SYSTEM OPCUATests
  (* Version 1.0, 2018-08-29, Alois Zoitl, Johannes Kepler University, initial API and implementation and/or initial documentation *)
  APPLICATION OpcUWrongParameters
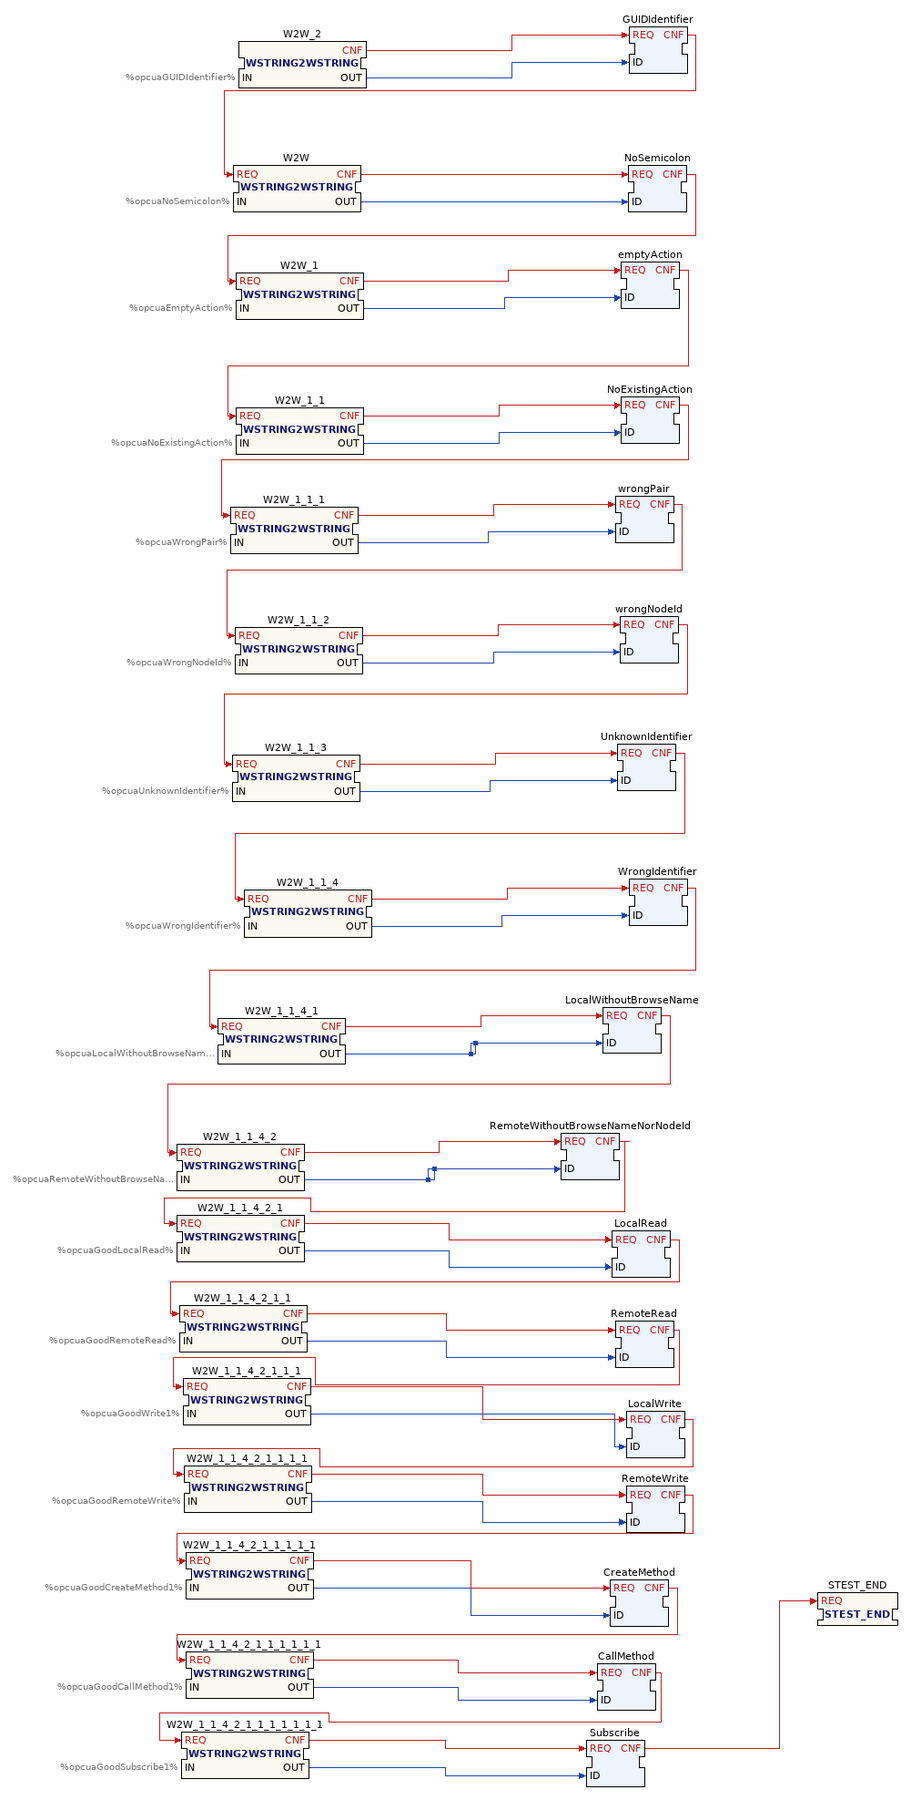
    FBS
      STEST_END : STEST_END;
      W2W : WSTRING2WSTRING(IN := %opcuaNoSemicolon%);
      W2W_1 : WSTRING2WSTRING(IN := %opcuaEmptyAction%);
      W2W_1_1 : WSTRING2WSTRING(IN := %opcuaNoExistingAction%);
      W2W_1_1_1 : WSTRING2WSTRING(IN := %opcuaWrongPair%);
      W2W_1_1_2 : WSTRING2WSTRING(IN := %opcuaWrongNodeId%);
      W2W_1_1_3 : WSTRING2WSTRING(IN := %opcuaUnknownIdentifier%);
      W2W_1_1_4 : WSTRING2WSTRING(IN := %opcuaWrongIdentifier%);
      W2W_1_1_4_1 : WSTRING2WSTRING(IN := %opcuaLocalWithoutBrowseName%);
      W2W_1_1_4_2 : WSTRING2WSTRING(IN := %opcuaRemoteWithoutBrowseNameNorNodeId%);
      W2W_1_1_4_2_1 : WSTRING2WSTRING(IN := %opcuaGoodLocalRead%);
      W2W_1_1_4_2_1_1 : WSTRING2WSTRING(IN := %opcuaGoodRemoteRead%);
      W2W_1_1_4_2_1_1_1 : WSTRING2WSTRING(IN := %opcuaGoodWrite1%);
      W2W_1_1_4_2_1_1_1_1 : WSTRING2WSTRING(IN := %opcuaGoodRemoteWrite%);
      W2W_1_1_4_2_1_1_1_1_1 : WSTRING2WSTRING(IN := %opcuaGoodCreateMethod1%);
      W2W_1_1_4_2_1_1_1_1_1_1 : WSTRING2WSTRING(IN := %opcuaGoodCallMethod1%);
      W2W_1_1_4_2_1_1_1_1_1_1_1 : WSTRING2WSTRING(IN := %opcuaGoodSubscribe1%);
      W2W_2 : WSTRING2WSTRING(IN := %opcuaGUIDIdentifier%);
    END_FBS
    SUBAPPLICATION NoSemicolon
      EVENT_INPUT
        REQ;
      END_EVENT
      EVENT_OUTPUT
        CNF;
      END_EVENT
      VAR_INPUT
        ID : WSTRING;
      END_VAR
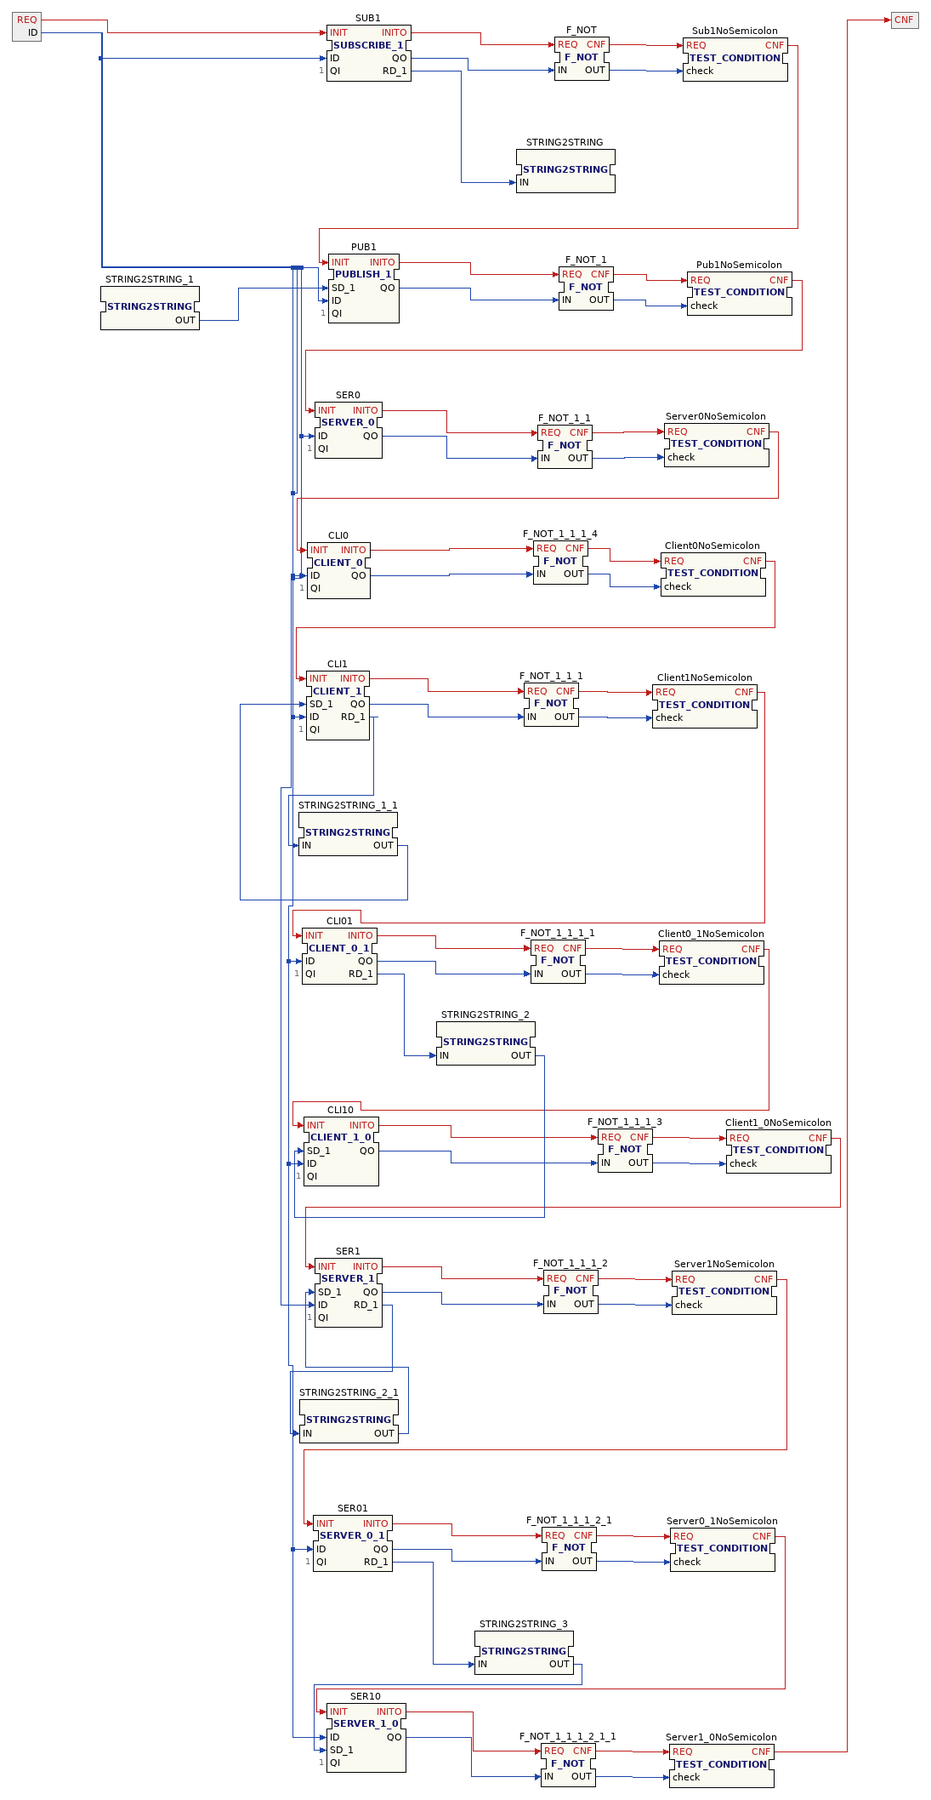
      FBS
        F_NOT_1_1_1 : F_NOT;
        Client1NoSemicolon : TEST_CONDITION;
        Pub1NoSemicolon : TEST_CONDITION;
        F_NOT_1_1 : F_NOT;
        PUB1 : PUBLISH_1(QI := 1);
        F_NOT : F_NOT;
        Server0NoSemicolon : TEST_CONDITION;
        Sub1NoSemicolon : TEST_CONDITION;
        F_NOT_1 : F_NOT;
        STRING2STRING : STRING2STRING;
        SUB1 : SUBSCRIBE_1(QI := 1);
        SER0 : SERVER_0(QI := 1);
        STRING2STRING_1 : STRING2STRING;
        Client0_1NoSemicolon : TEST_CONDITION;
        F_NOT_1_1_1_1 : F_NOT;
        Server1NoSemicolon : TEST_CONDITION;
        F_NOT_1_1_1_2 : F_NOT;
        CLI1 : CLIENT_1(QI := 1);
        CLI01 : CLIENT_0_1(QI := 1);
        Client1_0NoSemicolon : TEST_CONDITION;
        F_NOT_1_1_1_3 : F_NOT;
        CLI10 : CLIENT_1_0(QI := 1);
        STRING2STRING_1_1 : STRING2STRING;
        F_NOT_1_1_1_4 : F_NOT;
        Client0NoSemicolon : TEST_CONDITION;
        CLI0 : CLIENT_0(QI := 1);
        SER1 : SERVER_1(QI := 1);
        F_NOT_1_1_1_2_1 : F_NOT;
        Server0_1NoSemicolon : TEST_CONDITION;
        STRING2STRING_2 : STRING2STRING;
        STRING2STRING_2_1 : STRING2STRING;
        SER01 : SERVER_0_1(QI := 1);
        STRING2STRING_3 : STRING2STRING;
        Server1_0NoSemicolon : TEST_CONDITION;
        F_NOT_1_1_1_2_1_1 : F_NOT;
        SER10 : SERVER_1_0(QI := 1);
      END_FBS
      EVENT_CONNECTIONS
        F_NOT_1_1_1.CNF TO Client1NoSemicolon.REQ;
        F_NOT_1.CNF TO Pub1NoSemicolon.REQ;
        Pub1NoSemicolon.CNF TO SER0.INIT;
        SER0.INITO TO F_NOT_1_1.REQ;
        F_NOT_1_1.CNF TO Server0NoSemicolon.REQ;
        Sub1NoSemicolon.CNF TO PUB1.INIT;
        PUB1.INITO TO F_NOT_1.REQ;
        SUB1.INITO TO F_NOT.REQ;
        F_NOT.CNF TO Sub1NoSemicolon.REQ;
        REQ TO SUB1.INIT;
        F_NOT_1_1_1_1.CNF TO Client0_1NoSemicolon.REQ;
        F_NOT_1_1_1_2.CNF TO Server1NoSemicolon.REQ;
        CLI1.INITO TO F_NOT_1_1_1.REQ;
        CLI01.INITO TO F_NOT_1_1_1_1.REQ;
        CLI0.INITO TO F_NOT_1_1_1_4.REQ;
        F_NOT_1_1_1_4.CNF TO Client0NoSemicolon.REQ;
        F_NOT_1_1_1_3.CNF TO Client1_0NoSemicolon.REQ;
        CLI10.INITO TO F_NOT_1_1_1_3.REQ;
        SER1.INITO TO F_NOT_1_1_1_2.REQ;
        F_NOT_1_1_1_2_1.CNF TO Server0_1NoSemicolon.REQ;
        SER01.INITO TO F_NOT_1_1_1_2_1.REQ;
        Server0NoSemicolon.CNF TO CLI0.INIT;
        Client0NoSemicolon.CNF TO CLI1.INIT;
        Client1NoSemicolon.CNF TO CLI01.INIT;
        Client0_1NoSemicolon.CNF TO CLI10.INIT;
        Client1_0NoSemicolon.CNF TO SER1.INIT;
        Server1NoSemicolon.CNF TO SER01.INIT;
        F_NOT_1_1_1_2_1_1.CNF TO Server1_0NoSemicolon.REQ;
        Server1_0NoSemicolon.CNF TO CNF;
        Server0_1NoSemicolon.CNF TO SER10.INIT;
        SER10.INITO TO F_NOT_1_1_1_2_1_1.REQ;
      END_CONNECTIONS
      DATA_CONNECTIONS
        F_NOT_1_1_1.OUT TO Client1NoSemicolon.check;
        F_NOT_1.OUT TO Pub1NoSemicolon.check;
        SER0.QO TO F_NOT_1_1.IN;
        F_NOT_1_1.OUT TO Server0NoSemicolon.check;
        STRING2STRING_1.OUT TO PUB1.SD_1;
        PUB1.QO TO F_NOT_1.IN;
        SUB1.QO TO F_NOT.IN;
        F_NOT.OUT TO Sub1NoSemicolon.check;
        SUB1.RD_1 TO STRING2STRING.IN;
        F_NOT_1_1_1_1.OUT TO Client0_1NoSemicolon.check;
        F_NOT_1_1_1_2.OUT TO Server1NoSemicolon.check;
        CLI1.QO TO F_NOT_1_1_1.IN;
        CLI01.QO TO F_NOT_1_1_1_1.IN;
        STRING2STRING_1_1.OUT TO CLI1.SD_1;
        CLI1.RD_1 TO STRING2STRING_1_1.IN;
        F_NOT_1_1_1_4.OUT TO Client0NoSemicolon.check;
        CLI0.QO TO F_NOT_1_1_1_4.IN;
        F_NOT_1_1_1_3.OUT TO Client1_0NoSemicolon.check;
        CLI10.QO TO F_NOT_1_1_1_3.IN;
        SER1.QO TO F_NOT_1_1_1_2.IN;
        F_NOT_1_1_1_2_1.OUT TO Server0_1NoSemicolon.check;
        CLI01.RD_1 TO STRING2STRING_2.IN;
        STRING2STRING_2.OUT TO CLI10.SD_1;
        STRING2STRING_2_1.OUT TO SER1.SD_1;
        SER1.RD_1 TO STRING2STRING_2_1.IN;
        SER01.QO TO F_NOT_1_1_1_2_1.IN;
        SER01.RD_1 TO STRING2STRING_3.IN;
        ID TO SUB1.ID;
        ID TO PUB1.ID;
        ID TO SER0.ID;
        ID TO CLI0.ID;
        ID TO CLI1.ID;
        ID TO CLI01.ID;
        ID TO CLI10.ID;
        ID TO SER01.ID;
        ID TO SER1.ID;
        F_NOT_1_1_1_2_1_1.OUT TO Server1_0NoSemicolon.check;
        ID TO SER10.ID;
        SER10.QO TO F_NOT_1_1_1_2_1_1.IN;
        STRING2STRING_3.OUT TO SER10.SD_1;
      END_CONNECTIONS
    END_SUBAPPLICATION
    SUBAPPLICATION emptyAction
      EVENT_INPUT
        REQ;
      END_EVENT
      EVENT_OUTPUT
        CNF;
      END_EVENT
      VAR_INPUT
        ID : WSTRING;
      END_VAR
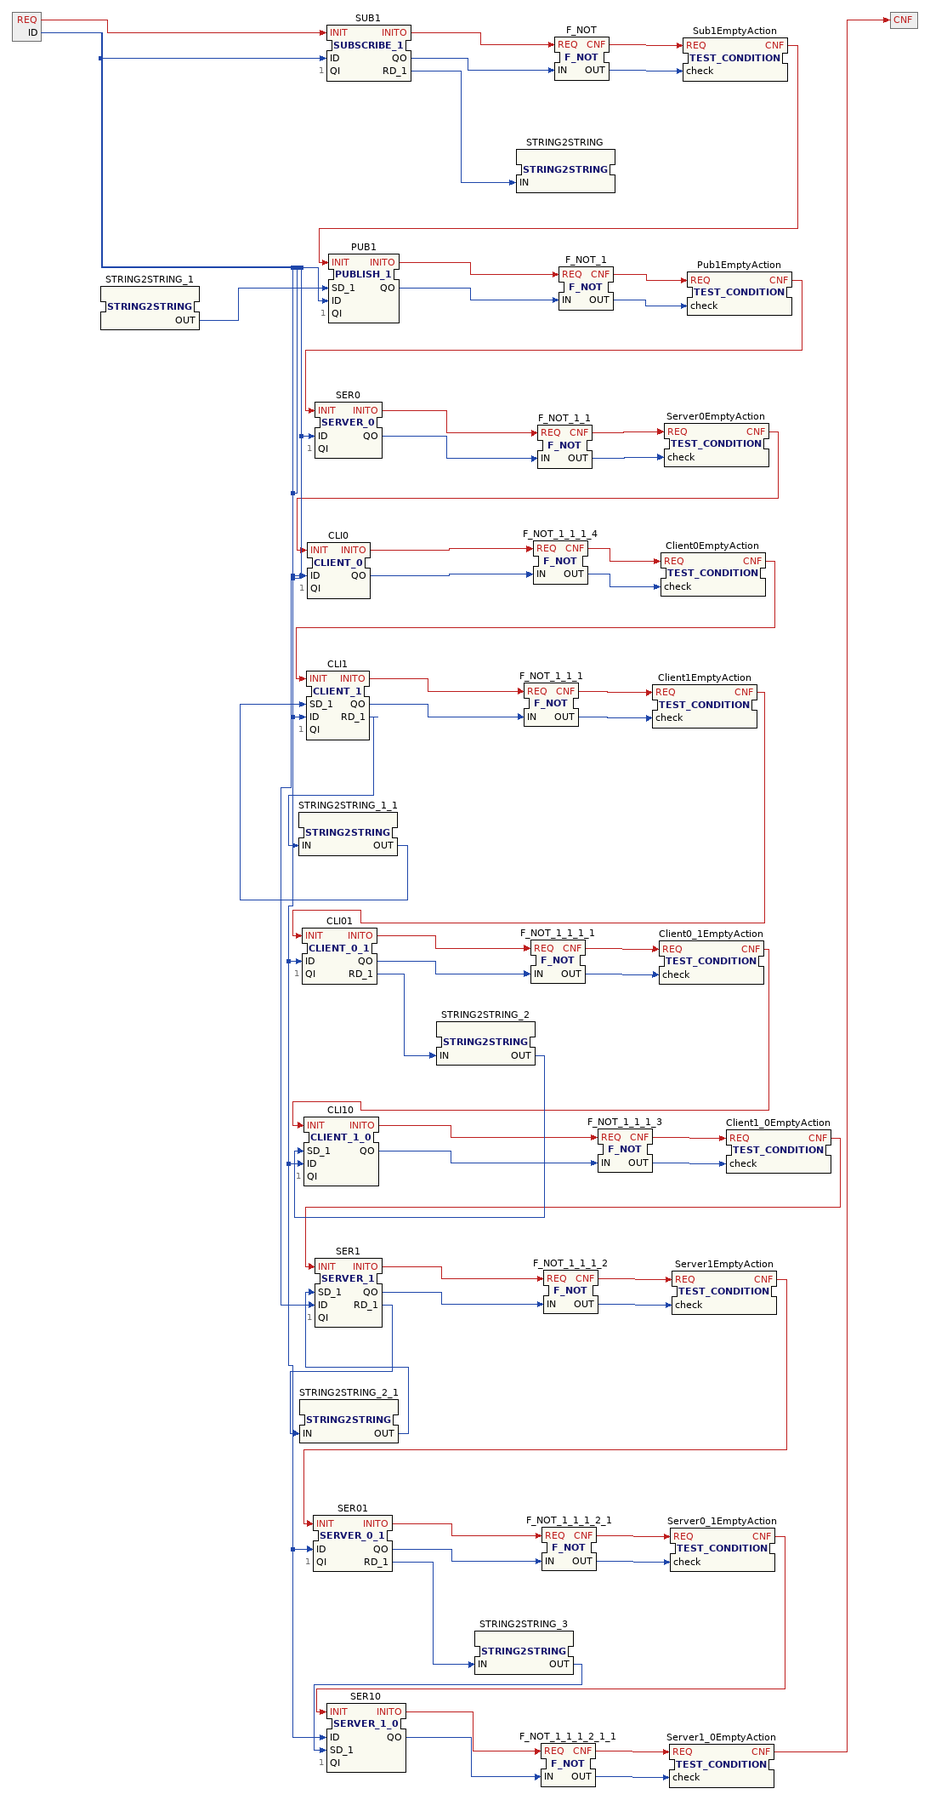
      FBS
        F_NOT_1_1_1 : F_NOT;
        Client1EmptyAction : TEST_CONDITION;
        Pub1EmptyAction : TEST_CONDITION;
        F_NOT_1_1 : F_NOT;
        PUB1 : PUBLISH_1(QI := 1);
        F_NOT : F_NOT;
        Server0EmptyAction : TEST_CONDITION;
        Sub1EmptyAction : TEST_CONDITION;
        F_NOT_1 : F_NOT;
        STRING2STRING : STRING2STRING;
        SUB1 : SUBSCRIBE_1(QI := 1);
        SER0 : SERVER_0(QI := 1);
        STRING2STRING_1 : STRING2STRING;
        Client0_1EmptyAction : TEST_CONDITION;
        F_NOT_1_1_1_1 : F_NOT;
        Server1EmptyAction : TEST_CONDITION;
        F_NOT_1_1_1_2 : F_NOT;
        CLI1 : CLIENT_1(QI := 1);
        CLI01 : CLIENT_0_1(QI := 1);
        Client1_0EmptyAction : TEST_CONDITION;
        F_NOT_1_1_1_3 : F_NOT;
        CLI10 : CLIENT_1_0(QI := 1);
        STRING2STRING_1_1 : STRING2STRING;
        F_NOT_1_1_1_4 : F_NOT;
        Client0EmptyAction : TEST_CONDITION;
        CLI0 : CLIENT_0(QI := 1);
        SER1 : SERVER_1(QI := 1);
        F_NOT_1_1_1_2_1 : F_NOT;
        Server0_1EmptyAction : TEST_CONDITION;
        STRING2STRING_2 : STRING2STRING;
        STRING2STRING_2_1 : STRING2STRING;
        SER01 : SERVER_0_1(QI := 1);
        STRING2STRING_3 : STRING2STRING;
        Server1_0EmptyAction : TEST_CONDITION;
        F_NOT_1_1_1_2_1_1 : F_NOT;
        SER10 : SERVER_1_0(QI := 1);
      END_FBS
      EVENT_CONNECTIONS
        F_NOT_1_1_1.CNF TO Client1EmptyAction.REQ;
        F_NOT_1.CNF TO Pub1EmptyAction.REQ;
        Pub1EmptyAction.CNF TO SER0.INIT;
        SER0.INITO TO F_NOT_1_1.REQ;
        F_NOT_1_1.CNF TO Server0EmptyAction.REQ;
        Sub1EmptyAction.CNF TO PUB1.INIT;
        PUB1.INITO TO F_NOT_1.REQ;
        SUB1.INITO TO F_NOT.REQ;
        F_NOT.CNF TO Sub1EmptyAction.REQ;
        REQ TO SUB1.INIT;
        F_NOT_1_1_1_1.CNF TO Client0_1EmptyAction.REQ;
        F_NOT_1_1_1_2.CNF TO Server1EmptyAction.REQ;
        CLI1.INITO TO F_NOT_1_1_1.REQ;
        CLI01.INITO TO F_NOT_1_1_1_1.REQ;
        CLI0.INITO TO F_NOT_1_1_1_4.REQ;
        F_NOT_1_1_1_4.CNF TO Client0EmptyAction.REQ;
        F_NOT_1_1_1_3.CNF TO Client1_0EmptyAction.REQ;
        CLI10.INITO TO F_NOT_1_1_1_3.REQ;
        SER1.INITO TO F_NOT_1_1_1_2.REQ;
        F_NOT_1_1_1_2_1.CNF TO Server0_1EmptyAction.REQ;
        SER01.INITO TO F_NOT_1_1_1_2_1.REQ;
        Server0EmptyAction.CNF TO CLI0.INIT;
        Client0EmptyAction.CNF TO CLI1.INIT;
        Client1EmptyAction.CNF TO CLI01.INIT;
        Client0_1EmptyAction.CNF TO CLI10.INIT;
        Client1_0EmptyAction.CNF TO SER1.INIT;
        Server1EmptyAction.CNF TO SER01.INIT;
        F_NOT_1_1_1_2_1_1.CNF TO Server1_0EmptyAction.REQ;
        Server1_0EmptyAction.CNF TO CNF;
        Server0_1EmptyAction.CNF TO SER10.INIT;
        SER10.INITO TO F_NOT_1_1_1_2_1_1.REQ;
      END_CONNECTIONS
      DATA_CONNECTIONS
        F_NOT_1_1_1.OUT TO Client1EmptyAction.check;
        F_NOT_1.OUT TO Pub1EmptyAction.check;
        SER0.QO TO F_NOT_1_1.IN;
        F_NOT_1_1.OUT TO Server0EmptyAction.check;
        STRING2STRING_1.OUT TO PUB1.SD_1;
        PUB1.QO TO F_NOT_1.IN;
        SUB1.QO TO F_NOT.IN;
        F_NOT.OUT TO Sub1EmptyAction.check;
        SUB1.RD_1 TO STRING2STRING.IN;
        F_NOT_1_1_1_1.OUT TO Client0_1EmptyAction.check;
        F_NOT_1_1_1_2.OUT TO Server1EmptyAction.check;
        CLI1.QO TO F_NOT_1_1_1.IN;
        CLI01.QO TO F_NOT_1_1_1_1.IN;
        STRING2STRING_1_1.OUT TO CLI1.SD_1;
        CLI1.RD_1 TO STRING2STRING_1_1.IN;
        F_NOT_1_1_1_4.OUT TO Client0EmptyAction.check;
        CLI0.QO TO F_NOT_1_1_1_4.IN;
        F_NOT_1_1_1_3.OUT TO Client1_0EmptyAction.check;
        CLI10.QO TO F_NOT_1_1_1_3.IN;
        SER1.QO TO F_NOT_1_1_1_2.IN;
        F_NOT_1_1_1_2_1.OUT TO Server0_1EmptyAction.check;
        CLI01.RD_1 TO STRING2STRING_2.IN;
        STRING2STRING_2.OUT TO CLI10.SD_1;
        STRING2STRING_2_1.OUT TO SER1.SD_1;
        SER1.RD_1 TO STRING2STRING_2_1.IN;
        SER01.QO TO F_NOT_1_1_1_2_1.IN;
        SER01.RD_1 TO STRING2STRING_3.IN;
        ID TO SUB1.ID;
        ID TO PUB1.ID;
        ID TO SER0.ID;
        ID TO CLI0.ID;
        ID TO CLI1.ID;
        ID TO CLI01.ID;
        ID TO CLI10.ID;
        ID TO SER01.ID;
        ID TO SER1.ID;
        F_NOT_1_1_1_2_1_1.OUT TO Server1_0EmptyAction.check;
        ID TO SER10.ID;
        SER10.QO TO F_NOT_1_1_1_2_1_1.IN;
        STRING2STRING_3.OUT TO SER10.SD_1;
      END_CONNECTIONS
    END_SUBAPPLICATION
    SUBAPPLICATION NoExistingAction
      EVENT_INPUT
        REQ;
      END_EVENT
      EVENT_OUTPUT
        CNF;
      END_EVENT
      VAR_INPUT
        ID : WSTRING;
      END_VAR
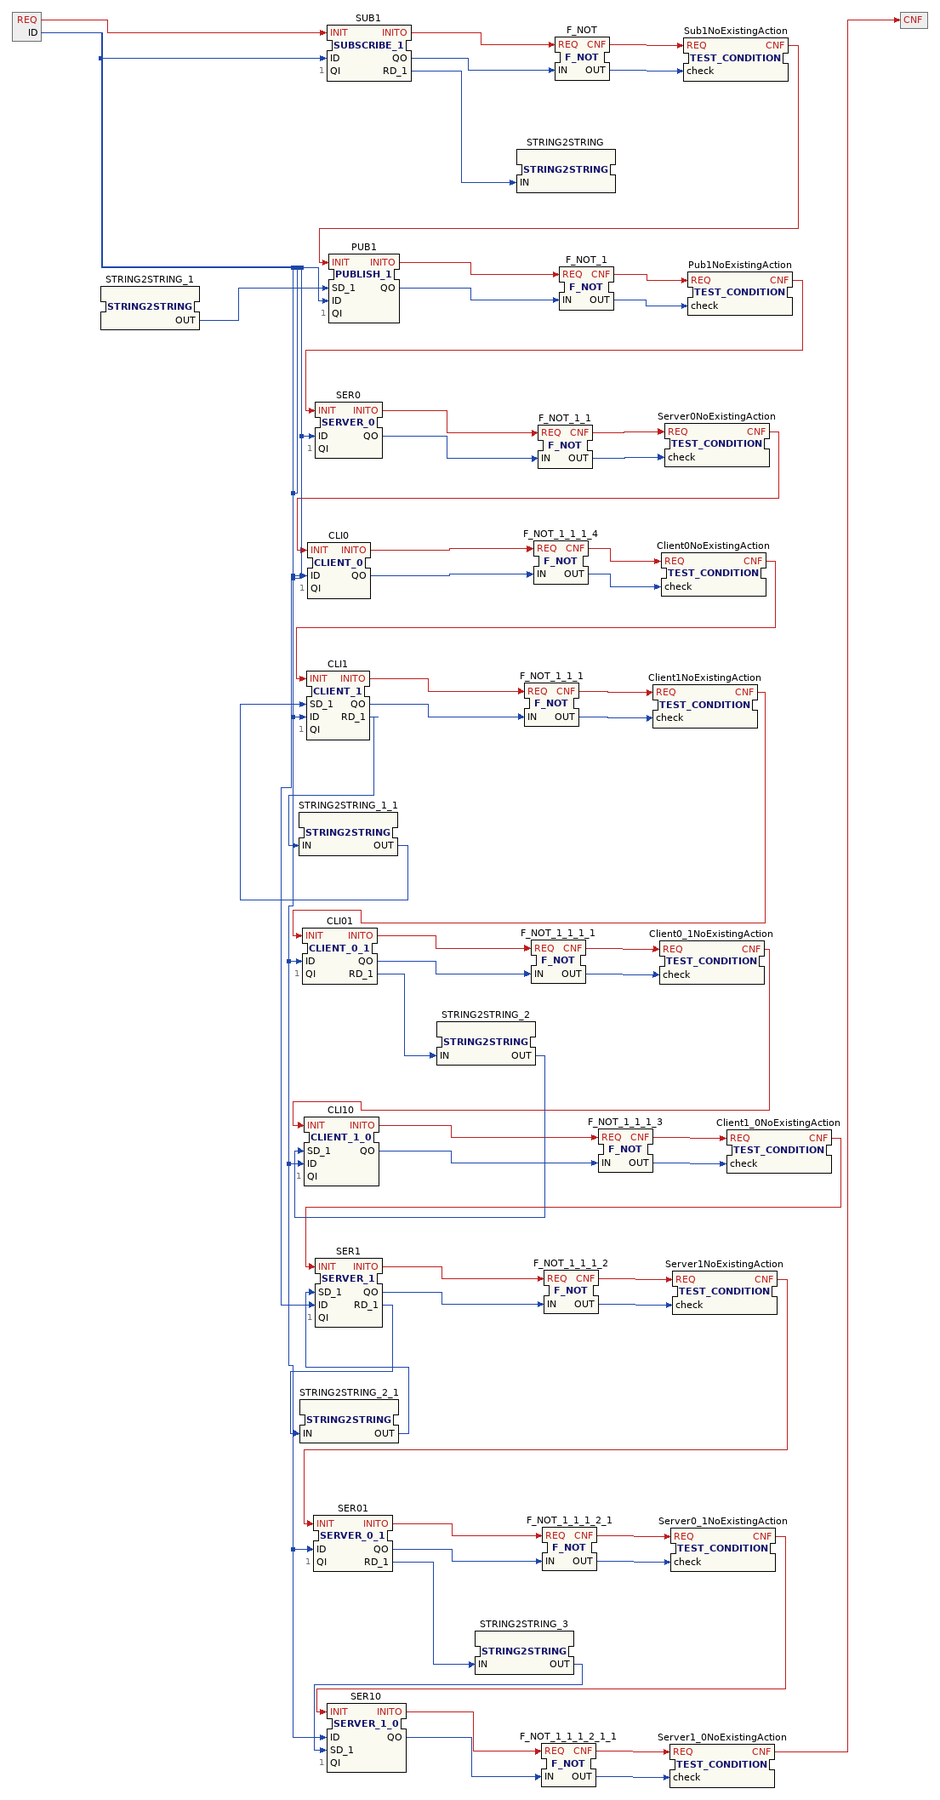
      FBS
        F_NOT_1_1_1 : F_NOT;
        Client1NoExistingAction : TEST_CONDITION;
        Pub1NoExistingAction : TEST_CONDITION;
        F_NOT_1_1 : F_NOT;
        PUB1 : PUBLISH_1(QI := 1);
        F_NOT : F_NOT;
        Server0NoExistingAction : TEST_CONDITION;
        Sub1NoExistingAction : TEST_CONDITION;
        F_NOT_1 : F_NOT;
        STRING2STRING : STRING2STRING;
        SUB1 : SUBSCRIBE_1(QI := 1);
        SER0 : SERVER_0(QI := 1);
        STRING2STRING_1 : STRING2STRING;
        Client0_1NoExistingAction : TEST_CONDITION;
        F_NOT_1_1_1_1 : F_NOT;
        Server1NoExistingAction : TEST_CONDITION;
        F_NOT_1_1_1_2 : F_NOT;
        CLI1 : CLIENT_1(QI := 1);
        CLI01 : CLIENT_0_1(QI := 1);
        Client1_0NoExistingAction : TEST_CONDITION;
        F_NOT_1_1_1_3 : F_NOT;
        CLI10 : CLIENT_1_0(QI := 1);
        STRING2STRING_1_1 : STRING2STRING;
        F_NOT_1_1_1_4 : F_NOT;
        Client0NoExistingAction : TEST_CONDITION;
        CLI0 : CLIENT_0(QI := 1);
        SER1 : SERVER_1(QI := 1);
        F_NOT_1_1_1_2_1 : F_NOT;
        Server0_1NoExistingAction : TEST_CONDITION;
        STRING2STRING_2 : STRING2STRING;
        STRING2STRING_2_1 : STRING2STRING;
        SER01 : SERVER_0_1(QI := 1);
        STRING2STRING_3 : STRING2STRING;
        Server1_0NoExistingAction : TEST_CONDITION;
        F_NOT_1_1_1_2_1_1 : F_NOT;
        SER10 : SERVER_1_0(QI := 1);
      END_FBS
      EVENT_CONNECTIONS
        F_NOT_1_1_1.CNF TO Client1NoExistingAction.REQ;
        F_NOT_1.CNF TO Pub1NoExistingAction.REQ;
        Pub1NoExistingAction.CNF TO SER0.INIT;
        SER0.INITO TO F_NOT_1_1.REQ;
        F_NOT_1_1.CNF TO Server0NoExistingAction.REQ;
        Sub1NoExistingAction.CNF TO PUB1.INIT;
        PUB1.INITO TO F_NOT_1.REQ;
        SUB1.INITO TO F_NOT.REQ;
        F_NOT.CNF TO Sub1NoExistingAction.REQ;
        REQ TO SUB1.INIT;
        F_NOT_1_1_1_1.CNF TO Client0_1NoExistingAction.REQ;
        F_NOT_1_1_1_2.CNF TO Server1NoExistingAction.REQ;
        CLI1.INITO TO F_NOT_1_1_1.REQ;
        CLI01.INITO TO F_NOT_1_1_1_1.REQ;
        CLI0.INITO TO F_NOT_1_1_1_4.REQ;
        F_NOT_1_1_1_4.CNF TO Client0NoExistingAction.REQ;
        F_NOT_1_1_1_3.CNF TO Client1_0NoExistingAction.REQ;
        CLI10.INITO TO F_NOT_1_1_1_3.REQ;
        SER1.INITO TO F_NOT_1_1_1_2.REQ;
        F_NOT_1_1_1_2_1.CNF TO Server0_1NoExistingAction.REQ;
        SER01.INITO TO F_NOT_1_1_1_2_1.REQ;
        Server0NoExistingAction.CNF TO CLI0.INIT;
        Client0NoExistingAction.CNF TO CLI1.INIT;
        Client1NoExistingAction.CNF TO CLI01.INIT;
        Client0_1NoExistingAction.CNF TO CLI10.INIT;
        Client1_0NoExistingAction.CNF TO SER1.INIT;
        Server1NoExistingAction.CNF TO SER01.INIT;
        F_NOT_1_1_1_2_1_1.CNF TO Server1_0NoExistingAction.REQ;
        Server1_0NoExistingAction.CNF TO CNF;
        Server0_1NoExistingAction.CNF TO SER10.INIT;
        SER10.INITO TO F_NOT_1_1_1_2_1_1.REQ;
      END_CONNECTIONS
      DATA_CONNECTIONS
        F_NOT_1_1_1.OUT TO Client1NoExistingAction.check;
        F_NOT_1.OUT TO Pub1NoExistingAction.check;
        SER0.QO TO F_NOT_1_1.IN;
        F_NOT_1_1.OUT TO Server0NoExistingAction.check;
        STRING2STRING_1.OUT TO PUB1.SD_1;
        PUB1.QO TO F_NOT_1.IN;
        SUB1.QO TO F_NOT.IN;
        F_NOT.OUT TO Sub1NoExistingAction.check;
        SUB1.RD_1 TO STRING2STRING.IN;
        F_NOT_1_1_1_1.OUT TO Client0_1NoExistingAction.check;
        F_NOT_1_1_1_2.OUT TO Server1NoExistingAction.check;
        CLI1.QO TO F_NOT_1_1_1.IN;
        CLI01.QO TO F_NOT_1_1_1_1.IN;
        STRING2STRING_1_1.OUT TO CLI1.SD_1;
        CLI1.RD_1 TO STRING2STRING_1_1.IN;
        F_NOT_1_1_1_4.OUT TO Client0NoExistingAction.check;
        CLI0.QO TO F_NOT_1_1_1_4.IN;
        F_NOT_1_1_1_3.OUT TO Client1_0NoExistingAction.check;
        CLI10.QO TO F_NOT_1_1_1_3.IN;
        SER1.QO TO F_NOT_1_1_1_2.IN;
        F_NOT_1_1_1_2_1.OUT TO Server0_1NoExistingAction.check;
        CLI01.RD_1 TO STRING2STRING_2.IN;
        STRING2STRING_2.OUT TO CLI10.SD_1;
        STRING2STRING_2_1.OUT TO SER1.SD_1;
        SER1.RD_1 TO STRING2STRING_2_1.IN;
        SER01.QO TO F_NOT_1_1_1_2_1.IN;
        SER01.RD_1 TO STRING2STRING_3.IN;
        ID TO SUB1.ID;
        ID TO PUB1.ID;
        ID TO SER0.ID;
        ID TO CLI0.ID;
        ID TO CLI1.ID;
        ID TO CLI01.ID;
        ID TO CLI10.ID;
        ID TO SER01.ID;
        ID TO SER1.ID;
        F_NOT_1_1_1_2_1_1.OUT TO Server1_0NoExistingAction.check;
        ID TO SER10.ID;
        SER10.QO TO F_NOT_1_1_1_2_1_1.IN;
        STRING2STRING_3.OUT TO SER10.SD_1;
      END_CONNECTIONS
    END_SUBAPPLICATION
    SUBAPPLICATION wrongPair
      EVENT_INPUT
        REQ;
      END_EVENT
      EVENT_OUTPUT
        CNF;
      END_EVENT
      VAR_INPUT
        ID : WSTRING;
      END_VAR
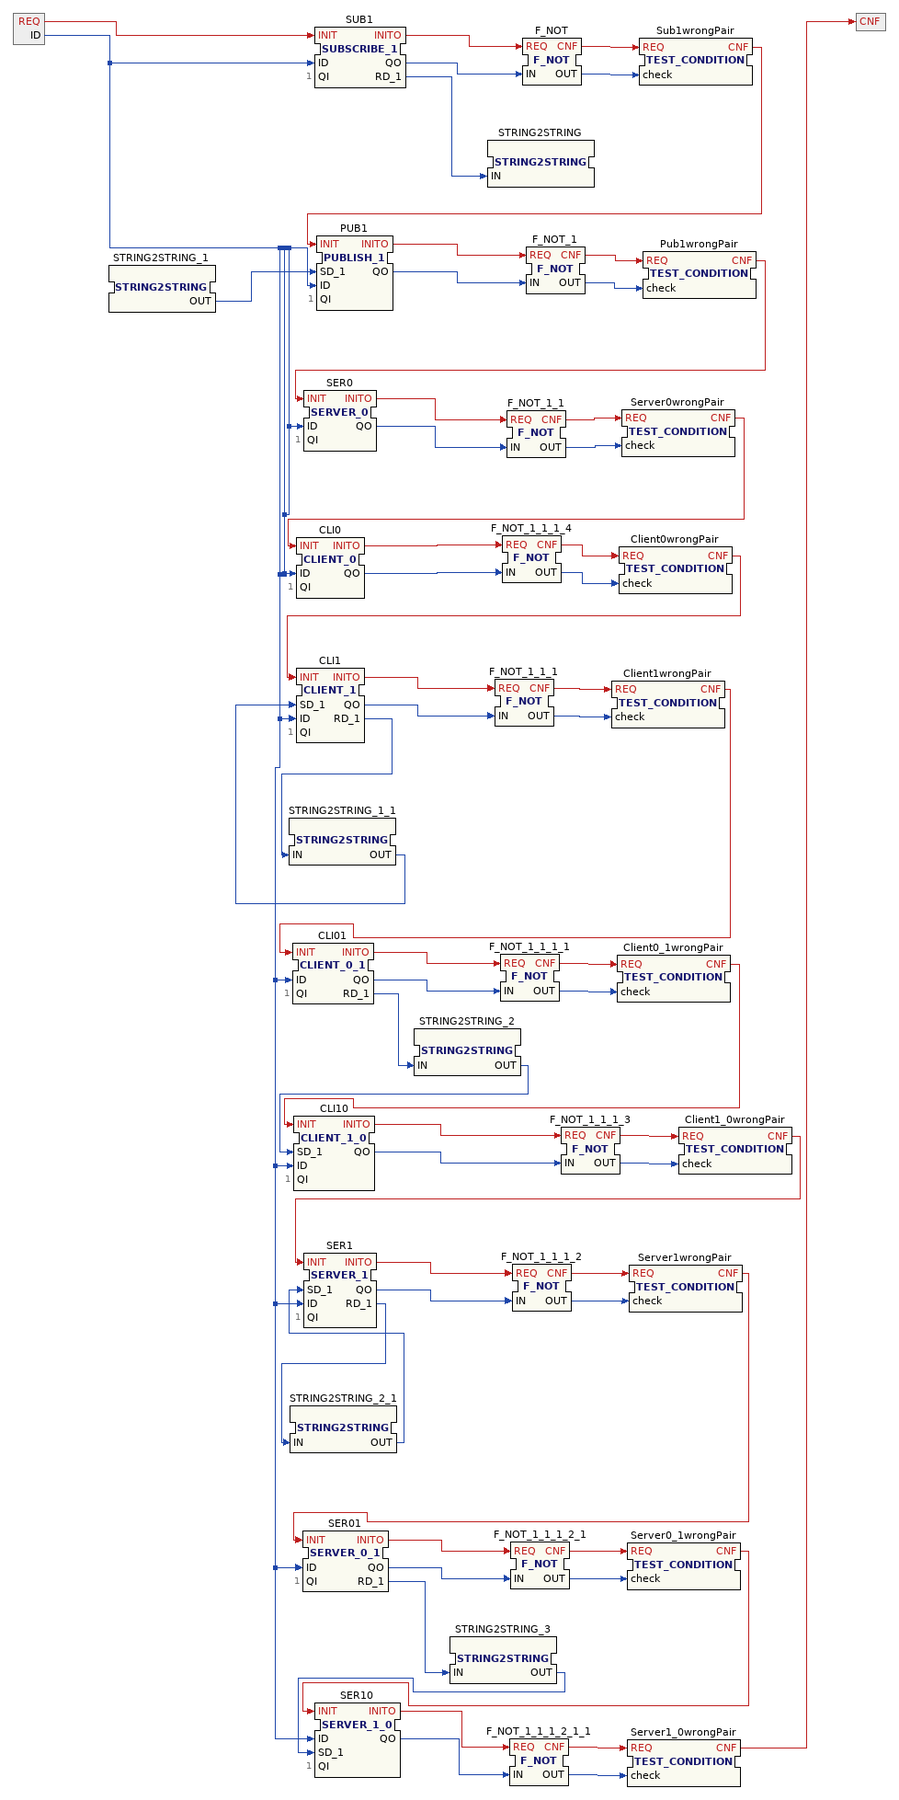
      FBS
        F_NOT_1_1_1 : F_NOT;
        Client1wrongPair : TEST_CONDITION;
        Pub1wrongPair : TEST_CONDITION;
        F_NOT_1_1 : F_NOT;
        PUB1 : PUBLISH_1(QI := 1);
        F_NOT : F_NOT;
        Server0wrongPair : TEST_CONDITION;
        Sub1wrongPair : TEST_CONDITION;
        F_NOT_1 : F_NOT;
        STRING2STRING : STRING2STRING;
        SUB1 : SUBSCRIBE_1(QI := 1);
        SER0 : SERVER_0(QI := 1);
        STRING2STRING_1 : STRING2STRING;
        Client0_1wrongPair : TEST_CONDITION;
        F_NOT_1_1_1_1 : F_NOT;
        Server1wrongPair : TEST_CONDITION;
        F_NOT_1_1_1_2 : F_NOT;
        CLI1 : CLIENT_1(QI := 1);
        CLI01 : CLIENT_0_1(QI := 1);
        Client1_0wrongPair : TEST_CONDITION;
        F_NOT_1_1_1_3 : F_NOT;
        CLI10 : CLIENT_1_0(QI := 1);
        STRING2STRING_1_1 : STRING2STRING;
        F_NOT_1_1_1_4 : F_NOT;
        Client0wrongPair : TEST_CONDITION;
        CLI0 : CLIENT_0(QI := 1);
        SER1 : SERVER_1(QI := 1);
        F_NOT_1_1_1_2_1 : F_NOT;
        Server0_1wrongPair : TEST_CONDITION;
        STRING2STRING_2 : STRING2STRING;
        STRING2STRING_2_1 : STRING2STRING;
        SER01 : SERVER_0_1(QI := 1);
        STRING2STRING_3 : STRING2STRING;
        Server1_0wrongPair : TEST_CONDITION;
        F_NOT_1_1_1_2_1_1 : F_NOT;
        SER10 : SERVER_1_0(QI := 1);
      END_FBS
      EVENT_CONNECTIONS
        F_NOT_1_1_1.CNF TO Client1wrongPair.REQ;
        F_NOT_1.CNF TO Pub1wrongPair.REQ;
        Pub1wrongPair.CNF TO SER0.INIT;
        SER0.INITO TO F_NOT_1_1.REQ;
        F_NOT_1_1.CNF TO Server0wrongPair.REQ;
        Sub1wrongPair.CNF TO PUB1.INIT;
        PUB1.INITO TO F_NOT_1.REQ;
        SUB1.INITO TO F_NOT.REQ;
        F_NOT.CNF TO Sub1wrongPair.REQ;
        REQ TO SUB1.INIT;
        F_NOT_1_1_1_1.CNF TO Client0_1wrongPair.REQ;
        F_NOT_1_1_1_2.CNF TO Server1wrongPair.REQ;
        CLI1.INITO TO F_NOT_1_1_1.REQ;
        CLI01.INITO TO F_NOT_1_1_1_1.REQ;
        CLI0.INITO TO F_NOT_1_1_1_4.REQ;
        F_NOT_1_1_1_4.CNF TO Client0wrongPair.REQ;
        F_NOT_1_1_1_3.CNF TO Client1_0wrongPair.REQ;
        CLI10.INITO TO F_NOT_1_1_1_3.REQ;
        SER1.INITO TO F_NOT_1_1_1_2.REQ;
        F_NOT_1_1_1_2_1.CNF TO Server0_1wrongPair.REQ;
        SER01.INITO TO F_NOT_1_1_1_2_1.REQ;
        Server0wrongPair.CNF TO CLI0.INIT;
        Client0wrongPair.CNF TO CLI1.INIT;
        Client1wrongPair.CNF TO CLI01.INIT;
        Client0_1wrongPair.CNF TO CLI10.INIT;
        Client1_0wrongPair.CNF TO SER1.INIT;
        Server1wrongPair.CNF TO SER01.INIT;
        F_NOT_1_1_1_2_1_1.CNF TO Server1_0wrongPair.REQ;
        Server1_0wrongPair.CNF TO CNF;
        Server0_1wrongPair.CNF TO SER10.INIT;
        SER10.INITO TO F_NOT_1_1_1_2_1_1.REQ;
      END_CONNECTIONS
      DATA_CONNECTIONS
        F_NOT_1_1_1.OUT TO Client1wrongPair.check;
        F_NOT_1.OUT TO Pub1wrongPair.check;
        SER0.QO TO F_NOT_1_1.IN;
        F_NOT_1_1.OUT TO Server0wrongPair.check;
        STRING2STRING_1.OUT TO PUB1.SD_1;
        PUB1.QO TO F_NOT_1.IN;
        SUB1.QO TO F_NOT.IN;
        F_NOT.OUT TO Sub1wrongPair.check;
        SUB1.RD_1 TO STRING2STRING.IN;
        F_NOT_1_1_1_1.OUT TO Client0_1wrongPair.check;
        F_NOT_1_1_1_2.OUT TO Server1wrongPair.check;
        CLI1.QO TO F_NOT_1_1_1.IN;
        CLI01.QO TO F_NOT_1_1_1_1.IN;
        STRING2STRING_1_1.OUT TO CLI1.SD_1;
        CLI1.RD_1 TO STRING2STRING_1_1.IN;
        F_NOT_1_1_1_4.OUT TO Client0wrongPair.check;
        CLI0.QO TO F_NOT_1_1_1_4.IN;
        F_NOT_1_1_1_3.OUT TO Client1_0wrongPair.check;
        CLI10.QO TO F_NOT_1_1_1_3.IN;
        SER1.QO TO F_NOT_1_1_1_2.IN;
        F_NOT_1_1_1_2_1.OUT TO Server0_1wrongPair.check;
        CLI01.RD_1 TO STRING2STRING_2.IN;
        STRING2STRING_2.OUT TO CLI10.SD_1;
        STRING2STRING_2_1.OUT TO SER1.SD_1;
        SER1.RD_1 TO STRING2STRING_2_1.IN;
        SER01.QO TO F_NOT_1_1_1_2_1.IN;
        SER01.RD_1 TO STRING2STRING_3.IN;
        ID TO SUB1.ID;
        ID TO PUB1.ID;
        ID TO SER0.ID;
        ID TO CLI0.ID;
        ID TO CLI1.ID;
        ID TO CLI01.ID;
        ID TO CLI10.ID;
        ID TO SER01.ID;
        ID TO SER1.ID;
        F_NOT_1_1_1_2_1_1.OUT TO Server1_0wrongPair.check;
        ID TO SER10.ID;
        SER10.QO TO F_NOT_1_1_1_2_1_1.IN;
        STRING2STRING_3.OUT TO SER10.SD_1;
      END_CONNECTIONS
    END_SUBAPPLICATION
    SUBAPPLICATION wrongNodeId
      EVENT_INPUT
        REQ;
      END_EVENT
      EVENT_OUTPUT
        CNF;
      END_EVENT
      VAR_INPUT
        ID : WSTRING;
      END_VAR
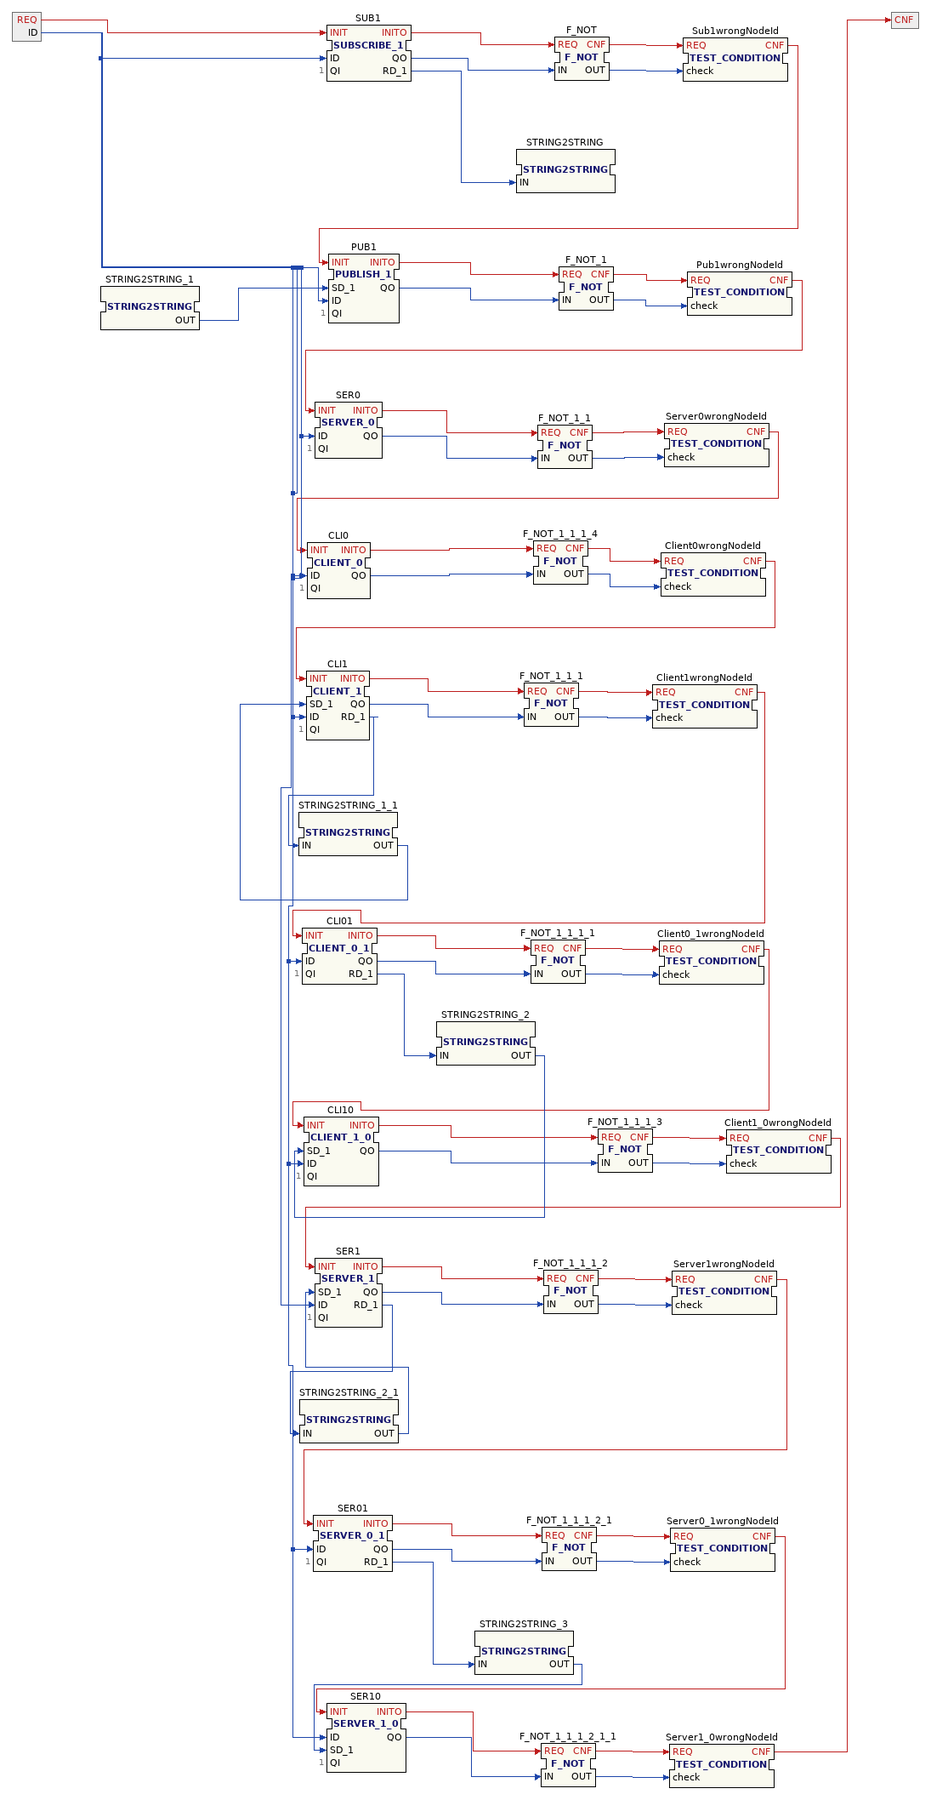
      FBS
        F_NOT_1_1_1 : F_NOT;
        Client1wrongNodeId : TEST_CONDITION;
        Pub1wrongNodeId : TEST_CONDITION;
        F_NOT_1_1 : F_NOT;
        PUB1 : PUBLISH_1(QI := 1);
        F_NOT : F_NOT;
        Server0wrongNodeId : TEST_CONDITION;
        Sub1wrongNodeId : TEST_CONDITION;
        F_NOT_1 : F_NOT;
        STRING2STRING : STRING2STRING;
        SUB1 : SUBSCRIBE_1(QI := 1);
        SER0 : SERVER_0(QI := 1);
        STRING2STRING_1 : STRING2STRING;
        Client0_1wrongNodeId : TEST_CONDITION;
        F_NOT_1_1_1_1 : F_NOT;
        Server1wrongNodeId : TEST_CONDITION;
        F_NOT_1_1_1_2 : F_NOT;
        CLI1 : CLIENT_1(QI := 1);
        CLI01 : CLIENT_0_1(QI := 1);
        Client1_0wrongNodeId : TEST_CONDITION;
        F_NOT_1_1_1_3 : F_NOT;
        CLI10 : CLIENT_1_0(QI := 1);
        STRING2STRING_1_1 : STRING2STRING;
        F_NOT_1_1_1_4 : F_NOT;
        Client0wrongNodeId : TEST_CONDITION;
        CLI0 : CLIENT_0(QI := 1);
        SER1 : SERVER_1(QI := 1);
        F_NOT_1_1_1_2_1 : F_NOT;
        Server0_1wrongNodeId : TEST_CONDITION;
        STRING2STRING_2 : STRING2STRING;
        STRING2STRING_2_1 : STRING2STRING;
        SER01 : SERVER_0_1(QI := 1);
        STRING2STRING_3 : STRING2STRING;
        Server1_0wrongNodeId : TEST_CONDITION;
        F_NOT_1_1_1_2_1_1 : F_NOT;
        SER10 : SERVER_1_0(QI := 1);
      END_FBS
      EVENT_CONNECTIONS
        F_NOT_1_1_1.CNF TO Client1wrongNodeId.REQ;
        F_NOT_1.CNF TO Pub1wrongNodeId.REQ;
        Pub1wrongNodeId.CNF TO SER0.INIT;
        SER0.INITO TO F_NOT_1_1.REQ;
        F_NOT_1_1.CNF TO Server0wrongNodeId.REQ;
        Sub1wrongNodeId.CNF TO PUB1.INIT;
        PUB1.INITO TO F_NOT_1.REQ;
        SUB1.INITO TO F_NOT.REQ;
        F_NOT.CNF TO Sub1wrongNodeId.REQ;
        REQ TO SUB1.INIT;
        F_NOT_1_1_1_1.CNF TO Client0_1wrongNodeId.REQ;
        F_NOT_1_1_1_2.CNF TO Server1wrongNodeId.REQ;
        CLI1.INITO TO F_NOT_1_1_1.REQ;
        CLI01.INITO TO F_NOT_1_1_1_1.REQ;
        CLI0.INITO TO F_NOT_1_1_1_4.REQ;
        F_NOT_1_1_1_4.CNF TO Client0wrongNodeId.REQ;
        F_NOT_1_1_1_3.CNF TO Client1_0wrongNodeId.REQ;
        CLI10.INITO TO F_NOT_1_1_1_3.REQ;
        SER1.INITO TO F_NOT_1_1_1_2.REQ;
        F_NOT_1_1_1_2_1.CNF TO Server0_1wrongNodeId.REQ;
        SER01.INITO TO F_NOT_1_1_1_2_1.REQ;
        Server0wrongNodeId.CNF TO CLI0.INIT;
        Client0wrongNodeId.CNF TO CLI1.INIT;
        Client1wrongNodeId.CNF TO CLI01.INIT;
        Client0_1wrongNodeId.CNF TO CLI10.INIT;
        Client1_0wrongNodeId.CNF TO SER1.INIT;
        Server1wrongNodeId.CNF TO SER01.INIT;
        F_NOT_1_1_1_2_1_1.CNF TO Server1_0wrongNodeId.REQ;
        Server1_0wrongNodeId.CNF TO CNF;
        Server0_1wrongNodeId.CNF TO SER10.INIT;
        SER10.INITO TO F_NOT_1_1_1_2_1_1.REQ;
      END_CONNECTIONS
      DATA_CONNECTIONS
        F_NOT_1_1_1.OUT TO Client1wrongNodeId.check;
        F_NOT_1.OUT TO Pub1wrongNodeId.check;
        SER0.QO TO F_NOT_1_1.IN;
        F_NOT_1_1.OUT TO Server0wrongNodeId.check;
        STRING2STRING_1.OUT TO PUB1.SD_1;
        PUB1.QO TO F_NOT_1.IN;
        SUB1.QO TO F_NOT.IN;
        F_NOT.OUT TO Sub1wrongNodeId.check;
        SUB1.RD_1 TO STRING2STRING.IN;
        F_NOT_1_1_1_1.OUT TO Client0_1wrongNodeId.check;
        F_NOT_1_1_1_2.OUT TO Server1wrongNodeId.check;
        CLI1.QO TO F_NOT_1_1_1.IN;
        CLI01.QO TO F_NOT_1_1_1_1.IN;
        STRING2STRING_1_1.OUT TO CLI1.SD_1;
        CLI1.RD_1 TO STRING2STRING_1_1.IN;
        F_NOT_1_1_1_4.OUT TO Client0wrongNodeId.check;
        CLI0.QO TO F_NOT_1_1_1_4.IN;
        F_NOT_1_1_1_3.OUT TO Client1_0wrongNodeId.check;
        CLI10.QO TO F_NOT_1_1_1_3.IN;
        SER1.QO TO F_NOT_1_1_1_2.IN;
        F_NOT_1_1_1_2_1.OUT TO Server0_1wrongNodeId.check;
        CLI01.RD_1 TO STRING2STRING_2.IN;
        STRING2STRING_2.OUT TO CLI10.SD_1;
        STRING2STRING_2_1.OUT TO SER1.SD_1;
        SER1.RD_1 TO STRING2STRING_2_1.IN;
        SER01.QO TO F_NOT_1_1_1_2_1.IN;
        SER01.RD_1 TO STRING2STRING_3.IN;
        ID TO SUB1.ID;
        ID TO PUB1.ID;
        ID TO SER0.ID;
        ID TO CLI0.ID;
        ID TO CLI1.ID;
        ID TO CLI01.ID;
        ID TO CLI10.ID;
        ID TO SER01.ID;
        ID TO SER1.ID;
        F_NOT_1_1_1_2_1_1.OUT TO Server1_0wrongNodeId.check;
        ID TO SER10.ID;
        SER10.QO TO F_NOT_1_1_1_2_1_1.IN;
        STRING2STRING_3.OUT TO SER10.SD_1;
      END_CONNECTIONS
    END_SUBAPPLICATION
    SUBAPPLICATION UnknownIdentifier
      EVENT_INPUT
        REQ;
      END_EVENT
      EVENT_OUTPUT
        CNF;
      END_EVENT
      VAR_INPUT
        ID : WSTRING;
      END_VAR
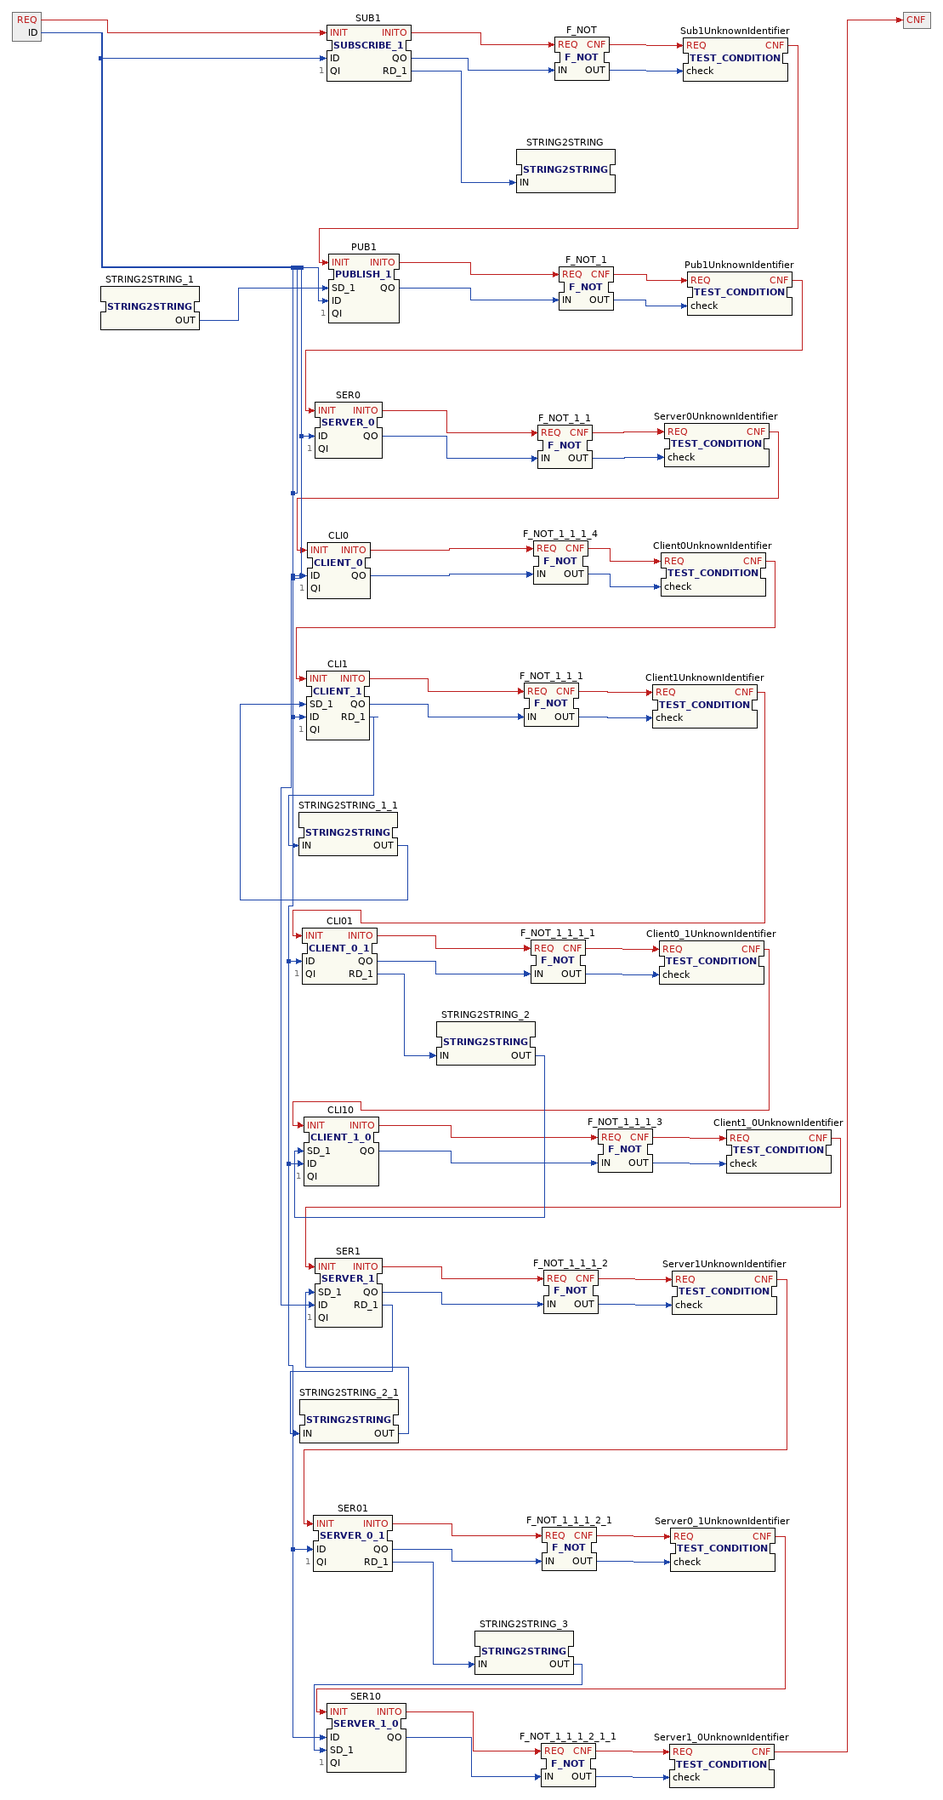
      FBS
        F_NOT_1_1_1 : F_NOT;
        Client1UnknownIdentifier : TEST_CONDITION;
        Pub1UnknownIdentifier : TEST_CONDITION;
        F_NOT_1_1 : F_NOT;
        PUB1 : PUBLISH_1(QI := 1);
        F_NOT : F_NOT;
        Server0UnknownIdentifier : TEST_CONDITION;
        Sub1UnknownIdentifier : TEST_CONDITION;
        F_NOT_1 : F_NOT;
        STRING2STRING : STRING2STRING;
        SUB1 : SUBSCRIBE_1(QI := 1);
        SER0 : SERVER_0(QI := 1);
        STRING2STRING_1 : STRING2STRING;
        Client0_1UnknownIdentifier : TEST_CONDITION;
        F_NOT_1_1_1_1 : F_NOT;
        Server1UnknownIdentifier : TEST_CONDITION;
        F_NOT_1_1_1_2 : F_NOT;
        CLI1 : CLIENT_1(QI := 1);
        CLI01 : CLIENT_0_1(QI := 1);
        Client1_0UnknownIdentifier : TEST_CONDITION;
        F_NOT_1_1_1_3 : F_NOT;
        CLI10 : CLIENT_1_0(QI := 1);
        STRING2STRING_1_1 : STRING2STRING;
        F_NOT_1_1_1_4 : F_NOT;
        Client0UnknownIdentifier : TEST_CONDITION;
        CLI0 : CLIENT_0(QI := 1);
        SER1 : SERVER_1(QI := 1);
        F_NOT_1_1_1_2_1 : F_NOT;
        Server0_1UnknownIdentifier : TEST_CONDITION;
        STRING2STRING_2 : STRING2STRING;
        STRING2STRING_2_1 : STRING2STRING;
        SER01 : SERVER_0_1(QI := 1);
        STRING2STRING_3 : STRING2STRING;
        Server1_0UnknownIdentifier : TEST_CONDITION;
        F_NOT_1_1_1_2_1_1 : F_NOT;
        SER10 : SERVER_1_0(QI := 1);
      END_FBS
      EVENT_CONNECTIONS
        F_NOT_1_1_1.CNF TO Client1UnknownIdentifier.REQ;
        F_NOT_1.CNF TO Pub1UnknownIdentifier.REQ;
        Pub1UnknownIdentifier.CNF TO SER0.INIT;
        SER0.INITO TO F_NOT_1_1.REQ;
        F_NOT_1_1.CNF TO Server0UnknownIdentifier.REQ;
        Sub1UnknownIdentifier.CNF TO PUB1.INIT;
        PUB1.INITO TO F_NOT_1.REQ;
        SUB1.INITO TO F_NOT.REQ;
        F_NOT.CNF TO Sub1UnknownIdentifier.REQ;
        REQ TO SUB1.INIT;
        F_NOT_1_1_1_1.CNF TO Client0_1UnknownIdentifier.REQ;
        F_NOT_1_1_1_2.CNF TO Server1UnknownIdentifier.REQ;
        CLI1.INITO TO F_NOT_1_1_1.REQ;
        CLI01.INITO TO F_NOT_1_1_1_1.REQ;
        CLI0.INITO TO F_NOT_1_1_1_4.REQ;
        F_NOT_1_1_1_4.CNF TO Client0UnknownIdentifier.REQ;
        F_NOT_1_1_1_3.CNF TO Client1_0UnknownIdentifier.REQ;
        CLI10.INITO TO F_NOT_1_1_1_3.REQ;
        SER1.INITO TO F_NOT_1_1_1_2.REQ;
        F_NOT_1_1_1_2_1.CNF TO Server0_1UnknownIdentifier.REQ;
        SER01.INITO TO F_NOT_1_1_1_2_1.REQ;
        Server0UnknownIdentifier.CNF TO CLI0.INIT;
        Client0UnknownIdentifier.CNF TO CLI1.INIT;
        Client1UnknownIdentifier.CNF TO CLI01.INIT;
        Client0_1UnknownIdentifier.CNF TO CLI10.INIT;
        Client1_0UnknownIdentifier.CNF TO SER1.INIT;
        Server1UnknownIdentifier.CNF TO SER01.INIT;
        F_NOT_1_1_1_2_1_1.CNF TO Server1_0UnknownIdentifier.REQ;
        Server1_0UnknownIdentifier.CNF TO CNF;
        Server0_1UnknownIdentifier.CNF TO SER10.INIT;
        SER10.INITO TO F_NOT_1_1_1_2_1_1.REQ;
      END_CONNECTIONS
      DATA_CONNECTIONS
        F_NOT_1_1_1.OUT TO Client1UnknownIdentifier.check;
        F_NOT_1.OUT TO Pub1UnknownIdentifier.check;
        SER0.QO TO F_NOT_1_1.IN;
        F_NOT_1_1.OUT TO Server0UnknownIdentifier.check;
        STRING2STRING_1.OUT TO PUB1.SD_1;
        PUB1.QO TO F_NOT_1.IN;
        SUB1.QO TO F_NOT.IN;
        F_NOT.OUT TO Sub1UnknownIdentifier.check;
        SUB1.RD_1 TO STRING2STRING.IN;
        F_NOT_1_1_1_1.OUT TO Client0_1UnknownIdentifier.check;
        F_NOT_1_1_1_2.OUT TO Server1UnknownIdentifier.check;
        CLI1.QO TO F_NOT_1_1_1.IN;
        CLI01.QO TO F_NOT_1_1_1_1.IN;
        STRING2STRING_1_1.OUT TO CLI1.SD_1;
        CLI1.RD_1 TO STRING2STRING_1_1.IN;
        F_NOT_1_1_1_4.OUT TO Client0UnknownIdentifier.check;
        CLI0.QO TO F_NOT_1_1_1_4.IN;
        F_NOT_1_1_1_3.OUT TO Client1_0UnknownIdentifier.check;
        CLI10.QO TO F_NOT_1_1_1_3.IN;
        SER1.QO TO F_NOT_1_1_1_2.IN;
        F_NOT_1_1_1_2_1.OUT TO Server0_1UnknownIdentifier.check;
        CLI01.RD_1 TO STRING2STRING_2.IN;
        STRING2STRING_2.OUT TO CLI10.SD_1;
        STRING2STRING_2_1.OUT TO SER1.SD_1;
        SER1.RD_1 TO STRING2STRING_2_1.IN;
        SER01.QO TO F_NOT_1_1_1_2_1.IN;
        SER01.RD_1 TO STRING2STRING_3.IN;
        ID TO SUB1.ID;
        ID TO PUB1.ID;
        ID TO SER0.ID;
        ID TO CLI0.ID;
        ID TO CLI1.ID;
        ID TO CLI01.ID;
        ID TO CLI10.ID;
        ID TO SER01.ID;
        ID TO SER1.ID;
        F_NOT_1_1_1_2_1_1.OUT TO Server1_0UnknownIdentifier.check;
        ID TO SER10.ID;
        SER10.QO TO F_NOT_1_1_1_2_1_1.IN;
        STRING2STRING_3.OUT TO SER10.SD_1;
      END_CONNECTIONS
    END_SUBAPPLICATION
    SUBAPPLICATION WrongIdentifier
      EVENT_INPUT
        REQ;
      END_EVENT
      EVENT_OUTPUT
        CNF;
      END_EVENT
      VAR_INPUT
        ID : WSTRING;
      END_VAR
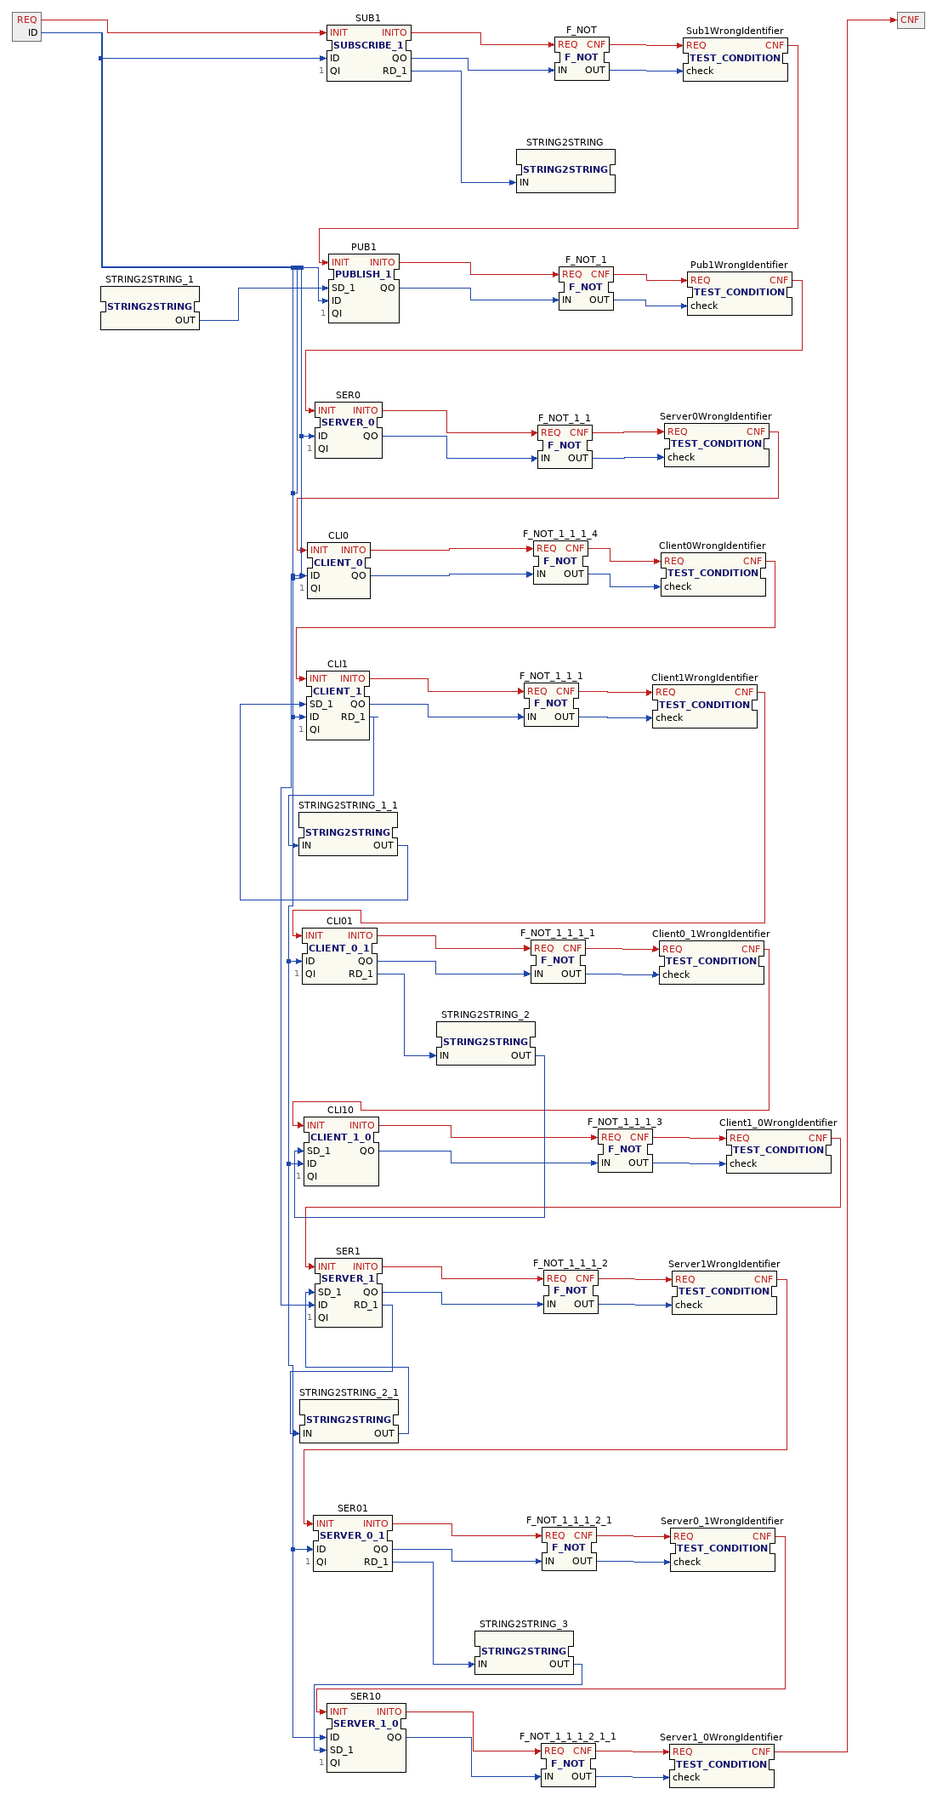
      FBS
        F_NOT_1_1_1 : F_NOT;
        Client1WrongIdentifier : TEST_CONDITION;
        Pub1WrongIdentifier : TEST_CONDITION;
        F_NOT_1_1 : F_NOT;
        PUB1 : PUBLISH_1(QI := 1);
        F_NOT : F_NOT;
        Server0WrongIdentifier : TEST_CONDITION;
        Sub1WrongIdentifier : TEST_CONDITION;
        F_NOT_1 : F_NOT;
        STRING2STRING : STRING2STRING;
        SUB1 : SUBSCRIBE_1(QI := 1);
        SER0 : SERVER_0(QI := 1);
        STRING2STRING_1 : STRING2STRING;
        Client0_1WrongIdentifier : TEST_CONDITION;
        F_NOT_1_1_1_1 : F_NOT;
        Server1WrongIdentifier : TEST_CONDITION;
        F_NOT_1_1_1_2 : F_NOT;
        CLI1 : CLIENT_1(QI := 1);
        CLI01 : CLIENT_0_1(QI := 1);
        Client1_0WrongIdentifier : TEST_CONDITION;
        F_NOT_1_1_1_3 : F_NOT;
        CLI10 : CLIENT_1_0(QI := 1);
        STRING2STRING_1_1 : STRING2STRING;
        F_NOT_1_1_1_4 : F_NOT;
        Client0WrongIdentifier : TEST_CONDITION;
        CLI0 : CLIENT_0(QI := 1);
        SER1 : SERVER_1(QI := 1);
        F_NOT_1_1_1_2_1 : F_NOT;
        Server0_1WrongIdentifier : TEST_CONDITION;
        STRING2STRING_2 : STRING2STRING;
        STRING2STRING_2_1 : STRING2STRING;
        SER01 : SERVER_0_1(QI := 1);
        STRING2STRING_3 : STRING2STRING;
        Server1_0WrongIdentifier : TEST_CONDITION;
        F_NOT_1_1_1_2_1_1 : F_NOT;
        SER10 : SERVER_1_0(QI := 1);
      END_FBS
      EVENT_CONNECTIONS
        F_NOT_1_1_1.CNF TO Client1WrongIdentifier.REQ;
        F_NOT_1.CNF TO Pub1WrongIdentifier.REQ;
        Pub1WrongIdentifier.CNF TO SER0.INIT;
        SER0.INITO TO F_NOT_1_1.REQ;
        F_NOT_1_1.CNF TO Server0WrongIdentifier.REQ;
        Sub1WrongIdentifier.CNF TO PUB1.INIT;
        PUB1.INITO TO F_NOT_1.REQ;
        SUB1.INITO TO F_NOT.REQ;
        F_NOT.CNF TO Sub1WrongIdentifier.REQ;
        REQ TO SUB1.INIT;
        F_NOT_1_1_1_1.CNF TO Client0_1WrongIdentifier.REQ;
        F_NOT_1_1_1_2.CNF TO Server1WrongIdentifier.REQ;
        CLI1.INITO TO F_NOT_1_1_1.REQ;
        CLI01.INITO TO F_NOT_1_1_1_1.REQ;
        CLI0.INITO TO F_NOT_1_1_1_4.REQ;
        F_NOT_1_1_1_4.CNF TO Client0WrongIdentifier.REQ;
        F_NOT_1_1_1_3.CNF TO Client1_0WrongIdentifier.REQ;
        CLI10.INITO TO F_NOT_1_1_1_3.REQ;
        SER1.INITO TO F_NOT_1_1_1_2.REQ;
        F_NOT_1_1_1_2_1.CNF TO Server0_1WrongIdentifier.REQ;
        SER01.INITO TO F_NOT_1_1_1_2_1.REQ;
        Server0WrongIdentifier.CNF TO CLI0.INIT;
        Client0WrongIdentifier.CNF TO CLI1.INIT;
        Client1WrongIdentifier.CNF TO CLI01.INIT;
        Client0_1WrongIdentifier.CNF TO CLI10.INIT;
        Client1_0WrongIdentifier.CNF TO SER1.INIT;
        Server1WrongIdentifier.CNF TO SER01.INIT;
        F_NOT_1_1_1_2_1_1.CNF TO Server1_0WrongIdentifier.REQ;
        Server1_0WrongIdentifier.CNF TO CNF;
        Server0_1WrongIdentifier.CNF TO SER10.INIT;
        SER10.INITO TO F_NOT_1_1_1_2_1_1.REQ;
      END_CONNECTIONS
      DATA_CONNECTIONS
        F_NOT_1_1_1.OUT TO Client1WrongIdentifier.check;
        F_NOT_1.OUT TO Pub1WrongIdentifier.check;
        SER0.QO TO F_NOT_1_1.IN;
        F_NOT_1_1.OUT TO Server0WrongIdentifier.check;
        STRING2STRING_1.OUT TO PUB1.SD_1;
        PUB1.QO TO F_NOT_1.IN;
        SUB1.QO TO F_NOT.IN;
        F_NOT.OUT TO Sub1WrongIdentifier.check;
        SUB1.RD_1 TO STRING2STRING.IN;
        F_NOT_1_1_1_1.OUT TO Client0_1WrongIdentifier.check;
        F_NOT_1_1_1_2.OUT TO Server1WrongIdentifier.check;
        CLI1.QO TO F_NOT_1_1_1.IN;
        CLI01.QO TO F_NOT_1_1_1_1.IN;
        STRING2STRING_1_1.OUT TO CLI1.SD_1;
        CLI1.RD_1 TO STRING2STRING_1_1.IN;
        F_NOT_1_1_1_4.OUT TO Client0WrongIdentifier.check;
        CLI0.QO TO F_NOT_1_1_1_4.IN;
        F_NOT_1_1_1_3.OUT TO Client1_0WrongIdentifier.check;
        CLI10.QO TO F_NOT_1_1_1_3.IN;
        SER1.QO TO F_NOT_1_1_1_2.IN;
        F_NOT_1_1_1_2_1.OUT TO Server0_1WrongIdentifier.check;
        CLI01.RD_1 TO STRING2STRING_2.IN;
        STRING2STRING_2.OUT TO CLI10.SD_1;
        STRING2STRING_2_1.OUT TO SER1.SD_1;
        SER1.RD_1 TO STRING2STRING_2_1.IN;
        SER01.QO TO F_NOT_1_1_1_2_1.IN;
        SER01.RD_1 TO STRING2STRING_3.IN;
        ID TO SUB1.ID;
        ID TO PUB1.ID;
        ID TO SER0.ID;
        ID TO CLI0.ID;
        ID TO CLI1.ID;
        ID TO CLI01.ID;
        ID TO CLI10.ID;
        ID TO SER01.ID;
        ID TO SER1.ID;
        F_NOT_1_1_1_2_1_1.OUT TO Server1_0WrongIdentifier.check;
        ID TO SER10.ID;
        SER10.QO TO F_NOT_1_1_1_2_1_1.IN;
        STRING2STRING_3.OUT TO SER10.SD_1;
      END_CONNECTIONS
    END_SUBAPPLICATION
    SUBAPPLICATION LocalWithoutBrowseName
      EVENT_INPUT
        REQ;
      END_EVENT
      EVENT_OUTPUT
        CNF;
      END_EVENT
      VAR_INPUT
        ID : WSTRING;
      END_VAR
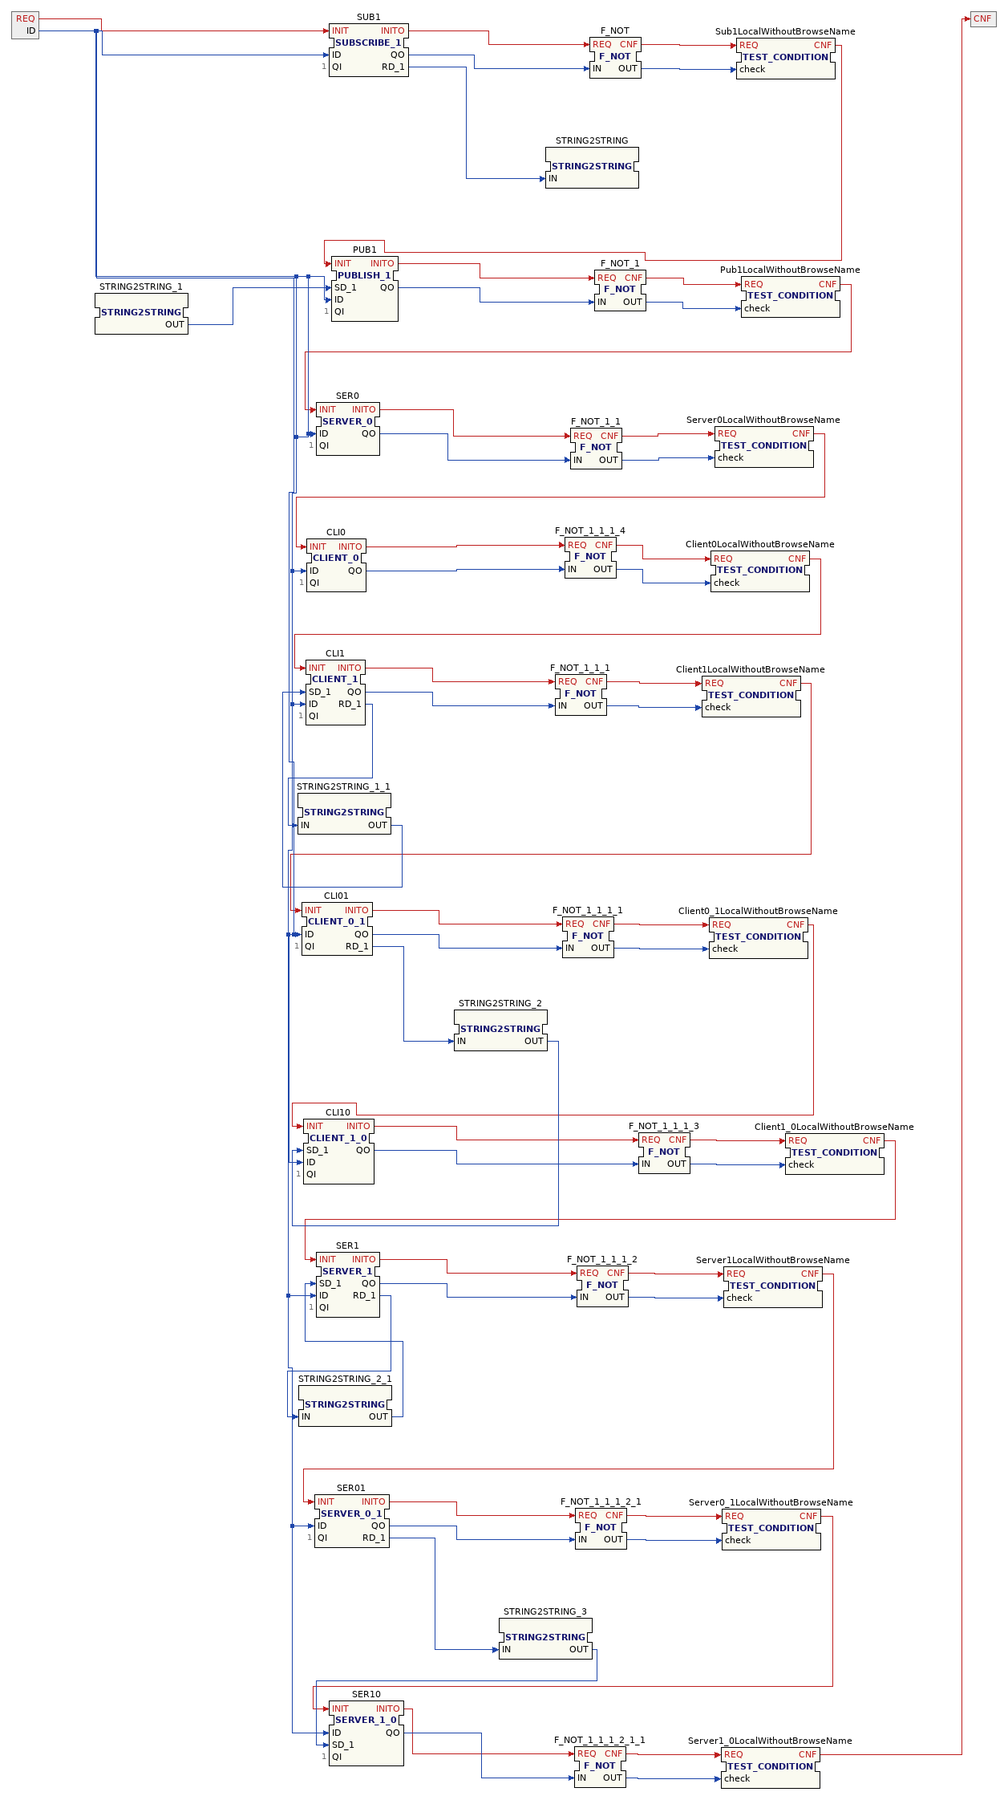
      FBS
        F_NOT_1_1_1 : F_NOT;
        Client1LocalWithoutBrowseName : TEST_CONDITION;
        Pub1LocalWithoutBrowseName : TEST_CONDITION;
        F_NOT_1_1 : F_NOT;
        PUB1 : PUBLISH_1(QI := 1);
        F_NOT : F_NOT;
        Server0LocalWithoutBrowseName : TEST_CONDITION;
        Sub1LocalWithoutBrowseName : TEST_CONDITION;
        F_NOT_1 : F_NOT;
        STRING2STRING : STRING2STRING;
        SUB1 : SUBSCRIBE_1(QI := 1);
        SER0 : SERVER_0(QI := 1);
        STRING2STRING_1 : STRING2STRING;
        Client0_1LocalWithoutBrowseName : TEST_CONDITION;
        F_NOT_1_1_1_1 : F_NOT;
        Server1LocalWithoutBrowseName : TEST_CONDITION;
        F_NOT_1_1_1_2 : F_NOT;
        CLI1 : CLIENT_1(QI := 1);
        CLI01 : CLIENT_0_1(QI := 1);
        Client1_0LocalWithoutBrowseName : TEST_CONDITION;
        F_NOT_1_1_1_3 : F_NOT;
        CLI10 : CLIENT_1_0(QI := 1);
        STRING2STRING_1_1 : STRING2STRING;
        F_NOT_1_1_1_4 : F_NOT;
        Client0LocalWithoutBrowseName : TEST_CONDITION;
        CLI0 : CLIENT_0(QI := 1);
        SER1 : SERVER_1(QI := 1);
        F_NOT_1_1_1_2_1 : F_NOT;
        Server0_1LocalWithoutBrowseName : TEST_CONDITION;
        STRING2STRING_2 : STRING2STRING;
        STRING2STRING_2_1 : STRING2STRING;
        SER01 : SERVER_0_1(QI := 1);
        STRING2STRING_3 : STRING2STRING;
        Server1_0LocalWithoutBrowseName : TEST_CONDITION;
        F_NOT_1_1_1_2_1_1 : F_NOT;
        SER10 : SERVER_1_0(QI := 1);
      END_FBS
      EVENT_CONNECTIONS
        F_NOT_1_1_1.CNF TO Client1LocalWithoutBrowseName.REQ;
        F_NOT_1.CNF TO Pub1LocalWithoutBrowseName.REQ;
        Pub1LocalWithoutBrowseName.CNF TO SER0.INIT;
        SER0.INITO TO F_NOT_1_1.REQ;
        F_NOT_1_1.CNF TO Server0LocalWithoutBrowseName.REQ;
        Sub1LocalWithoutBrowseName.CNF TO PUB1.INIT;
        PUB1.INITO TO F_NOT_1.REQ;
        SUB1.INITO TO F_NOT.REQ;
        F_NOT.CNF TO Sub1LocalWithoutBrowseName.REQ;
        REQ TO SUB1.INIT;
        F_NOT_1_1_1_1.CNF TO Client0_1LocalWithoutBrowseName.REQ;
        F_NOT_1_1_1_2.CNF TO Server1LocalWithoutBrowseName.REQ;
        CLI1.INITO TO F_NOT_1_1_1.REQ;
        CLI01.INITO TO F_NOT_1_1_1_1.REQ;
        CLI0.INITO TO F_NOT_1_1_1_4.REQ;
        F_NOT_1_1_1_4.CNF TO Client0LocalWithoutBrowseName.REQ;
        F_NOT_1_1_1_3.CNF TO Client1_0LocalWithoutBrowseName.REQ;
        CLI10.INITO TO F_NOT_1_1_1_3.REQ;
        SER1.INITO TO F_NOT_1_1_1_2.REQ;
        F_NOT_1_1_1_2_1.CNF TO Server0_1LocalWithoutBrowseName.REQ;
        SER01.INITO TO F_NOT_1_1_1_2_1.REQ;
        Server0LocalWithoutBrowseName.CNF TO CLI0.INIT;
        Client0LocalWithoutBrowseName.CNF TO CLI1.INIT;
        Client1LocalWithoutBrowseName.CNF TO CLI01.INIT;
        Client0_1LocalWithoutBrowseName.CNF TO CLI10.INIT;
        Client1_0LocalWithoutBrowseName.CNF TO SER1.INIT;
        Server1LocalWithoutBrowseName.CNF TO SER01.INIT;
        F_NOT_1_1_1_2_1_1.CNF TO Server1_0LocalWithoutBrowseName.REQ;
        Server1_0LocalWithoutBrowseName.CNF TO CNF;
        Server0_1LocalWithoutBrowseName.CNF TO SER10.INIT;
        SER10.INITO TO F_NOT_1_1_1_2_1_1.REQ;
      END_CONNECTIONS
      DATA_CONNECTIONS
        F_NOT_1_1_1.OUT TO Client1LocalWithoutBrowseName.check;
        F_NOT_1.OUT TO Pub1LocalWithoutBrowseName.check;
        SER0.QO TO F_NOT_1_1.IN;
        F_NOT_1_1.OUT TO Server0LocalWithoutBrowseName.check;
        STRING2STRING_1.OUT TO PUB1.SD_1;
        PUB1.QO TO F_NOT_1.IN;
        SUB1.QO TO F_NOT.IN;
        F_NOT.OUT TO Sub1LocalWithoutBrowseName.check;
        SUB1.RD_1 TO STRING2STRING.IN;
        F_NOT_1_1_1_1.OUT TO Client0_1LocalWithoutBrowseName.check;
        F_NOT_1_1_1_2.OUT TO Server1LocalWithoutBrowseName.check;
        CLI1.QO TO F_NOT_1_1_1.IN;
        CLI01.QO TO F_NOT_1_1_1_1.IN;
        STRING2STRING_1_1.OUT TO CLI1.SD_1;
        CLI1.RD_1 TO STRING2STRING_1_1.IN;
        F_NOT_1_1_1_4.OUT TO Client0LocalWithoutBrowseName.check;
        CLI0.QO TO F_NOT_1_1_1_4.IN;
        F_NOT_1_1_1_3.OUT TO Client1_0LocalWithoutBrowseName.check;
        CLI10.QO TO F_NOT_1_1_1_3.IN;
        SER1.QO TO F_NOT_1_1_1_2.IN;
        F_NOT_1_1_1_2_1.OUT TO Server0_1LocalWithoutBrowseName.check;
        CLI01.RD_1 TO STRING2STRING_2.IN;
        STRING2STRING_2.OUT TO CLI10.SD_1;
        STRING2STRING_2_1.OUT TO SER1.SD_1;
        SER1.RD_1 TO STRING2STRING_2_1.IN;
        SER01.QO TO F_NOT_1_1_1_2_1.IN;
        SER01.RD_1 TO STRING2STRING_3.IN;
        ID TO SUB1.ID;
        ID TO PUB1.ID;
        ID TO SER0.ID;
        ID TO CLI0.ID;
        ID TO CLI1.ID;
        ID TO CLI01.ID;
        ID TO CLI10.ID;
        ID TO SER01.ID;
        ID TO SER1.ID;
        F_NOT_1_1_1_2_1_1.OUT TO Server1_0LocalWithoutBrowseName.check;
        ID TO SER10.ID;
        SER10.QO TO F_NOT_1_1_1_2_1_1.IN;
        STRING2STRING_3.OUT TO SER10.SD_1;
      END_CONNECTIONS
    END_SUBAPPLICATION
    SUBAPPLICATION RemoteWithoutBrowseNameNorNodeId
      EVENT_INPUT
        REQ;
      END_EVENT
      EVENT_OUTPUT
        CNF;
      END_EVENT
      VAR_INPUT
        ID : WSTRING;
      END_VAR
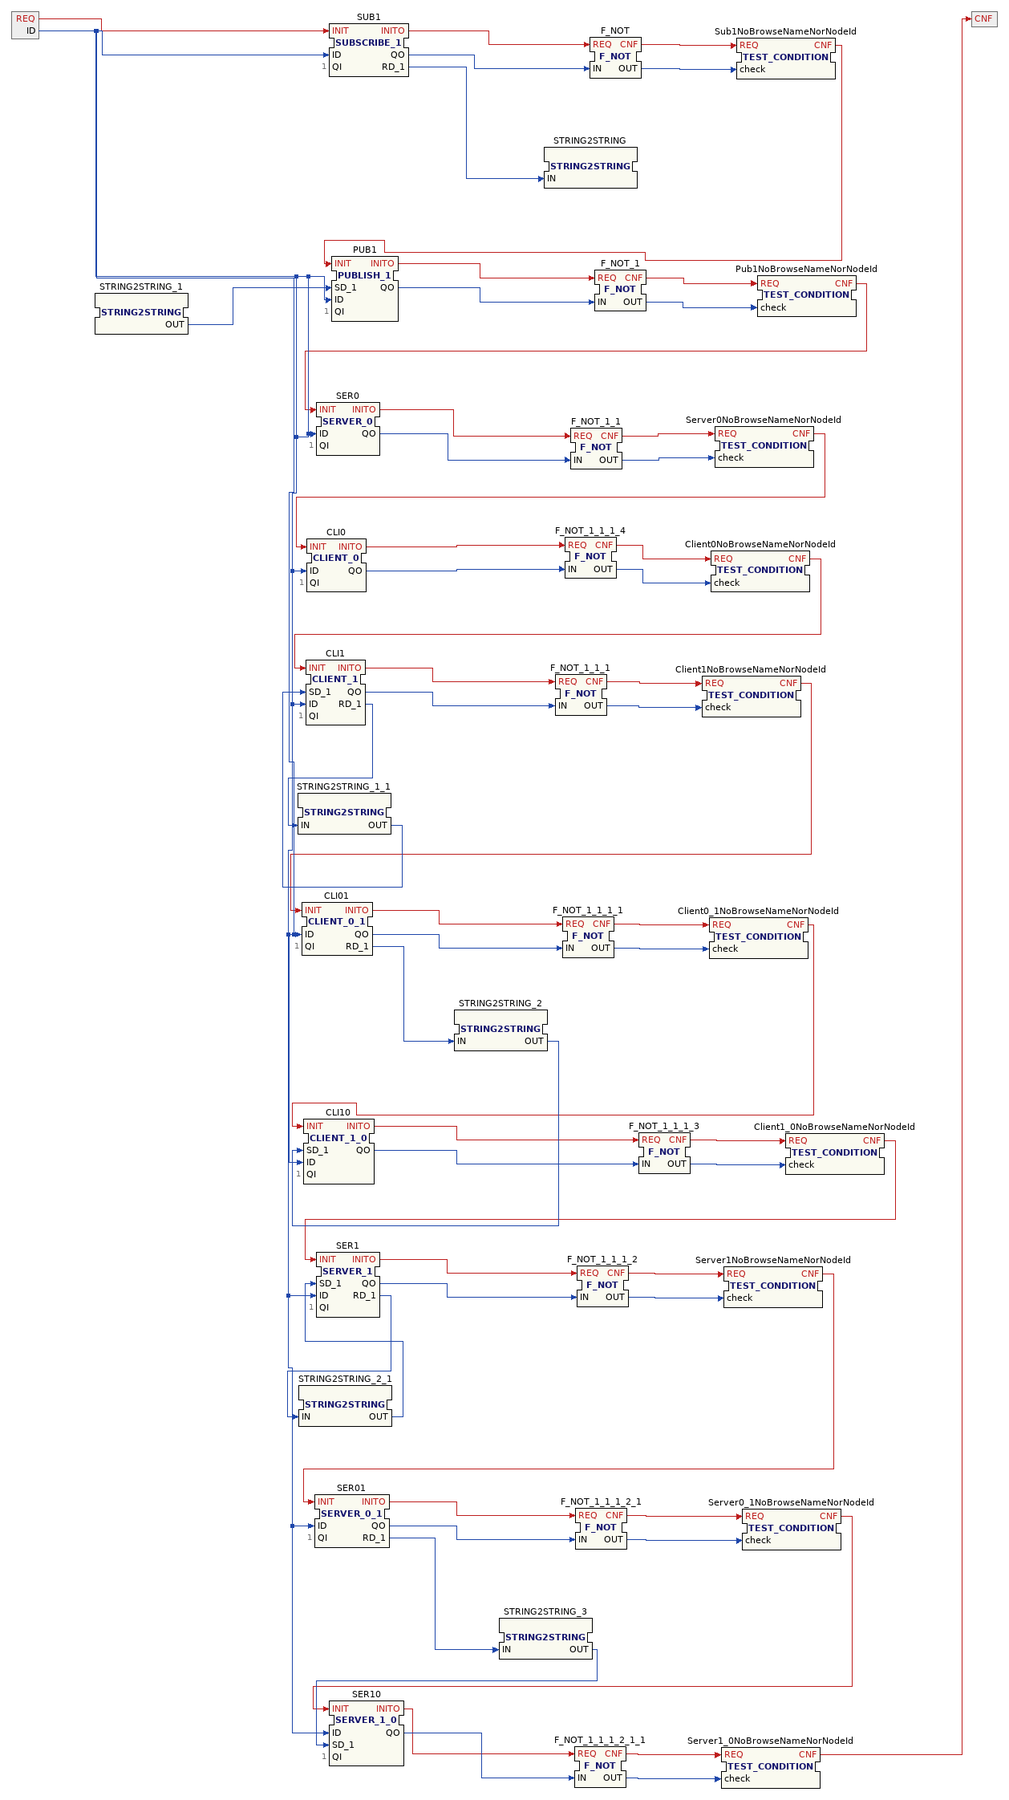
      FBS
        F_NOT_1_1_1 : F_NOT;
        Client1NoBrowseNameNorNodeId : TEST_CONDITION;
        Pub1NoBrowseNameNorNodeId : TEST_CONDITION;
        F_NOT_1_1 : F_NOT;
        PUB1 : PUBLISH_1(QI := 1);
        F_NOT : F_NOT;
        Server0NoBrowseNameNorNodeId : TEST_CONDITION;
        Sub1NoBrowseNameNorNodeId : TEST_CONDITION;
        F_NOT_1 : F_NOT;
        STRING2STRING : STRING2STRING;
        SUB1 : SUBSCRIBE_1(QI := 1);
        SER0 : SERVER_0(QI := 1);
        STRING2STRING_1 : STRING2STRING;
        Client0_1NoBrowseNameNorNodeId : TEST_CONDITION;
        F_NOT_1_1_1_1 : F_NOT;
        Server1NoBrowseNameNorNodeId : TEST_CONDITION;
        F_NOT_1_1_1_2 : F_NOT;
        CLI1 : CLIENT_1(QI := 1);
        CLI01 : CLIENT_0_1(QI := 1);
        Client1_0NoBrowseNameNorNodeId : TEST_CONDITION;
        F_NOT_1_1_1_3 : F_NOT;
        CLI10 : CLIENT_1_0(QI := 1);
        STRING2STRING_1_1 : STRING2STRING;
        F_NOT_1_1_1_4 : F_NOT;
        Client0NoBrowseNameNorNodeId : TEST_CONDITION;
        CLI0 : CLIENT_0(QI := 1);
        SER1 : SERVER_1(QI := 1);
        F_NOT_1_1_1_2_1 : F_NOT;
        Server0_1NoBrowseNameNorNodeId : TEST_CONDITION;
        STRING2STRING_2 : STRING2STRING;
        STRING2STRING_2_1 : STRING2STRING;
        SER01 : SERVER_0_1(QI := 1);
        STRING2STRING_3 : STRING2STRING;
        Server1_0NoBrowseNameNorNodeId : TEST_CONDITION;
        F_NOT_1_1_1_2_1_1 : F_NOT;
        SER10 : SERVER_1_0(QI := 1);
      END_FBS
      EVENT_CONNECTIONS
        F_NOT_1_1_1.CNF TO Client1NoBrowseNameNorNodeId.REQ;
        F_NOT_1.CNF TO Pub1NoBrowseNameNorNodeId.REQ;
        Pub1NoBrowseNameNorNodeId.CNF TO SER0.INIT;
        SER0.INITO TO F_NOT_1_1.REQ;
        F_NOT_1_1.CNF TO Server0NoBrowseNameNorNodeId.REQ;
        Sub1NoBrowseNameNorNodeId.CNF TO PUB1.INIT;
        PUB1.INITO TO F_NOT_1.REQ;
        SUB1.INITO TO F_NOT.REQ;
        F_NOT.CNF TO Sub1NoBrowseNameNorNodeId.REQ;
        REQ TO SUB1.INIT;
        F_NOT_1_1_1_1.CNF TO Client0_1NoBrowseNameNorNodeId.REQ;
        F_NOT_1_1_1_2.CNF TO Server1NoBrowseNameNorNodeId.REQ;
        CLI1.INITO TO F_NOT_1_1_1.REQ;
        CLI01.INITO TO F_NOT_1_1_1_1.REQ;
        CLI0.INITO TO F_NOT_1_1_1_4.REQ;
        F_NOT_1_1_1_4.CNF TO Client0NoBrowseNameNorNodeId.REQ;
        F_NOT_1_1_1_3.CNF TO Client1_0NoBrowseNameNorNodeId.REQ;
        CLI10.INITO TO F_NOT_1_1_1_3.REQ;
        SER1.INITO TO F_NOT_1_1_1_2.REQ;
        F_NOT_1_1_1_2_1.CNF TO Server0_1NoBrowseNameNorNodeId.REQ;
        SER01.INITO TO F_NOT_1_1_1_2_1.REQ;
        Server0NoBrowseNameNorNodeId.CNF TO CLI0.INIT;
        Client0NoBrowseNameNorNodeId.CNF TO CLI1.INIT;
        Client1NoBrowseNameNorNodeId.CNF TO CLI01.INIT;
        Client0_1NoBrowseNameNorNodeId.CNF TO CLI10.INIT;
        Client1_0NoBrowseNameNorNodeId.CNF TO SER1.INIT;
        Server1NoBrowseNameNorNodeId.CNF TO SER01.INIT;
        F_NOT_1_1_1_2_1_1.CNF TO Server1_0NoBrowseNameNorNodeId.REQ;
        Server1_0NoBrowseNameNorNodeId.CNF TO CNF;
        Server0_1NoBrowseNameNorNodeId.CNF TO SER10.INIT;
        SER10.INITO TO F_NOT_1_1_1_2_1_1.REQ;
      END_CONNECTIONS
      DATA_CONNECTIONS
        F_NOT_1_1_1.OUT TO Client1NoBrowseNameNorNodeId.check;
        F_NOT_1.OUT TO Pub1NoBrowseNameNorNodeId.check;
        SER0.QO TO F_NOT_1_1.IN;
        F_NOT_1_1.OUT TO Server0NoBrowseNameNorNodeId.check;
        STRING2STRING_1.OUT TO PUB1.SD_1;
        PUB1.QO TO F_NOT_1.IN;
        SUB1.QO TO F_NOT.IN;
        F_NOT.OUT TO Sub1NoBrowseNameNorNodeId.check;
        SUB1.RD_1 TO STRING2STRING.IN;
        F_NOT_1_1_1_1.OUT TO Client0_1NoBrowseNameNorNodeId.check;
        F_NOT_1_1_1_2.OUT TO Server1NoBrowseNameNorNodeId.check;
        CLI1.QO TO F_NOT_1_1_1.IN;
        CLI01.QO TO F_NOT_1_1_1_1.IN;
        STRING2STRING_1_1.OUT TO CLI1.SD_1;
        CLI1.RD_1 TO STRING2STRING_1_1.IN;
        F_NOT_1_1_1_4.OUT TO Client0NoBrowseNameNorNodeId.check;
        CLI0.QO TO F_NOT_1_1_1_4.IN;
        F_NOT_1_1_1_3.OUT TO Client1_0NoBrowseNameNorNodeId.check;
        CLI10.QO TO F_NOT_1_1_1_3.IN;
        SER1.QO TO F_NOT_1_1_1_2.IN;
        F_NOT_1_1_1_2_1.OUT TO Server0_1NoBrowseNameNorNodeId.check;
        CLI01.RD_1 TO STRING2STRING_2.IN;
        STRING2STRING_2.OUT TO CLI10.SD_1;
        STRING2STRING_2_1.OUT TO SER1.SD_1;
        SER1.RD_1 TO STRING2STRING_2_1.IN;
        SER01.QO TO F_NOT_1_1_1_2_1.IN;
        SER01.RD_1 TO STRING2STRING_3.IN;
        ID TO SUB1.ID;
        ID TO PUB1.ID;
        ID TO SER0.ID;
        ID TO CLI0.ID;
        ID TO CLI1.ID;
        ID TO CLI01.ID;
        ID TO CLI10.ID;
        ID TO SER01.ID;
        ID TO SER1.ID;
        F_NOT_1_1_1_2_1_1.OUT TO Server1_0NoBrowseNameNorNodeId.check;
        ID TO SER10.ID;
        SER10.QO TO F_NOT_1_1_1_2_1_1.IN;
        STRING2STRING_3.OUT TO SER10.SD_1;
      END_CONNECTIONS
    END_SUBAPPLICATION
    SUBAPPLICATION LocalRead
      EVENT_INPUT
        REQ;
      END_EVENT
      EVENT_OUTPUT
        CNF;
      END_EVENT
      VAR_INPUT
        ID : WSTRING;
      END_VAR
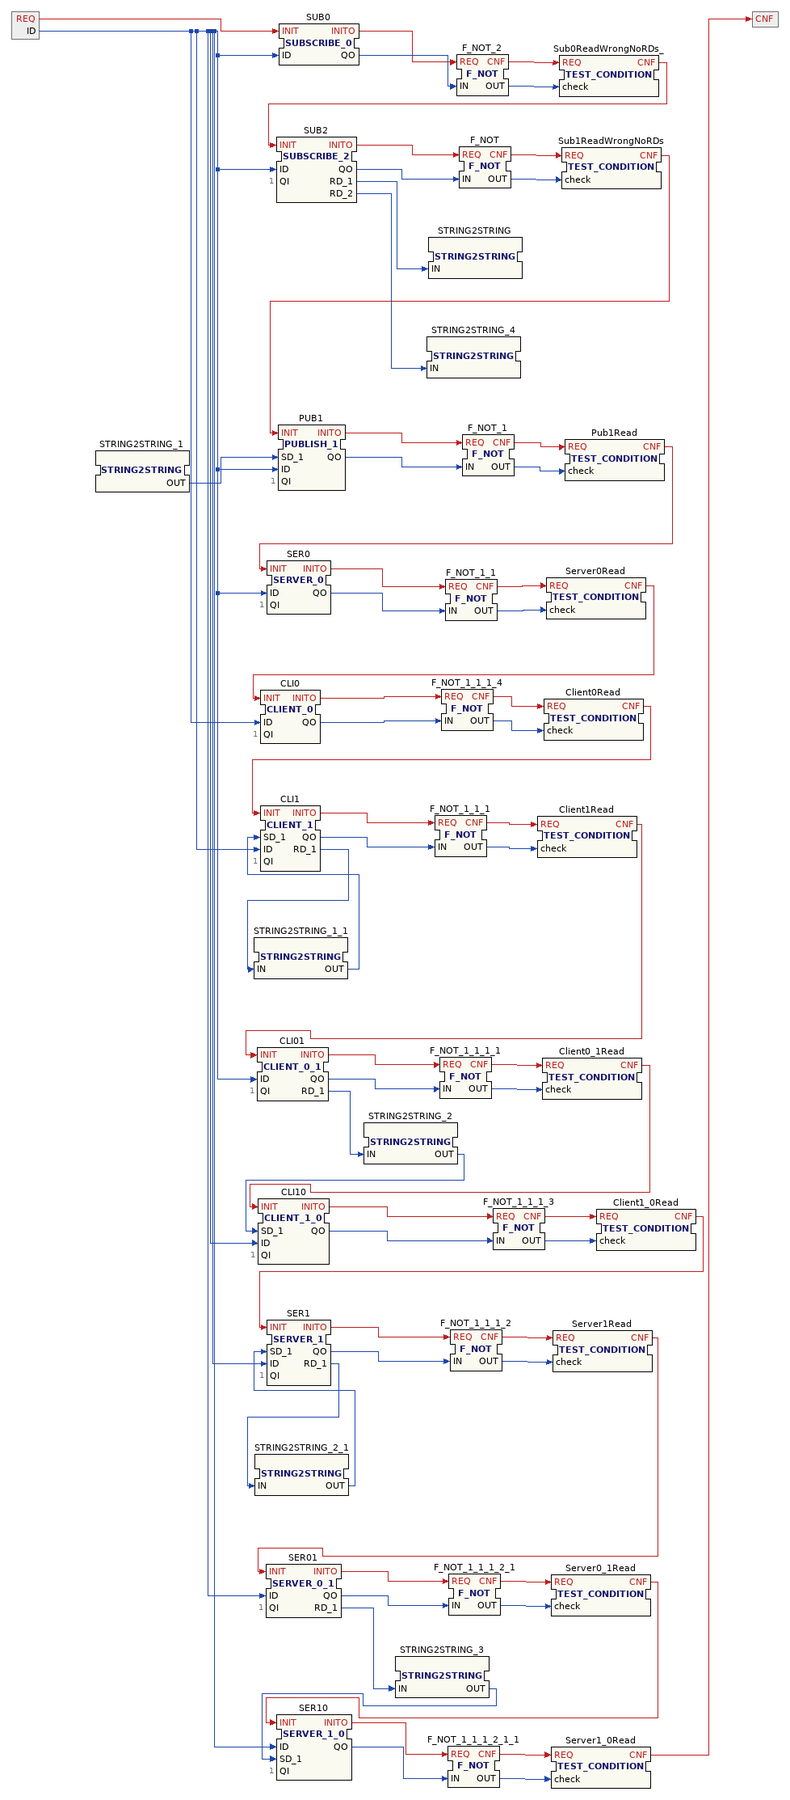
      FBS
        F_NOT_1_1_1 : F_NOT;
        Client1Read : TEST_CONDITION;
        Pub1Read : TEST_CONDITION;
        F_NOT_1_1 : F_NOT;
        PUB1 : PUBLISH_1(QI := 1);
        F_NOT : F_NOT;
        Server0Read : TEST_CONDITION;
        Sub1ReadWrongNoRDs : TEST_CONDITION;
        F_NOT_1 : F_NOT;
        STRING2STRING : STRING2STRING;
        SER0 : SERVER_0(QI := 1);
        STRING2STRING_1 : STRING2STRING;
        Client0_1Read : TEST_CONDITION;
        F_NOT_1_1_1_1 : F_NOT;
        Server1Read : TEST_CONDITION;
        F_NOT_1_1_1_2 : F_NOT;
        CLI1 : CLIENT_1(QI := 1);
        CLI01 : CLIENT_0_1(QI := 1);
        Client1_0Read : TEST_CONDITION;
        F_NOT_1_1_1_3 : F_NOT;
        CLI10 : CLIENT_1_0(QI := 1);
        STRING2STRING_1_1 : STRING2STRING;
        F_NOT_1_1_1_4 : F_NOT;
        Client0Read : TEST_CONDITION;
        CLI0 : CLIENT_0(QI := 1);
        SER1 : SERVER_1(QI := 1);
        F_NOT_1_1_1_2_1 : F_NOT;
        Server0_1Read : TEST_CONDITION;
        STRING2STRING_2 : STRING2STRING;
        STRING2STRING_2_1 : STRING2STRING;
        SER01 : SERVER_0_1(QI := 1);
        STRING2STRING_3 : STRING2STRING;
        Server1_0Read : TEST_CONDITION;
        F_NOT_1_1_1_2_1_1 : F_NOT;
        SER10 : SERVER_1_0(QI := 1);
        SUB2 : SUBSCRIBE_2(QI := 1);
        STRING2STRING_4 : STRING2STRING;
        Sub0ReadWrongNoRDs_ : TEST_CONDITION;
        F_NOT_2 : F_NOT;
        SUB0 : SUBSCRIBE_0;
      END_FBS
      EVENT_CONNECTIONS
        F_NOT_1_1_1.CNF TO Client1Read.REQ;
        F_NOT_1.CNF TO Pub1Read.REQ;
        Pub1Read.CNF TO SER0.INIT;
        SER0.INITO TO F_NOT_1_1.REQ;
        F_NOT_1_1.CNF TO Server0Read.REQ;
        Sub1ReadWrongNoRDs.CNF TO PUB1.INIT;
        PUB1.INITO TO F_NOT_1.REQ;
        F_NOT.CNF TO Sub1ReadWrongNoRDs.REQ;
        F_NOT_1_1_1_1.CNF TO Client0_1Read.REQ;
        F_NOT_1_1_1_2.CNF TO Server1Read.REQ;
        CLI1.INITO TO F_NOT_1_1_1.REQ;
        CLI01.INITO TO F_NOT_1_1_1_1.REQ;
        CLI0.INITO TO F_NOT_1_1_1_4.REQ;
        F_NOT_1_1_1_4.CNF TO Client0Read.REQ;
        F_NOT_1_1_1_3.CNF TO Client1_0Read.REQ;
        CLI10.INITO TO F_NOT_1_1_1_3.REQ;
        SER1.INITO TO F_NOT_1_1_1_2.REQ;
        F_NOT_1_1_1_2_1.CNF TO Server0_1Read.REQ;
        SER01.INITO TO F_NOT_1_1_1_2_1.REQ;
        Server0Read.CNF TO CLI0.INIT;
        Client0Read.CNF TO CLI1.INIT;
        Client1Read.CNF TO CLI01.INIT;
        Client0_1Read.CNF TO CLI10.INIT;
        Client1_0Read.CNF TO SER1.INIT;
        Server1Read.CNF TO SER01.INIT;
        F_NOT_1_1_1_2_1_1.CNF TO Server1_0Read.REQ;
        Server1_0Read.CNF TO CNF;
        Server0_1Read.CNF TO SER10.INIT;
        SER10.INITO TO F_NOT_1_1_1_2_1_1.REQ;
        SUB2.INITO TO F_NOT.REQ;
        REQ TO SUB0.INIT;
        SUB0.INITO TO F_NOT_2.REQ;
        F_NOT_2.CNF TO Sub0ReadWrongNoRDs_.REQ;
        Sub0ReadWrongNoRDs_.CNF TO SUB2.INIT;
      END_CONNECTIONS
      DATA_CONNECTIONS
        F_NOT_1_1_1.OUT TO Client1Read.check;
        F_NOT_1.OUT TO Pub1Read.check;
        SER0.QO TO F_NOT_1_1.IN;
        F_NOT_1_1.OUT TO Server0Read.check;
        STRING2STRING_1.OUT TO PUB1.SD_1;
        PUB1.QO TO F_NOT_1.IN;
        F_NOT.OUT TO Sub1ReadWrongNoRDs.check;
        F_NOT_1_1_1_1.OUT TO Client0_1Read.check;
        F_NOT_1_1_1_2.OUT TO Server1Read.check;
        CLI1.QO TO F_NOT_1_1_1.IN;
        CLI01.QO TO F_NOT_1_1_1_1.IN;
        STRING2STRING_1_1.OUT TO CLI1.SD_1;
        CLI1.RD_1 TO STRING2STRING_1_1.IN;
        F_NOT_1_1_1_4.OUT TO Client0Read.check;
        CLI0.QO TO F_NOT_1_1_1_4.IN;
        F_NOT_1_1_1_3.OUT TO Client1_0Read.check;
        CLI10.QO TO F_NOT_1_1_1_3.IN;
        SER1.QO TO F_NOT_1_1_1_2.IN;
        F_NOT_1_1_1_2_1.OUT TO Server0_1Read.check;
        CLI01.RD_1 TO STRING2STRING_2.IN;
        STRING2STRING_2.OUT TO CLI10.SD_1;
        STRING2STRING_2_1.OUT TO SER1.SD_1;
        SER1.RD_1 TO STRING2STRING_2_1.IN;
        SER01.QO TO F_NOT_1_1_1_2_1.IN;
        SER01.RD_1 TO STRING2STRING_3.IN;
        ID TO PUB1.ID;
        ID TO SER0.ID;
        ID TO CLI0.ID;
        ID TO CLI1.ID;
        ID TO CLI01.ID;
        ID TO CLI10.ID;
        ID TO SER01.ID;
        ID TO SER1.ID;
        F_NOT_1_1_1_2_1_1.OUT TO Server1_0Read.check;
        ID TO SER10.ID;
        SER10.QO TO F_NOT_1_1_1_2_1_1.IN;
        STRING2STRING_3.OUT TO SER10.SD_1;
        SUB2.QO TO F_NOT.IN;
        SUB2.RD_1 TO STRING2STRING.IN;
        SUB2.RD_2 TO STRING2STRING_4.IN;
        ID TO SUB2.ID;
        ID TO SUB0.ID;
        SUB0.QO TO F_NOT_2.IN;
        F_NOT_2.OUT TO Sub0ReadWrongNoRDs_.check;
      END_CONNECTIONS
    END_SUBAPPLICATION
    SUBAPPLICATION RemoteRead
      EVENT_INPUT
        REQ;
      END_EVENT
      EVENT_OUTPUT
        CNF;
      END_EVENT
      VAR_INPUT
        ID : WSTRING;
      END_VAR
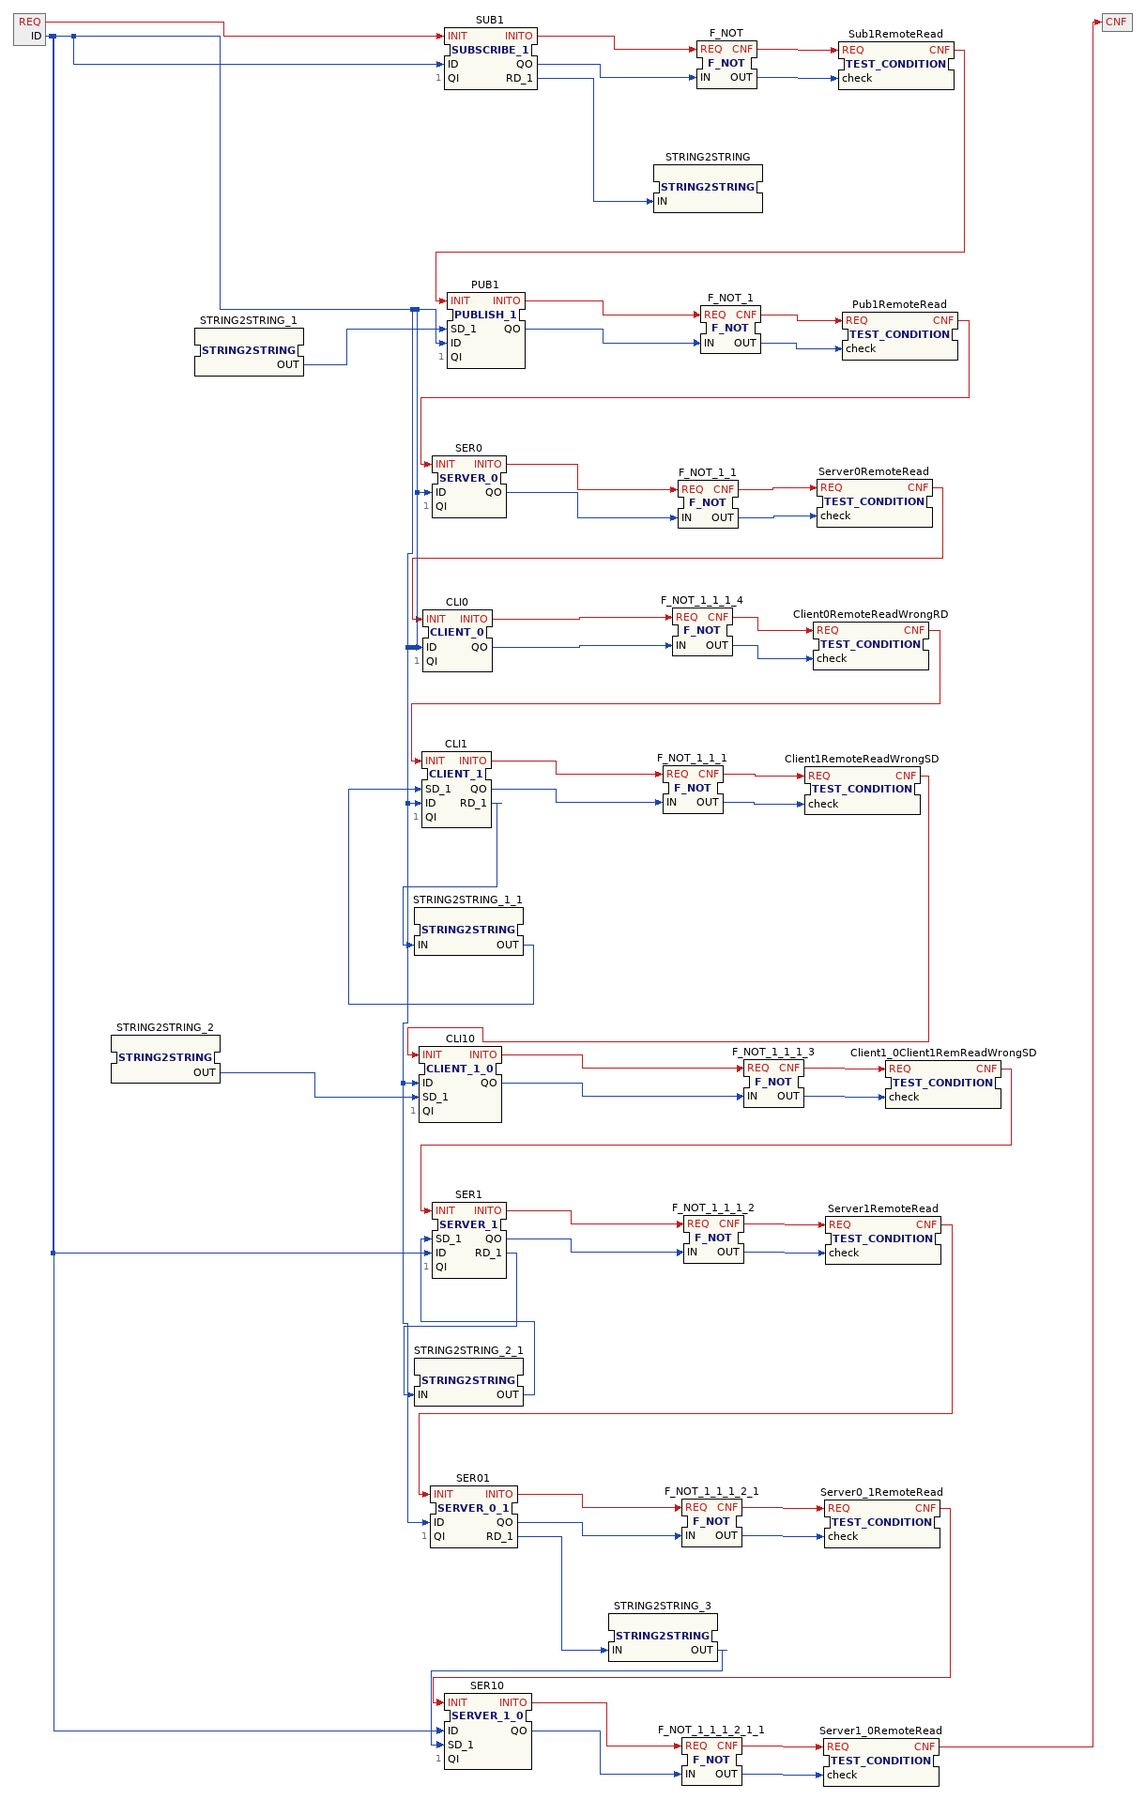
      FBS
        F_NOT_1_1_1 : F_NOT;
        Client1RemoteReadWrongSD : TEST_CONDITION;
        Pub1RemoteRead : TEST_CONDITION;
        F_NOT_1_1 : F_NOT;
        PUB1 : PUBLISH_1(QI := 1);
        F_NOT : F_NOT;
        Server0RemoteRead : TEST_CONDITION;
        Sub1RemoteRead : TEST_CONDITION;
        F_NOT_1 : F_NOT;
        STRING2STRING : STRING2STRING;
        SER0 : SERVER_0(QI := 1);
        STRING2STRING_1 : STRING2STRING;
        Server1RemoteRead : TEST_CONDITION;
        F_NOT_1_1_1_2 : F_NOT;
        CLI1 : CLIENT_1(QI := 1);
        Client1_0Client1RemReadWrongSD : TEST_CONDITION;
        F_NOT_1_1_1_3 : F_NOT;
        CLI10 : CLIENT_1_0(QI := 1);
        STRING2STRING_1_1 : STRING2STRING;
        F_NOT_1_1_1_4 : F_NOT;
        Client0RemoteReadWrongRD : TEST_CONDITION;
        CLI0 : CLIENT_0(QI := 1);
        SER1 : SERVER_1(QI := 1);
        F_NOT_1_1_1_2_1 : F_NOT;
        Server0_1RemoteRead : TEST_CONDITION;
        STRING2STRING_2_1 : STRING2STRING;
        SER01 : SERVER_0_1(QI := 1);
        STRING2STRING_3 : STRING2STRING;
        Server1_0RemoteRead : TEST_CONDITION;
        F_NOT_1_1_1_2_1_1 : F_NOT;
        SER10 : SERVER_1_0(QI := 1);
        SUB1 : SUBSCRIBE_1(QI := 1);
        STRING2STRING_2 : STRING2STRING;
      END_FBS
      EVENT_CONNECTIONS
        F_NOT_1_1_1.CNF TO Client1RemoteReadWrongSD.REQ;
        F_NOT_1.CNF TO Pub1RemoteRead.REQ;
        Pub1RemoteRead.CNF TO SER0.INIT;
        SER0.INITO TO F_NOT_1_1.REQ;
        F_NOT_1_1.CNF TO Server0RemoteRead.REQ;
        Sub1RemoteRead.CNF TO PUB1.INIT;
        PUB1.INITO TO F_NOT_1.REQ;
        F_NOT.CNF TO Sub1RemoteRead.REQ;
        F_NOT_1_1_1_2.CNF TO Server1RemoteRead.REQ;
        CLI1.INITO TO F_NOT_1_1_1.REQ;
        CLI0.INITO TO F_NOT_1_1_1_4.REQ;
        F_NOT_1_1_1_4.CNF TO Client0RemoteReadWrongRD.REQ;
        F_NOT_1_1_1_3.CNF TO Client1_0Client1RemReadWrongSD.REQ;
        CLI10.INITO TO F_NOT_1_1_1_3.REQ;
        SER1.INITO TO F_NOT_1_1_1_2.REQ;
        F_NOT_1_1_1_2_1.CNF TO Server0_1RemoteRead.REQ;
        SER01.INITO TO F_NOT_1_1_1_2_1.REQ;
        Server0RemoteRead.CNF TO CLI0.INIT;
        Client0RemoteReadWrongRD.CNF TO CLI1.INIT;
        Client1_0Client1RemReadWrongSD.CNF TO SER1.INIT;
        Server1RemoteRead.CNF TO SER01.INIT;
        F_NOT_1_1_1_2_1_1.CNF TO Server1_0RemoteRead.REQ;
        Server1_0RemoteRead.CNF TO CNF;
        Server0_1RemoteRead.CNF TO SER10.INIT;
        SER10.INITO TO F_NOT_1_1_1_2_1_1.REQ;
        REQ TO SUB1.INIT;
        SUB1.INITO TO F_NOT.REQ;
        Client1RemoteReadWrongSD.CNF TO CLI10.INIT;
      END_CONNECTIONS
      DATA_CONNECTIONS
        F_NOT_1_1_1.OUT TO Client1RemoteReadWrongSD.check;
        F_NOT_1.OUT TO Pub1RemoteRead.check;
        SER0.QO TO F_NOT_1_1.IN;
        F_NOT_1_1.OUT TO Server0RemoteRead.check;
        STRING2STRING_1.OUT TO PUB1.SD_1;
        PUB1.QO TO F_NOT_1.IN;
        F_NOT.OUT TO Sub1RemoteRead.check;
        F_NOT_1_1_1_2.OUT TO Server1RemoteRead.check;
        CLI1.QO TO F_NOT_1_1_1.IN;
        STRING2STRING_1_1.OUT TO CLI1.SD_1;
        CLI1.RD_1 TO STRING2STRING_1_1.IN;
        F_NOT_1_1_1_4.OUT TO Client0RemoteReadWrongRD.check;
        CLI0.QO TO F_NOT_1_1_1_4.IN;
        F_NOT_1_1_1_3.OUT TO Client1_0Client1RemReadWrongSD.check;
        CLI10.QO TO F_NOT_1_1_1_3.IN;
        SER1.QO TO F_NOT_1_1_1_2.IN;
        F_NOT_1_1_1_2_1.OUT TO Server0_1RemoteRead.check;
        STRING2STRING_2_1.OUT TO SER1.SD_1;
        SER1.RD_1 TO STRING2STRING_2_1.IN;
        SER01.QO TO F_NOT_1_1_1_2_1.IN;
        SER01.RD_1 TO STRING2STRING_3.IN;
        ID TO PUB1.ID;
        ID TO SER0.ID;
        ID TO CLI0.ID;
        ID TO CLI1.ID;
        ID TO CLI10.ID;
        ID TO SER01.ID;
        ID TO SER1.ID;
        F_NOT_1_1_1_2_1_1.OUT TO Server1_0RemoteRead.check;
        ID TO SER10.ID;
        SER10.QO TO F_NOT_1_1_1_2_1_1.IN;
        STRING2STRING_3.OUT TO SER10.SD_1;
        ID TO SUB1.ID;
        SUB1.QO TO F_NOT.IN;
        SUB1.RD_1 TO STRING2STRING.IN;
        STRING2STRING_2.OUT TO CLI10.SD_1;
      END_CONNECTIONS
    END_SUBAPPLICATION
    SUBAPPLICATION LocalWrite
      EVENT_INPUT
        REQ;
      END_EVENT
      EVENT_OUTPUT
        CNF;
      END_EVENT
      VAR_INPUT
        ID : WSTRING;
      END_VAR
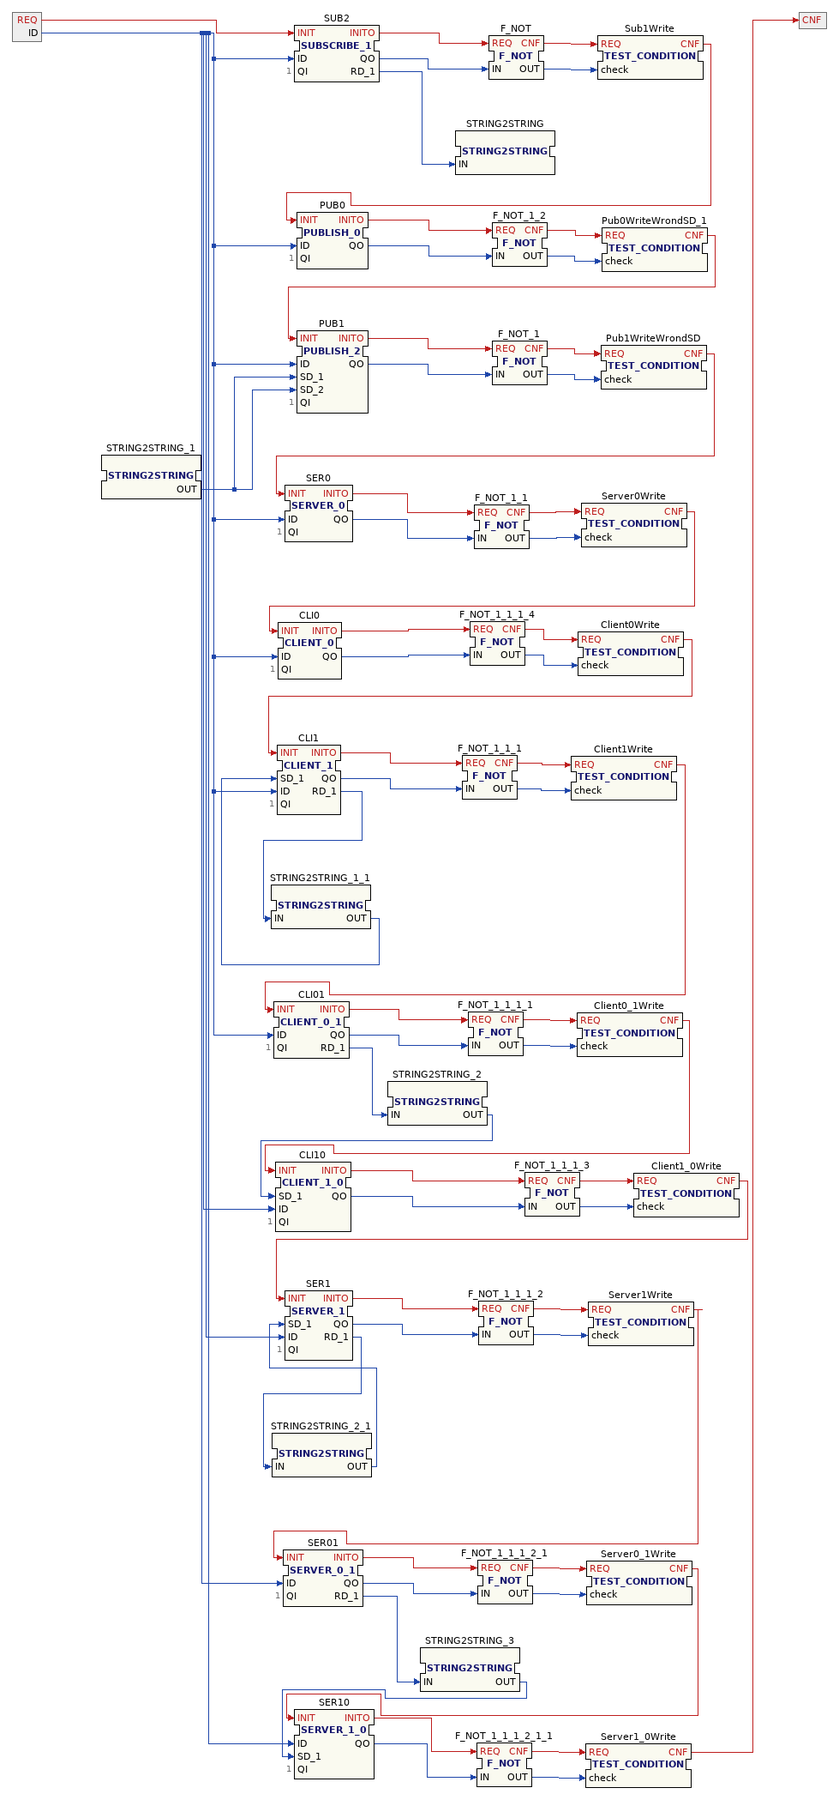
      FBS
        F_NOT_1_1_1 : F_NOT;
        Client1Write : TEST_CONDITION;
        Pub1WriteWrondSD : TEST_CONDITION;
        F_NOT_1_1 : F_NOT;
        F_NOT : F_NOT;
        Server0Write : TEST_CONDITION;
        Sub1Write : TEST_CONDITION;
        F_NOT_1 : F_NOT;
        STRING2STRING : STRING2STRING;
        SER0 : SERVER_0(QI := 1);
        STRING2STRING_1 : STRING2STRING;
        Client0_1Write : TEST_CONDITION;
        F_NOT_1_1_1_1 : F_NOT;
        Server1Write : TEST_CONDITION;
        F_NOT_1_1_1_2 : F_NOT;
        CLI1 : CLIENT_1(QI := 1);
        CLI01 : CLIENT_0_1(QI := 1);
        Client1_0Write : TEST_CONDITION;
        F_NOT_1_1_1_3 : F_NOT;
        CLI10 : CLIENT_1_0(QI := 1);
        STRING2STRING_1_1 : STRING2STRING;
        F_NOT_1_1_1_4 : F_NOT;
        Client0Write : TEST_CONDITION;
        CLI0 : CLIENT_0(QI := 1);
        SER1 : SERVER_1(QI := 1);
        F_NOT_1_1_1_2_1 : F_NOT;
        Server0_1Write : TEST_CONDITION;
        STRING2STRING_2 : STRING2STRING;
        STRING2STRING_2_1 : STRING2STRING;
        SER01 : SERVER_0_1(QI := 1);
        STRING2STRING_3 : STRING2STRING;
        Server1_0Write : TEST_CONDITION;
        F_NOT_1_1_1_2_1_1 : F_NOT;
        SER10 : SERVER_1_0(QI := 1);
        SUB2 : SUBSCRIBE_1(QI := 1);
        PUB1 : PUBLISH_2(QI := 1);
        Pub0WriteWrondSD_1 : TEST_CONDITION;
        F_NOT_1_2 : F_NOT;
        PUB0 : PUBLISH_0(QI := 1);
      END_FBS
      EVENT_CONNECTIONS
        F_NOT_1_1_1.CNF TO Client1Write.REQ;
        F_NOT_1.CNF TO Pub1WriteWrondSD.REQ;
        Pub1WriteWrondSD.CNF TO SER0.INIT;
        SER0.INITO TO F_NOT_1_1.REQ;
        F_NOT_1_1.CNF TO Server0Write.REQ;
        F_NOT.CNF TO Sub1Write.REQ;
        F_NOT_1_1_1_1.CNF TO Client0_1Write.REQ;
        F_NOT_1_1_1_2.CNF TO Server1Write.REQ;
        CLI1.INITO TO F_NOT_1_1_1.REQ;
        CLI01.INITO TO F_NOT_1_1_1_1.REQ;
        CLI0.INITO TO F_NOT_1_1_1_4.REQ;
        F_NOT_1_1_1_4.CNF TO Client0Write.REQ;
        F_NOT_1_1_1_3.CNF TO Client1_0Write.REQ;
        CLI10.INITO TO F_NOT_1_1_1_3.REQ;
        SER1.INITO TO F_NOT_1_1_1_2.REQ;
        F_NOT_1_1_1_2_1.CNF TO Server0_1Write.REQ;
        SER01.INITO TO F_NOT_1_1_1_2_1.REQ;
        Server0Write.CNF TO CLI0.INIT;
        Client0Write.CNF TO CLI1.INIT;
        Client1Write.CNF TO CLI01.INIT;
        Client0_1Write.CNF TO CLI10.INIT;
        Client1_0Write.CNF TO SER1.INIT;
        Server1Write.CNF TO SER01.INIT;
        F_NOT_1_1_1_2_1_1.CNF TO Server1_0Write.REQ;
        Server1_0Write.CNF TO CNF;
        Server0_1Write.CNF TO SER10.INIT;
        SER10.INITO TO F_NOT_1_1_1_2_1_1.REQ;
        REQ TO SUB2.INIT;
        SUB2.INITO TO F_NOT.REQ;
        PUB1.INITO TO F_NOT_1.REQ;
        F_NOT_1_2.CNF TO Pub0WriteWrondSD_1.REQ;
        PUB0.INITO TO F_NOT_1_2.REQ;
        Sub1Write.CNF TO PUB0.INIT;
        Pub0WriteWrondSD_1.CNF TO PUB1.INIT;
      END_CONNECTIONS
      DATA_CONNECTIONS
        F_NOT_1_1_1.OUT TO Client1Write.check;
        F_NOT_1.OUT TO Pub1WriteWrondSD.check;
        SER0.QO TO F_NOT_1_1.IN;
        F_NOT_1_1.OUT TO Server0Write.check;
        F_NOT.OUT TO Sub1Write.check;
        F_NOT_1_1_1_1.OUT TO Client0_1Write.check;
        F_NOT_1_1_1_2.OUT TO Server1Write.check;
        CLI1.QO TO F_NOT_1_1_1.IN;
        CLI01.QO TO F_NOT_1_1_1_1.IN;
        STRING2STRING_1_1.OUT TO CLI1.SD_1;
        CLI1.RD_1 TO STRING2STRING_1_1.IN;
        F_NOT_1_1_1_4.OUT TO Client0Write.check;
        CLI0.QO TO F_NOT_1_1_1_4.IN;
        F_NOT_1_1_1_3.OUT TO Client1_0Write.check;
        CLI10.QO TO F_NOT_1_1_1_3.IN;
        SER1.QO TO F_NOT_1_1_1_2.IN;
        F_NOT_1_1_1_2_1.OUT TO Server0_1Write.check;
        CLI01.RD_1 TO STRING2STRING_2.IN;
        STRING2STRING_2.OUT TO CLI10.SD_1;
        STRING2STRING_2_1.OUT TO SER1.SD_1;
        SER1.RD_1 TO STRING2STRING_2_1.IN;
        SER01.QO TO F_NOT_1_1_1_2_1.IN;
        SER01.RD_1 TO STRING2STRING_3.IN;
        ID TO SER0.ID;
        ID TO CLI0.ID;
        ID TO CLI1.ID;
        ID TO CLI01.ID;
        ID TO CLI10.ID;
        ID TO SER01.ID;
        ID TO SER1.ID;
        F_NOT_1_1_1_2_1_1.OUT TO Server1_0Write.check;
        ID TO SER10.ID;
        SER10.QO TO F_NOT_1_1_1_2_1_1.IN;
        STRING2STRING_3.OUT TO SER10.SD_1;
        ID TO SUB2.ID;
        SUB2.QO TO F_NOT.IN;
        SUB2.RD_1 TO STRING2STRING.IN;
        ID TO PUB1.ID;
        STRING2STRING_1.OUT TO PUB1.SD_1;
        PUB1.QO TO F_NOT_1.IN;
        STRING2STRING_1.OUT TO PUB1.SD_2;
        F_NOT_1_2.OUT TO Pub0WriteWrondSD_1.check;
        PUB0.QO TO F_NOT_1_2.IN;
        ID TO PUB0.ID;
      END_CONNECTIONS
    END_SUBAPPLICATION
    SUBAPPLICATION RemoteWrite
      EVENT_INPUT
        REQ;
      END_EVENT
      EVENT_OUTPUT
        CNF;
      END_EVENT
      VAR_INPUT
        ID : WSTRING;
      END_VAR
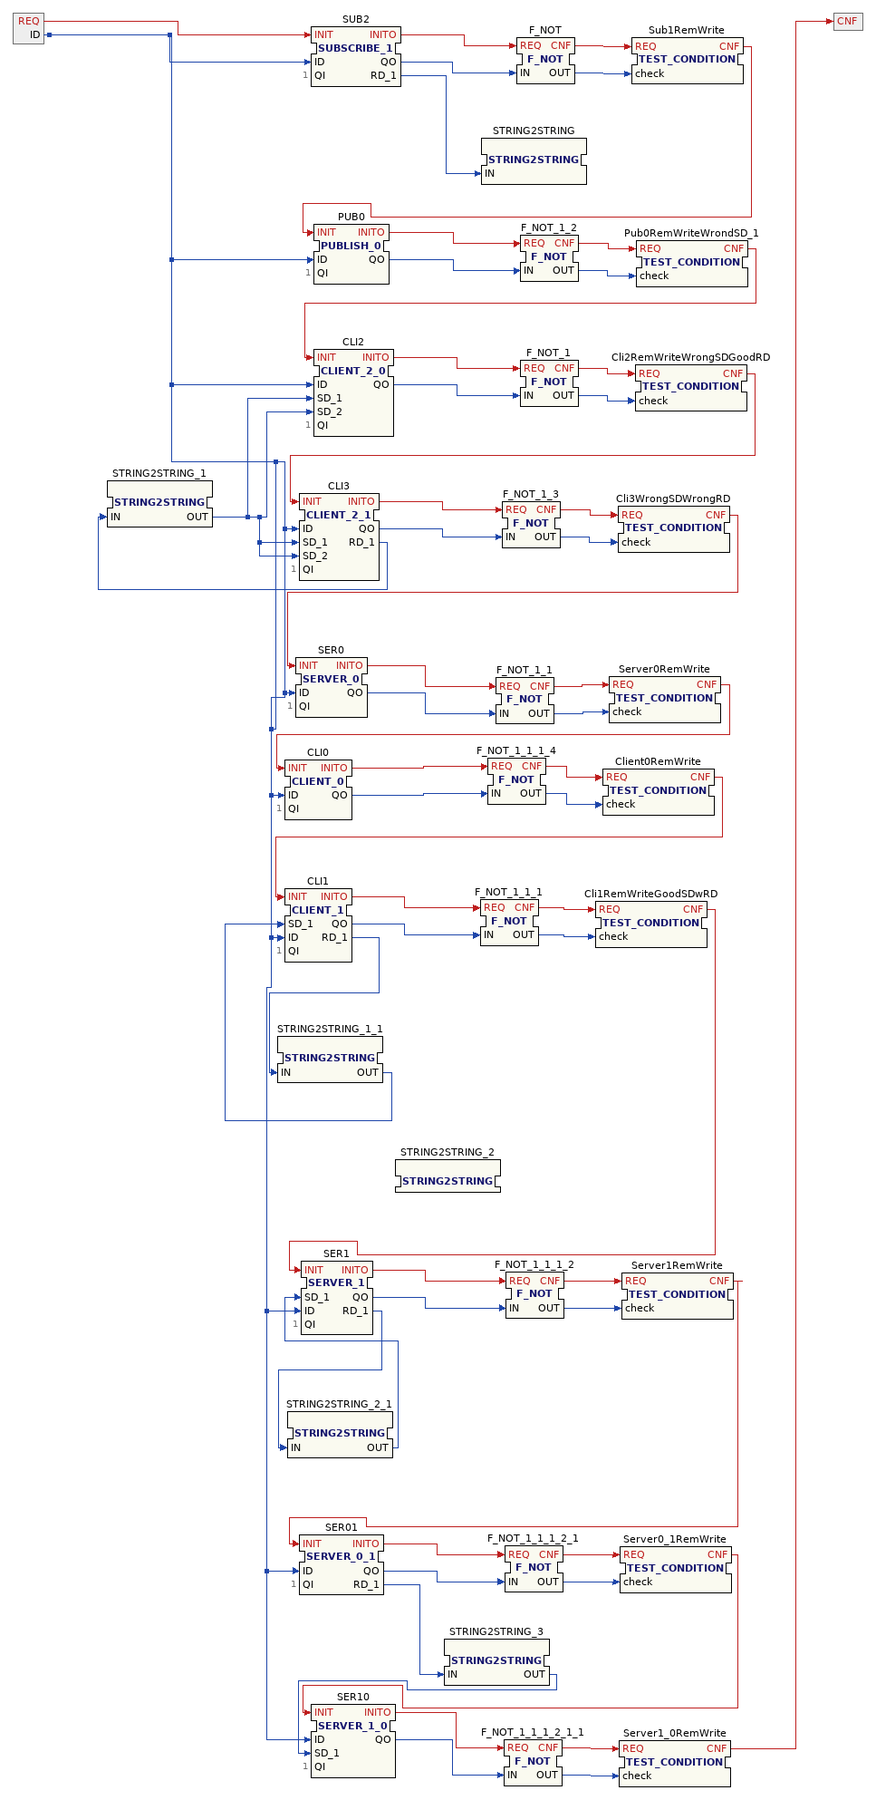
      FBS
        F_NOT_1_1_1 : F_NOT;
        Cli1RemWriteGoodSDwRD : TEST_CONDITION;
        Cli2RemWriteWrongSDGoodRD : TEST_CONDITION;
        F_NOT_1_1 : F_NOT;
        F_NOT : F_NOT;
        Server0RemWrite : TEST_CONDITION;
        Sub1RemWrite : TEST_CONDITION;
        F_NOT_1 : F_NOT;
        STRING2STRING : STRING2STRING;
        SER0 : SERVER_0(QI := 1);
        STRING2STRING_1 : STRING2STRING;
        Server1RemWrite : TEST_CONDITION;
        F_NOT_1_1_1_2 : F_NOT;
        CLI1 : CLIENT_1(QI := 1);
        STRING2STRING_1_1 : STRING2STRING;
        F_NOT_1_1_1_4 : F_NOT;
        Client0RemWrite : TEST_CONDITION;
        CLI0 : CLIENT_0(QI := 1);
        SER1 : SERVER_1(QI := 1);
        F_NOT_1_1_1_2_1 : F_NOT;
        Server0_1RemWrite : TEST_CONDITION;
        STRING2STRING_2 : STRING2STRING;
        STRING2STRING_2_1 : STRING2STRING;
        SER01 : SERVER_0_1(QI := 1);
        STRING2STRING_3 : STRING2STRING;
        Server1_0RemWrite : TEST_CONDITION;
        F_NOT_1_1_1_2_1_1 : F_NOT;
        SER10 : SERVER_1_0(QI := 1);
        SUB2 : SUBSCRIBE_1(QI := 1);
        Pub0RemWriteWrondSD_1 : TEST_CONDITION;
        F_NOT_1_2 : F_NOT;
        PUB0 : PUBLISH_0(QI := 1);
        CLI2 : CLIENT_2_0(QI := 1);
        F_NOT_1_3 : F_NOT;
        Cli3WrongSDWrongRD : TEST_CONDITION;
        CLI3 : CLIENT_2_1(QI := 1);
      END_FBS
      EVENT_CONNECTIONS
        F_NOT_1_1_1.CNF TO Cli1RemWriteGoodSDwRD.REQ;
        F_NOT_1.CNF TO Cli2RemWriteWrongSDGoodRD.REQ;
        SER0.INITO TO F_NOT_1_1.REQ;
        F_NOT_1_1.CNF TO Server0RemWrite.REQ;
        F_NOT.CNF TO Sub1RemWrite.REQ;
        F_NOT_1_1_1_2.CNF TO Server1RemWrite.REQ;
        CLI1.INITO TO F_NOT_1_1_1.REQ;
        CLI0.INITO TO F_NOT_1_1_1_4.REQ;
        F_NOT_1_1_1_4.CNF TO Client0RemWrite.REQ;
        SER1.INITO TO F_NOT_1_1_1_2.REQ;
        F_NOT_1_1_1_2_1.CNF TO Server0_1RemWrite.REQ;
        SER01.INITO TO F_NOT_1_1_1_2_1.REQ;
        Server0RemWrite.CNF TO CLI0.INIT;
        Client0RemWrite.CNF TO CLI1.INIT;
        Server1RemWrite.CNF TO SER01.INIT;
        F_NOT_1_1_1_2_1_1.CNF TO Server1_0RemWrite.REQ;
        Server1_0RemWrite.CNF TO CNF;
        Server0_1RemWrite.CNF TO SER10.INIT;
        SER10.INITO TO F_NOT_1_1_1_2_1_1.REQ;
        REQ TO SUB2.INIT;
        SUB2.INITO TO F_NOT.REQ;
        F_NOT_1_2.CNF TO Pub0RemWriteWrondSD_1.REQ;
        PUB0.INITO TO F_NOT_1_2.REQ;
        Sub1RemWrite.CNF TO PUB0.INIT;
        Pub0RemWriteWrondSD_1.CNF TO CLI2.INIT;
        CLI2.INITO TO F_NOT_1.REQ;
        F_NOT_1_3.CNF TO Cli3WrongSDWrongRD.REQ;
        Cli3WrongSDWrongRD.CNF TO SER0.INIT;
        Cli2RemWriteWrongSDGoodRD.CNF TO CLI3.INIT;
        CLI3.INITO TO F_NOT_1_3.REQ;
        Cli1RemWriteGoodSDwRD.CNF TO SER1.INIT;
      END_CONNECTIONS
      DATA_CONNECTIONS
        F_NOT_1_1_1.OUT TO Cli1RemWriteGoodSDwRD.check;
        F_NOT_1.OUT TO Cli2RemWriteWrongSDGoodRD.check;
        SER0.QO TO F_NOT_1_1.IN;
        F_NOT_1_1.OUT TO Server0RemWrite.check;
        F_NOT.OUT TO Sub1RemWrite.check;
        F_NOT_1_1_1_2.OUT TO Server1RemWrite.check;
        CLI1.QO TO F_NOT_1_1_1.IN;
        STRING2STRING_1_1.OUT TO CLI1.SD_1;
        CLI1.RD_1 TO STRING2STRING_1_1.IN;
        F_NOT_1_1_1_4.OUT TO Client0RemWrite.check;
        CLI0.QO TO F_NOT_1_1_1_4.IN;
        SER1.QO TO F_NOT_1_1_1_2.IN;
        F_NOT_1_1_1_2_1.OUT TO Server0_1RemWrite.check;
        STRING2STRING_2_1.OUT TO SER1.SD_1;
        SER1.RD_1 TO STRING2STRING_2_1.IN;
        SER01.QO TO F_NOT_1_1_1_2_1.IN;
        SER01.RD_1 TO STRING2STRING_3.IN;
        ID TO SER0.ID;
        ID TO CLI0.ID;
        ID TO CLI1.ID;
        ID TO SER01.ID;
        ID TO SER1.ID;
        F_NOT_1_1_1_2_1_1.OUT TO Server1_0RemWrite.check;
        ID TO SER10.ID;
        SER10.QO TO F_NOT_1_1_1_2_1_1.IN;
        STRING2STRING_3.OUT TO SER10.SD_1;
        ID TO SUB2.ID;
        SUB2.QO TO F_NOT.IN;
        SUB2.RD_1 TO STRING2STRING.IN;
        F_NOT_1_2.OUT TO Pub0RemWriteWrondSD_1.check;
        PUB0.QO TO F_NOT_1_2.IN;
        ID TO PUB0.ID;
        ID TO CLI2.ID;
        STRING2STRING_1.OUT TO CLI2.SD_1;
        STRING2STRING_1.OUT TO CLI2.SD_2;
        CLI2.QO TO F_NOT_1.IN;
        F_NOT_1_3.OUT TO Cli3WrongSDWrongRD.check;
        ID TO CLI3.ID;
        STRING2STRING_1.OUT TO CLI3.SD_1;
        STRING2STRING_1.OUT TO CLI3.SD_2;
        CLI3.QO TO F_NOT_1_3.IN;
        CLI3.RD_1 TO STRING2STRING_1.IN;
      END_CONNECTIONS
    END_SUBAPPLICATION
    SUBAPPLICATION CreateMethod
      EVENT_INPUT
        REQ;
      END_EVENT
      EVENT_OUTPUT
        CNF;
      END_EVENT
      VAR_INPUT
        ID : WSTRING;
      END_VAR
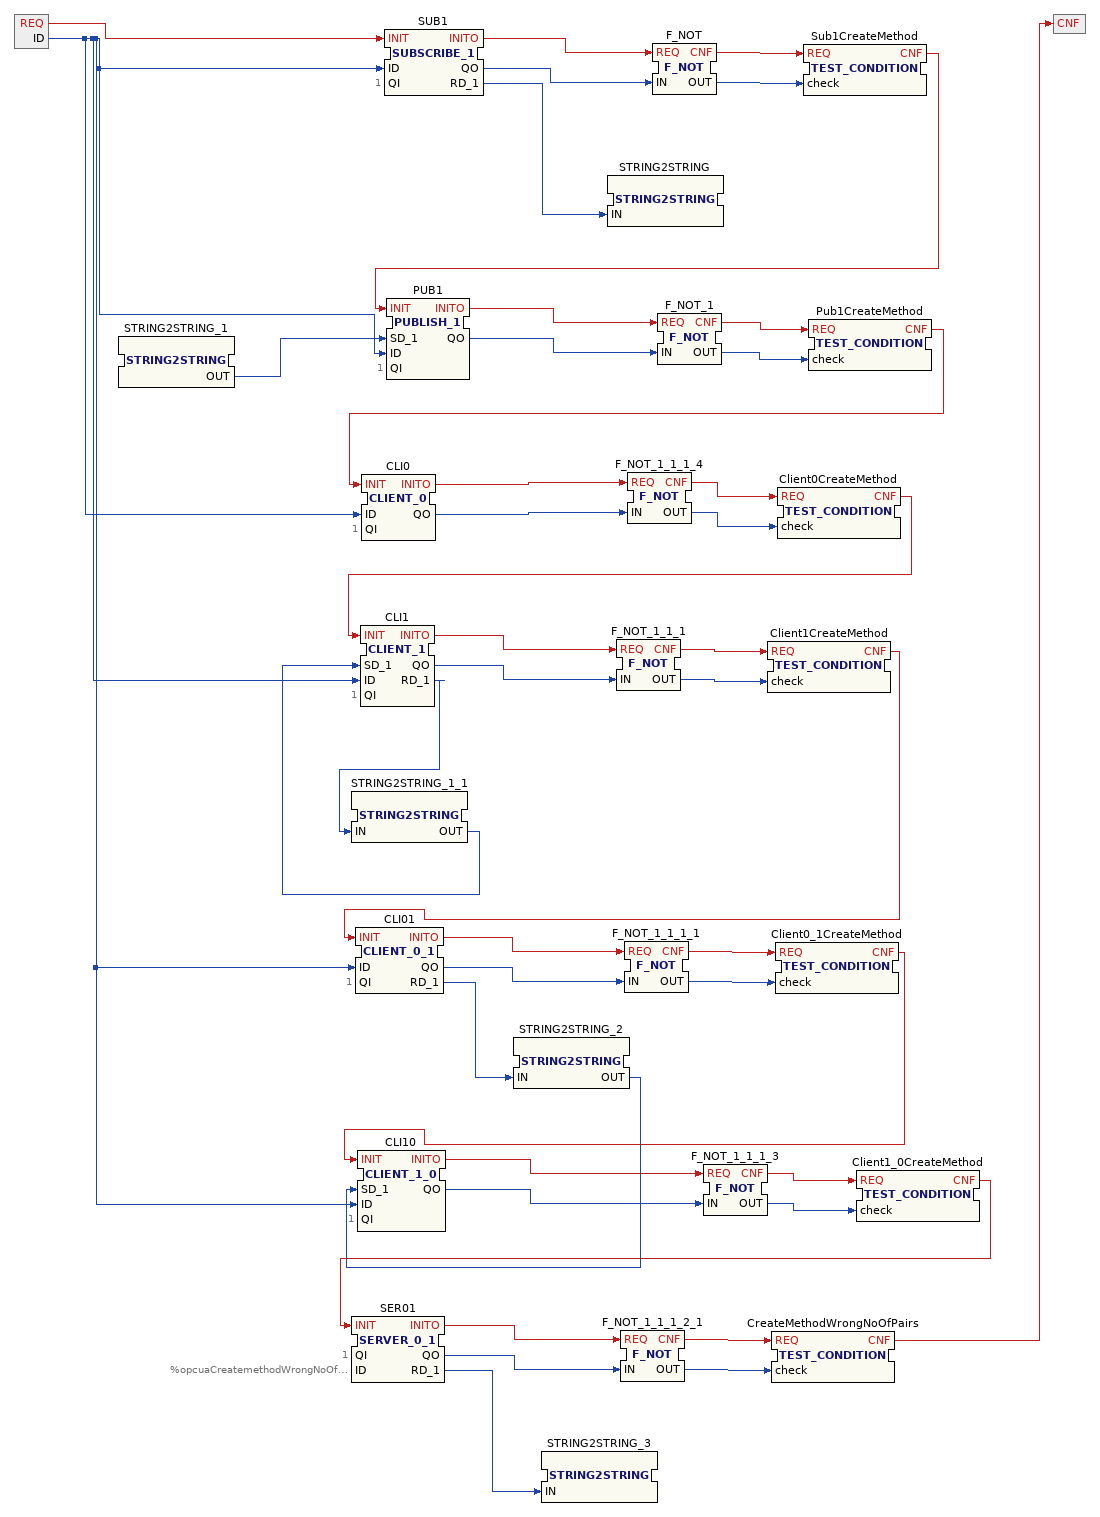
      FBS
        F_NOT_1_1_1 : F_NOT;
        Client1CreateMethod : TEST_CONDITION;
        Pub1CreateMethod : TEST_CONDITION;
        PUB1 : PUBLISH_1(QI := 1);
        F_NOT : F_NOT;
        Sub1CreateMethod : TEST_CONDITION;
        F_NOT_1 : F_NOT;
        STRING2STRING : STRING2STRING;
        SUB1 : SUBSCRIBE_1(QI := 1);
        STRING2STRING_1 : STRING2STRING;
        Client0_1CreateMethod : TEST_CONDITION;
        F_NOT_1_1_1_1 : F_NOT;
        CLI1 : CLIENT_1(QI := 1);
        CLI01 : CLIENT_0_1(QI := 1);
        Client1_0CreateMethod : TEST_CONDITION;
        F_NOT_1_1_1_3 : F_NOT;
        CLI10 : CLIENT_1_0(QI := 1);
        STRING2STRING_1_1 : STRING2STRING;
        F_NOT_1_1_1_4 : F_NOT;
        Client0CreateMethod : TEST_CONDITION;
        CLI0 : CLIENT_0(QI := 1);
        F_NOT_1_1_1_2_1 : F_NOT;
        CreateMethodWrongNoOfPairs : TEST_CONDITION;
        STRING2STRING_2 : STRING2STRING;
        SER01 : SERVER_0_1(QI := 1, ID := %opcuaCreatemethodWrongNoOfPairs%);
        STRING2STRING_3 : STRING2STRING;
      END_FBS
      EVENT_CONNECTIONS
        F_NOT_1_1_1.CNF TO Client1CreateMethod.REQ;
        F_NOT_1.CNF TO Pub1CreateMethod.REQ;
        Sub1CreateMethod.CNF TO PUB1.INIT;
        PUB1.INITO TO F_NOT_1.REQ;
        SUB1.INITO TO F_NOT.REQ;
        F_NOT.CNF TO Sub1CreateMethod.REQ;
        REQ TO SUB1.INIT;
        F_NOT_1_1_1_1.CNF TO Client0_1CreateMethod.REQ;
        CLI1.INITO TO F_NOT_1_1_1.REQ;
        CLI01.INITO TO F_NOT_1_1_1_1.REQ;
        CLI0.INITO TO F_NOT_1_1_1_4.REQ;
        F_NOT_1_1_1_4.CNF TO Client0CreateMethod.REQ;
        F_NOT_1_1_1_3.CNF TO Client1_0CreateMethod.REQ;
        CLI10.INITO TO F_NOT_1_1_1_3.REQ;
        F_NOT_1_1_1_2_1.CNF TO CreateMethodWrongNoOfPairs.REQ;
        SER01.INITO TO F_NOT_1_1_1_2_1.REQ;
        Client0CreateMethod.CNF TO CLI1.INIT;
        Client1CreateMethod.CNF TO CLI01.INIT;
        Client0_1CreateMethod.CNF TO CLI10.INIT;
        Pub1CreateMethod.CNF TO CLI0.INIT;
        Client1_0CreateMethod.CNF TO SER01.INIT;
        CreateMethodWrongNoOfPairs.CNF TO CNF;
      END_CONNECTIONS
      DATA_CONNECTIONS
        F_NOT_1_1_1.OUT TO Client1CreateMethod.check;
        F_NOT_1.OUT TO Pub1CreateMethod.check;
        STRING2STRING_1.OUT TO PUB1.SD_1;
        PUB1.QO TO F_NOT_1.IN;
        SUB1.QO TO F_NOT.IN;
        F_NOT.OUT TO Sub1CreateMethod.check;
        SUB1.RD_1 TO STRING2STRING.IN;
        F_NOT_1_1_1_1.OUT TO Client0_1CreateMethod.check;
        CLI1.QO TO F_NOT_1_1_1.IN;
        CLI01.QO TO F_NOT_1_1_1_1.IN;
        STRING2STRING_1_1.OUT TO CLI1.SD_1;
        CLI1.RD_1 TO STRING2STRING_1_1.IN;
        F_NOT_1_1_1_4.OUT TO Client0CreateMethod.check;
        CLI0.QO TO F_NOT_1_1_1_4.IN;
        F_NOT_1_1_1_3.OUT TO Client1_0CreateMethod.check;
        CLI10.QO TO F_NOT_1_1_1_3.IN;
        F_NOT_1_1_1_2_1.OUT TO CreateMethodWrongNoOfPairs.check;
        CLI01.RD_1 TO STRING2STRING_2.IN;
        STRING2STRING_2.OUT TO CLI10.SD_1;
        SER01.QO TO F_NOT_1_1_1_2_1.IN;
        SER01.RD_1 TO STRING2STRING_3.IN;
        ID TO SUB1.ID;
        ID TO PUB1.ID;
        ID TO CLI0.ID;
        ID TO CLI1.ID;
        ID TO CLI01.ID;
        ID TO CLI10.ID;
      END_CONNECTIONS
    END_SUBAPPLICATION
    SUBAPPLICATION CallMethod
      EVENT_INPUT
        REQ;
      END_EVENT
      EVENT_OUTPUT
        CNF;
      END_EVENT
      VAR_INPUT
        ID : WSTRING;
      END_VAR
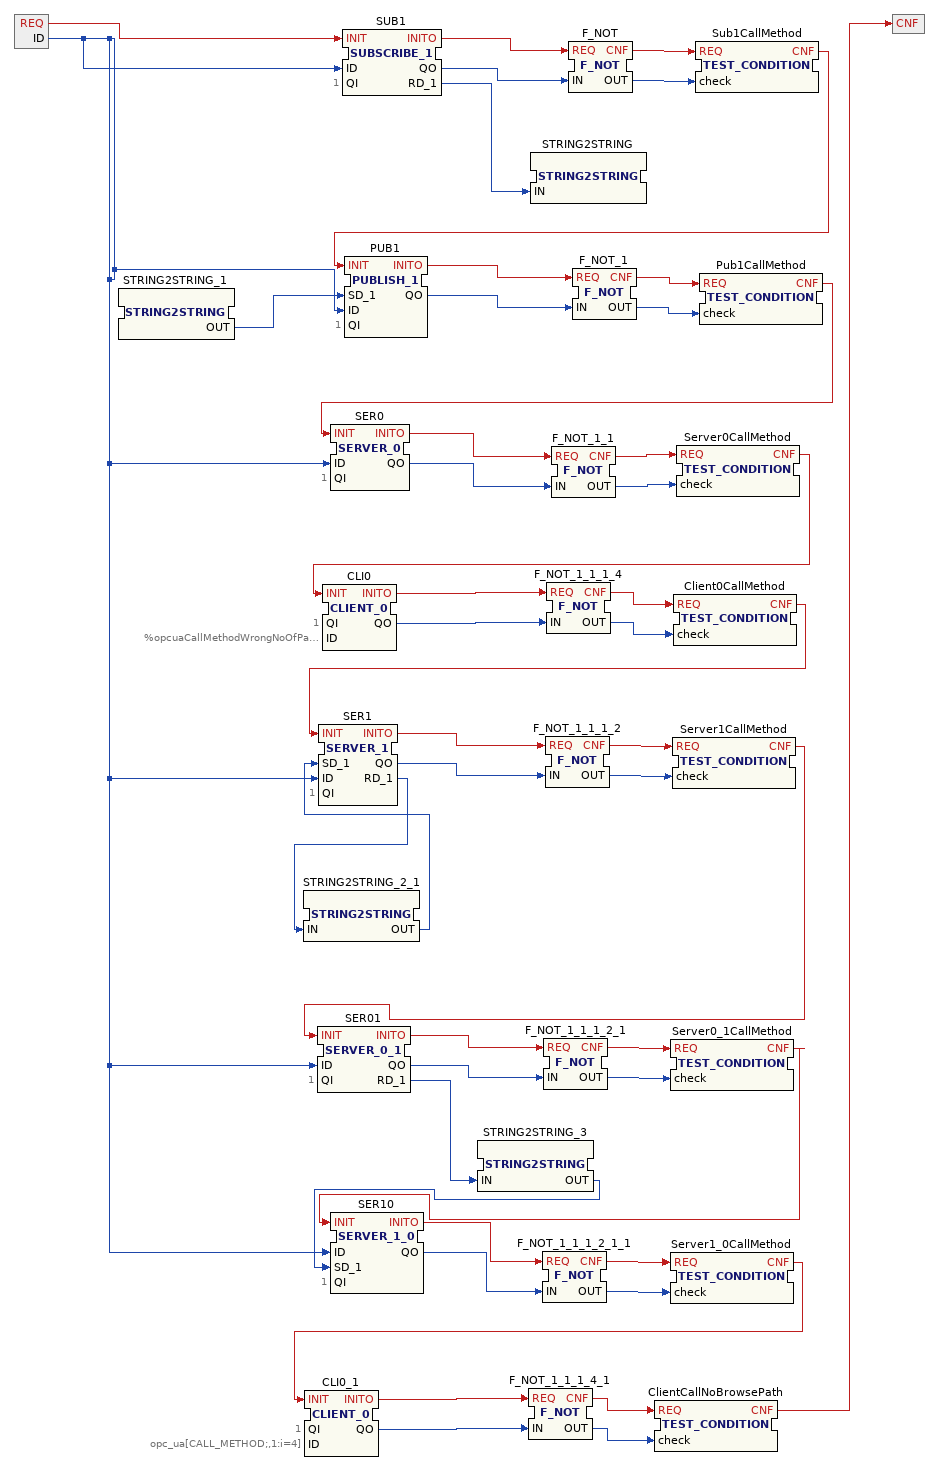
      FBS
        Pub1CallMethod : TEST_CONDITION;
        F_NOT_1_1 : F_NOT;
        PUB1 : PUBLISH_1(QI := 1);
        F_NOT : F_NOT;
        Server0CallMethod : TEST_CONDITION;
        Sub1CallMethod : TEST_CONDITION;
        F_NOT_1 : F_NOT;
        STRING2STRING : STRING2STRING;
        SUB1 : SUBSCRIBE_1(QI := 1);
        SER0 : SERVER_0(QI := 1);
        STRING2STRING_1 : STRING2STRING;
        Server1CallMethod : TEST_CONDITION;
        F_NOT_1_1_1_2 : F_NOT;
        F_NOT_1_1_1_4 : F_NOT;
        Client0CallMethod : TEST_CONDITION;
        CLI0 : CLIENT_0(QI := 1, ID := %opcuaCallMethodWrongNoOfPairs%);
        SER1 : SERVER_1(QI := 1);
        F_NOT_1_1_1_2_1 : F_NOT;
        Server0_1CallMethod : TEST_CONDITION;
        STRING2STRING_2_1 : STRING2STRING;
        SER01 : SERVER_0_1(QI := 1);
        STRING2STRING_3 : STRING2STRING;
        Server1_0CallMethod : TEST_CONDITION;
        F_NOT_1_1_1_2_1_1 : F_NOT;
        SER10 : SERVER_1_0(QI := 1);
        CLI0_1 : CLIENT_0(QI := 1, ID := opc_ua[CALL_METHOD;,1:i=4]);
        ClientCallNoBrowsePath : TEST_CONDITION;
        F_NOT_1_1_1_4_1 : F_NOT;
      END_FBS
      EVENT_CONNECTIONS
        F_NOT_1.CNF TO Pub1CallMethod.REQ;
        Pub1CallMethod.CNF TO SER0.INIT;
        SER0.INITO TO F_NOT_1_1.REQ;
        F_NOT_1_1.CNF TO Server0CallMethod.REQ;
        Sub1CallMethod.CNF TO PUB1.INIT;
        PUB1.INITO TO F_NOT_1.REQ;
        SUB1.INITO TO F_NOT.REQ;
        F_NOT.CNF TO Sub1CallMethod.REQ;
        REQ TO SUB1.INIT;
        F_NOT_1_1_1_2.CNF TO Server1CallMethod.REQ;
        CLI0.INITO TO F_NOT_1_1_1_4.REQ;
        F_NOT_1_1_1_4.CNF TO Client0CallMethod.REQ;
        SER1.INITO TO F_NOT_1_1_1_2.REQ;
        F_NOT_1_1_1_2_1.CNF TO Server0_1CallMethod.REQ;
        SER01.INITO TO F_NOT_1_1_1_2_1.REQ;
        Server0CallMethod.CNF TO CLI0.INIT;
        Server1CallMethod.CNF TO SER01.INIT;
        F_NOT_1_1_1_2_1_1.CNF TO Server1_0CallMethod.REQ;
        Server0_1CallMethod.CNF TO SER10.INIT;
        SER10.INITO TO F_NOT_1_1_1_2_1_1.REQ;
        Client0CallMethod.CNF TO SER1.INIT;
        F_NOT_1_1_1_4_1.CNF TO ClientCallNoBrowsePath.REQ;
        ClientCallNoBrowsePath.CNF TO CNF;
        Server1_0CallMethod.CNF TO CLI0_1.INIT;
        CLI0_1.INITO TO F_NOT_1_1_1_4_1.REQ;
      END_CONNECTIONS
      DATA_CONNECTIONS
        F_NOT_1.OUT TO Pub1CallMethod.check;
        SER0.QO TO F_NOT_1_1.IN;
        F_NOT_1_1.OUT TO Server0CallMethod.check;
        STRING2STRING_1.OUT TO PUB1.SD_1;
        PUB1.QO TO F_NOT_1.IN;
        SUB1.QO TO F_NOT.IN;
        F_NOT.OUT TO Sub1CallMethod.check;
        SUB1.RD_1 TO STRING2STRING.IN;
        F_NOT_1_1_1_2.OUT TO Server1CallMethod.check;
        F_NOT_1_1_1_4.OUT TO Client0CallMethod.check;
        CLI0.QO TO F_NOT_1_1_1_4.IN;
        SER1.QO TO F_NOT_1_1_1_2.IN;
        F_NOT_1_1_1_2_1.OUT TO Server0_1CallMethod.check;
        STRING2STRING_2_1.OUT TO SER1.SD_1;
        SER1.RD_1 TO STRING2STRING_2_1.IN;
        SER01.QO TO F_NOT_1_1_1_2_1.IN;
        SER01.RD_1 TO STRING2STRING_3.IN;
        ID TO SUB1.ID;
        ID TO PUB1.ID;
        ID TO SER0.ID;
        ID TO SER01.ID;
        ID TO SER1.ID;
        F_NOT_1_1_1_2_1_1.OUT TO Server1_0CallMethod.check;
        ID TO SER10.ID;
        SER10.QO TO F_NOT_1_1_1_2_1_1.IN;
        STRING2STRING_3.OUT TO SER10.SD_1;
        F_NOT_1_1_1_4_1.OUT TO ClientCallNoBrowsePath.check;
        CLI0_1.QO TO F_NOT_1_1_1_4_1.IN;
      END_CONNECTIONS
    END_SUBAPPLICATION
    SUBAPPLICATION Subscribe
      EVENT_INPUT
        REQ;
      END_EVENT
      EVENT_OUTPUT
        CNF;
      END_EVENT
      VAR_INPUT
        ID : WSTRING;
      END_VAR
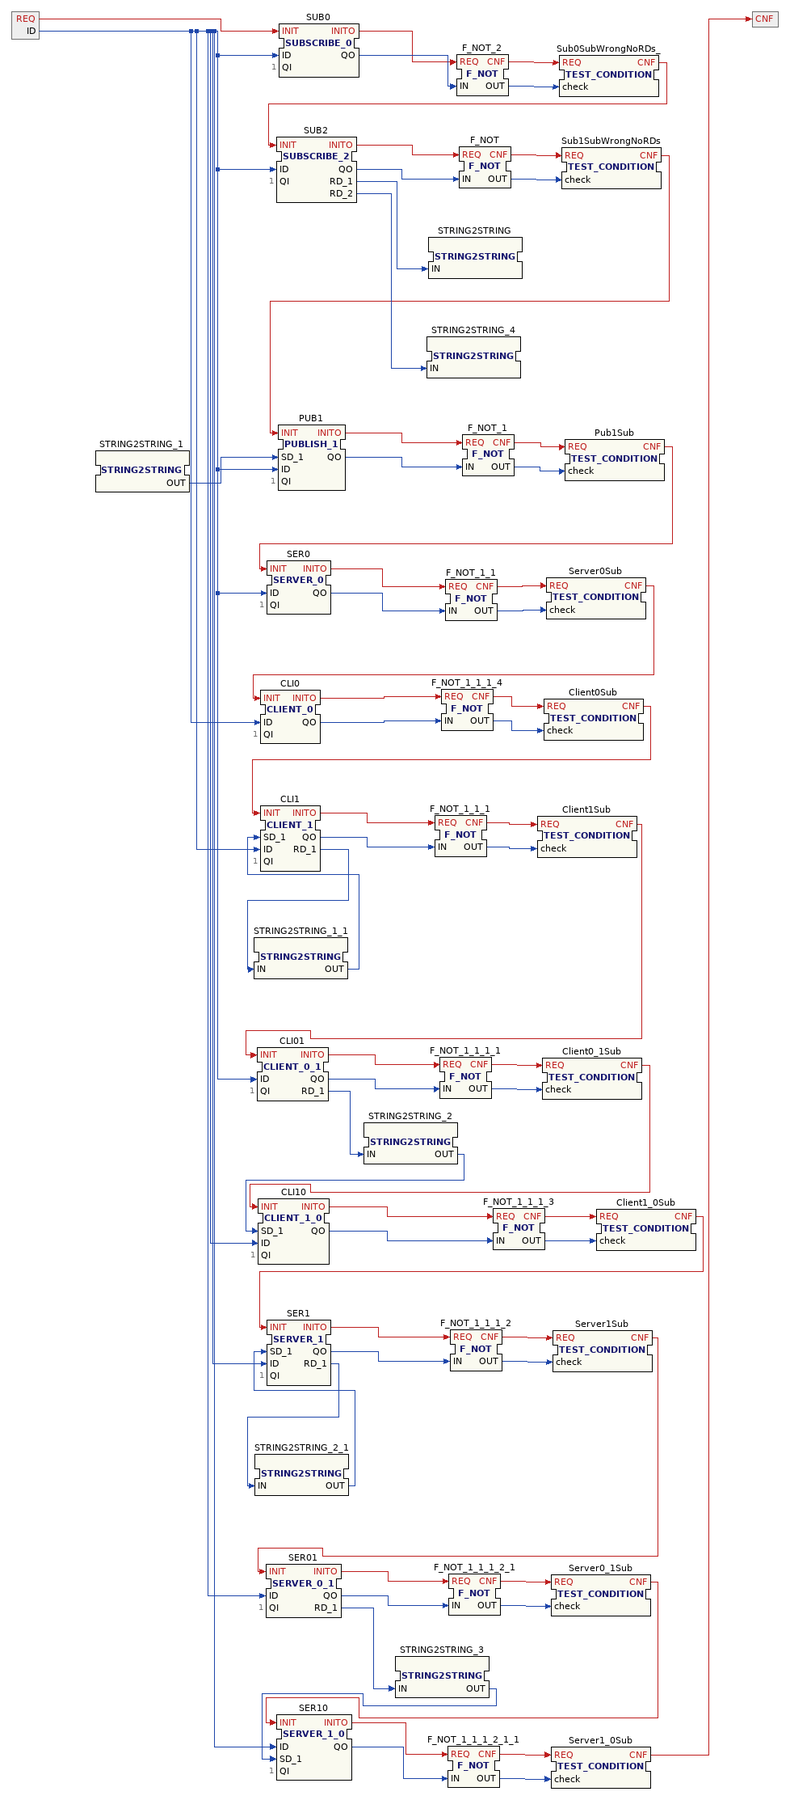
      FBS
        F_NOT_1_1_1 : F_NOT;
        Client1Sub : TEST_CONDITION;
        Pub1Sub : TEST_CONDITION;
        F_NOT_1_1 : F_NOT;
        PUB1 : PUBLISH_1(QI := 1);
        F_NOT : F_NOT;
        Server0Sub : TEST_CONDITION;
        Sub1SubWrongNoRDs : TEST_CONDITION;
        F_NOT_1 : F_NOT;
        STRING2STRING : STRING2STRING;
        SER0 : SERVER_0(QI := 1);
        STRING2STRING_1 : STRING2STRING;
        Client0_1Sub : TEST_CONDITION;
        F_NOT_1_1_1_1 : F_NOT;
        Server1Sub : TEST_CONDITION;
        F_NOT_1_1_1_2 : F_NOT;
        CLI1 : CLIENT_1(QI := 1);
        CLI01 : CLIENT_0_1(QI := 1);
        Client1_0Sub : TEST_CONDITION;
        F_NOT_1_1_1_3 : F_NOT;
        CLI10 : CLIENT_1_0(QI := 1);
        STRING2STRING_1_1 : STRING2STRING;
        F_NOT_1_1_1_4 : F_NOT;
        Client0Sub : TEST_CONDITION;
        CLI0 : CLIENT_0(QI := 1);
        SER1 : SERVER_1(QI := 1);
        F_NOT_1_1_1_2_1 : F_NOT;
        Server0_1Sub : TEST_CONDITION;
        STRING2STRING_2 : STRING2STRING;
        STRING2STRING_2_1 : STRING2STRING;
        SER01 : SERVER_0_1(QI := 1);
        STRING2STRING_3 : STRING2STRING;
        Server1_0Sub : TEST_CONDITION;
        F_NOT_1_1_1_2_1_1 : F_NOT;
        SER10 : SERVER_1_0(QI := 1);
        SUB2 : SUBSCRIBE_2(QI := 1);
        STRING2STRING_4 : STRING2STRING;
        Sub0SubWrongNoRDs_ : TEST_CONDITION;
        F_NOT_2 : F_NOT;
        SUB0 : SUBSCRIBE_0(QI := 1);
      END_FBS
      EVENT_CONNECTIONS
        F_NOT_1_1_1.CNF TO Client1Sub.REQ;
        F_NOT_1.CNF TO Pub1Sub.REQ;
        Pub1Sub.CNF TO SER0.INIT;
        SER0.INITO TO F_NOT_1_1.REQ;
        F_NOT_1_1.CNF TO Server0Sub.REQ;
        Sub1SubWrongNoRDs.CNF TO PUB1.INIT;
        PUB1.INITO TO F_NOT_1.REQ;
        F_NOT.CNF TO Sub1SubWrongNoRDs.REQ;
        F_NOT_1_1_1_1.CNF TO Client0_1Sub.REQ;
        F_NOT_1_1_1_2.CNF TO Server1Sub.REQ;
        CLI1.INITO TO F_NOT_1_1_1.REQ;
        CLI01.INITO TO F_NOT_1_1_1_1.REQ;
        CLI0.INITO TO F_NOT_1_1_1_4.REQ;
        F_NOT_1_1_1_4.CNF TO Client0Sub.REQ;
        F_NOT_1_1_1_3.CNF TO Client1_0Sub.REQ;
        CLI10.INITO TO F_NOT_1_1_1_3.REQ;
        SER1.INITO TO F_NOT_1_1_1_2.REQ;
        F_NOT_1_1_1_2_1.CNF TO Server0_1Sub.REQ;
        SER01.INITO TO F_NOT_1_1_1_2_1.REQ;
        Server0Sub.CNF TO CLI0.INIT;
        Client0Sub.CNF TO CLI1.INIT;
        Client1Sub.CNF TO CLI01.INIT;
        Client0_1Sub.CNF TO CLI10.INIT;
        Client1_0Sub.CNF TO SER1.INIT;
        Server1Sub.CNF TO SER01.INIT;
        F_NOT_1_1_1_2_1_1.CNF TO Server1_0Sub.REQ;
        Server1_0Sub.CNF TO CNF;
        Server0_1Sub.CNF TO SER10.INIT;
        SER10.INITO TO F_NOT_1_1_1_2_1_1.REQ;
        SUB2.INITO TO F_NOT.REQ;
        REQ TO SUB0.INIT;
        SUB0.INITO TO F_NOT_2.REQ;
        F_NOT_2.CNF TO Sub0SubWrongNoRDs_.REQ;
        Sub0SubWrongNoRDs_.CNF TO SUB2.INIT;
      END_CONNECTIONS
      DATA_CONNECTIONS
        F_NOT_1_1_1.OUT TO Client1Sub.check;
        F_NOT_1.OUT TO Pub1Sub.check;
        SER0.QO TO F_NOT_1_1.IN;
        F_NOT_1_1.OUT TO Server0Sub.check;
        STRING2STRING_1.OUT TO PUB1.SD_1;
        PUB1.QO TO F_NOT_1.IN;
        F_NOT.OUT TO Sub1SubWrongNoRDs.check;
        F_NOT_1_1_1_1.OUT TO Client0_1Sub.check;
        F_NOT_1_1_1_2.OUT TO Server1Sub.check;
        CLI1.QO TO F_NOT_1_1_1.IN;
        CLI01.QO TO F_NOT_1_1_1_1.IN;
        STRING2STRING_1_1.OUT TO CLI1.SD_1;
        CLI1.RD_1 TO STRING2STRING_1_1.IN;
        F_NOT_1_1_1_4.OUT TO Client0Sub.check;
        CLI0.QO TO F_NOT_1_1_1_4.IN;
        F_NOT_1_1_1_3.OUT TO Client1_0Sub.check;
        CLI10.QO TO F_NOT_1_1_1_3.IN;
        SER1.QO TO F_NOT_1_1_1_2.IN;
        F_NOT_1_1_1_2_1.OUT TO Server0_1Sub.check;
        CLI01.RD_1 TO STRING2STRING_2.IN;
        STRING2STRING_2.OUT TO CLI10.SD_1;
        STRING2STRING_2_1.OUT TO SER1.SD_1;
        SER1.RD_1 TO STRING2STRING_2_1.IN;
        SER01.QO TO F_NOT_1_1_1_2_1.IN;
        SER01.RD_1 TO STRING2STRING_3.IN;
        ID TO PUB1.ID;
        ID TO SER0.ID;
        ID TO CLI0.ID;
        ID TO CLI1.ID;
        ID TO CLI01.ID;
        ID TO CLI10.ID;
        ID TO SER01.ID;
        ID TO SER1.ID;
        F_NOT_1_1_1_2_1_1.OUT TO Server1_0Sub.check;
        ID TO SER10.ID;
        SER10.QO TO F_NOT_1_1_1_2_1_1.IN;
        STRING2STRING_3.OUT TO SER10.SD_1;
        SUB2.QO TO F_NOT.IN;
        SUB2.RD_1 TO STRING2STRING.IN;
        SUB2.RD_2 TO STRING2STRING_4.IN;
        ID TO SUB2.ID;
        ID TO SUB0.ID;
        SUB0.QO TO F_NOT_2.IN;
        F_NOT_2.OUT TO Sub0SubWrongNoRDs_.check;
      END_CONNECTIONS
    END_SUBAPPLICATION
    SUBAPPLICATION GUIDIdentifier
      EVENT_INPUT
        REQ;
      END_EVENT
      EVENT_OUTPUT
        CNF;
      END_EVENT
      VAR_INPUT
        ID : WSTRING;
      END_VAR
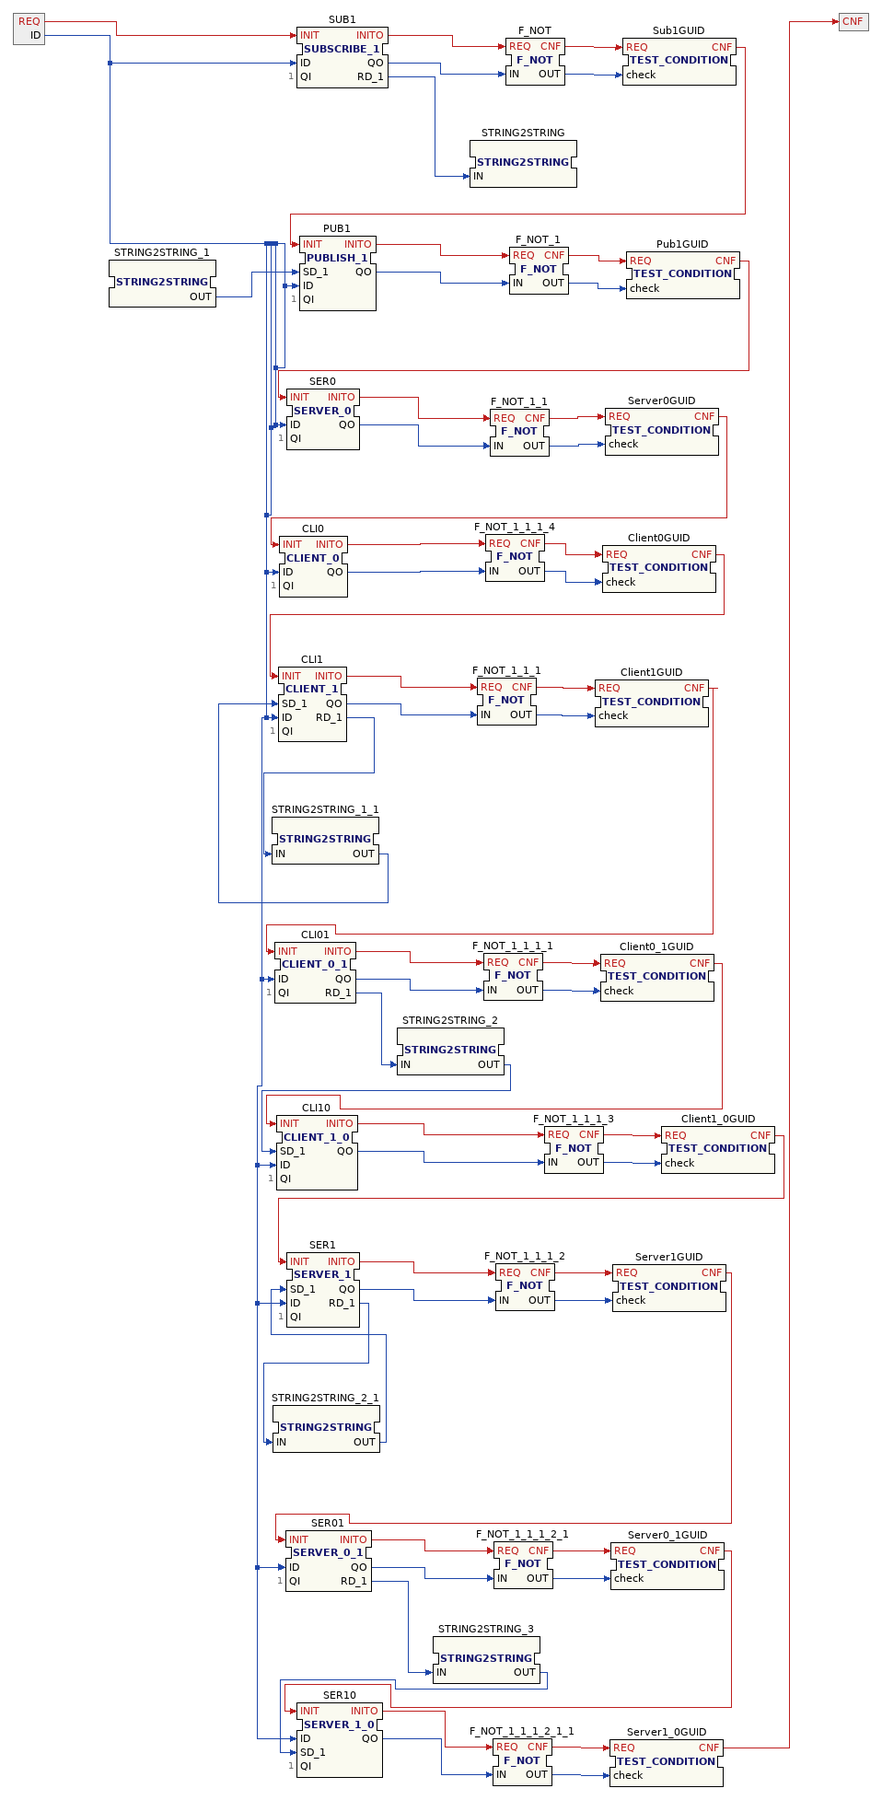
      FBS
        F_NOT_1_1_1 : F_NOT;
        Client1GUID : TEST_CONDITION;
        Pub1GUID : TEST_CONDITION;
        F_NOT_1_1 : F_NOT;
        PUB1 : PUBLISH_1(QI := 1);
        F_NOT : F_NOT;
        Server0GUID : TEST_CONDITION;
        Sub1GUID : TEST_CONDITION;
        F_NOT_1 : F_NOT;
        STRING2STRING : STRING2STRING;
        SUB1 : SUBSCRIBE_1(QI := 1);
        SER0 : SERVER_0(QI := 1);
        STRING2STRING_1 : STRING2STRING;
        Client0_1GUID : TEST_CONDITION;
        F_NOT_1_1_1_1 : F_NOT;
        Server1GUID : TEST_CONDITION;
        F_NOT_1_1_1_2 : F_NOT;
        CLI1 : CLIENT_1(QI := 1);
        CLI01 : CLIENT_0_1(QI := 1);
        Client1_0GUID : TEST_CONDITION;
        F_NOT_1_1_1_3 : F_NOT;
        CLI10 : CLIENT_1_0(QI := 1);
        STRING2STRING_1_1 : STRING2STRING;
        F_NOT_1_1_1_4 : F_NOT;
        Client0GUID : TEST_CONDITION;
        CLI0 : CLIENT_0(QI := 1);
        SER1 : SERVER_1(QI := 1);
        F_NOT_1_1_1_2_1 : F_NOT;
        Server0_1GUID : TEST_CONDITION;
        STRING2STRING_2 : STRING2STRING;
        STRING2STRING_2_1 : STRING2STRING;
        SER01 : SERVER_0_1(QI := 1);
        STRING2STRING_3 : STRING2STRING;
        Server1_0GUID : TEST_CONDITION;
        F_NOT_1_1_1_2_1_1 : F_NOT;
        SER10 : SERVER_1_0(QI := 1);
      END_FBS
      EVENT_CONNECTIONS
        F_NOT_1_1_1.CNF TO Client1GUID.REQ;
        F_NOT_1.CNF TO Pub1GUID.REQ;
        Pub1GUID.CNF TO SER0.INIT;
        SER0.INITO TO F_NOT_1_1.REQ;
        F_NOT_1_1.CNF TO Server0GUID.REQ;
        Sub1GUID.CNF TO PUB1.INIT;
        PUB1.INITO TO F_NOT_1.REQ;
        SUB1.INITO TO F_NOT.REQ;
        F_NOT.CNF TO Sub1GUID.REQ;
        REQ TO SUB1.INIT;
        F_NOT_1_1_1_1.CNF TO Client0_1GUID.REQ;
        F_NOT_1_1_1_2.CNF TO Server1GUID.REQ;
        CLI1.INITO TO F_NOT_1_1_1.REQ;
        CLI01.INITO TO F_NOT_1_1_1_1.REQ;
        CLI0.INITO TO F_NOT_1_1_1_4.REQ;
        F_NOT_1_1_1_4.CNF TO Client0GUID.REQ;
        F_NOT_1_1_1_3.CNF TO Client1_0GUID.REQ;
        CLI10.INITO TO F_NOT_1_1_1_3.REQ;
        SER1.INITO TO F_NOT_1_1_1_2.REQ;
        F_NOT_1_1_1_2_1.CNF TO Server0_1GUID.REQ;
        SER01.INITO TO F_NOT_1_1_1_2_1.REQ;
        Server0GUID.CNF TO CLI0.INIT;
        Client0GUID.CNF TO CLI1.INIT;
        Client1GUID.CNF TO CLI01.INIT;
        Client0_1GUID.CNF TO CLI10.INIT;
        Client1_0GUID.CNF TO SER1.INIT;
        Server1GUID.CNF TO SER01.INIT;
        F_NOT_1_1_1_2_1_1.CNF TO Server1_0GUID.REQ;
        Server1_0GUID.CNF TO CNF;
        Server0_1GUID.CNF TO SER10.INIT;
        SER10.INITO TO F_NOT_1_1_1_2_1_1.REQ;
      END_CONNECTIONS
      DATA_CONNECTIONS
        F_NOT_1_1_1.OUT TO Client1GUID.check;
        F_NOT_1.OUT TO Pub1GUID.check;
        SER0.QO TO F_NOT_1_1.IN;
        F_NOT_1_1.OUT TO Server0GUID.check;
        STRING2STRING_1.OUT TO PUB1.SD_1;
        PUB1.QO TO F_NOT_1.IN;
        SUB1.QO TO F_NOT.IN;
        F_NOT.OUT TO Sub1GUID.check;
        SUB1.RD_1 TO STRING2STRING.IN;
        F_NOT_1_1_1_1.OUT TO Client0_1GUID.check;
        F_NOT_1_1_1_2.OUT TO Server1GUID.check;
        CLI1.QO TO F_NOT_1_1_1.IN;
        CLI01.QO TO F_NOT_1_1_1_1.IN;
        STRING2STRING_1_1.OUT TO CLI1.SD_1;
        CLI1.RD_1 TO STRING2STRING_1_1.IN;
        F_NOT_1_1_1_4.OUT TO Client0GUID.check;
        CLI0.QO TO F_NOT_1_1_1_4.IN;
        F_NOT_1_1_1_3.OUT TO Client1_0GUID.check;
        CLI10.QO TO F_NOT_1_1_1_3.IN;
        SER1.QO TO F_NOT_1_1_1_2.IN;
        F_NOT_1_1_1_2_1.OUT TO Server0_1GUID.check;
        CLI01.RD_1 TO STRING2STRING_2.IN;
        STRING2STRING_2.OUT TO CLI10.SD_1;
        STRING2STRING_2_1.OUT TO SER1.SD_1;
        SER1.RD_1 TO STRING2STRING_2_1.IN;
        SER01.QO TO F_NOT_1_1_1_2_1.IN;
        SER01.RD_1 TO STRING2STRING_3.IN;
        ID TO SUB1.ID;
        ID TO PUB1.ID;
        ID TO SER0.ID;
        ID TO CLI0.ID;
        ID TO CLI1.ID;
        ID TO CLI01.ID;
        ID TO CLI10.ID;
        ID TO SER01.ID;
        ID TO SER1.ID;
        F_NOT_1_1_1_2_1_1.OUT TO Server1_0GUID.check;
        ID TO SER10.ID;
        SER10.QO TO F_NOT_1_1_1_2_1_1.IN;
        STRING2STRING_3.OUT TO SER10.SD_1;
      END_CONNECTIONS
    END_SUBAPPLICATION
    EVENT_CONNECTIONS
      NoSemicolon.CNF TO W2W_1.REQ;
      W2W_1.CNF TO emptyAction.REQ;
      emptyAction.CNF TO W2W_1_1.REQ;
      W2W_1_1.CNF TO NoExistingAction.REQ;
      W2W_1_1_1.CNF TO wrongPair.REQ;
      W2W_1_1_2.CNF TO wrongNodeId.REQ;
      W2W_1_1_3.CNF TO UnknownIdentifier.REQ;
      W2W_1_1_4.CNF TO WrongIdentifier.REQ;
      UnknownIdentifier.CNF TO W2W_1_1_4.REQ;
      wrongNodeId.CNF TO W2W_1_1_3.REQ;
      wrongPair.CNF TO W2W_1_1_2.REQ;
      NoExistingAction.CNF TO W2W_1_1_1.REQ;
      W2W.CNF TO NoSemicolon.REQ;
      W2W_1_1_4_1.CNF TO LocalWithoutBrowseName.REQ;
      W2W_1_1_4_2.CNF TO RemoteWithoutBrowseNameNorNodeId.REQ;
      WrongIdentifier.CNF TO W2W_1_1_4_1.REQ;
      LocalWithoutBrowseName.CNF TO W2W_1_1_4_2.REQ;
      W2W_1_1_4_2_1.CNF TO LocalRead.REQ;
      RemoteWithoutBrowseNameNorNodeId.CNF TO W2W_1_1_4_2_1.REQ;
      W2W_1_1_4_2_1_1.CNF TO RemoteRead.REQ;
      LocalRead.CNF TO W2W_1_1_4_2_1_1.REQ;
      RemoteRead.CNF TO W2W_1_1_4_2_1_1_1.REQ;
      LocalWrite.CNF TO W2W_1_1_4_2_1_1_1_1.REQ;
      W2W_1_1_4_2_1_1_1_1.CNF TO RemoteWrite.REQ;
      W2W_1_1_4_2_1_1_1.CNF TO LocalWrite.REQ;
      W2W_1_1_4_2_1_1_1_1_1.CNF TO CreateMethod.REQ;
      RemoteWrite.CNF TO W2W_1_1_4_2_1_1_1_1_1.REQ;
      W2W_1_1_4_2_1_1_1_1_1_1.CNF TO CallMethod.REQ;
      CreateMethod.CNF TO W2W_1_1_4_2_1_1_1_1_1_1.REQ;
      W2W_1_1_4_2_1_1_1_1_1_1_1.CNF TO Subscribe.REQ;
      CallMethod.CNF TO W2W_1_1_4_2_1_1_1_1_1_1_1.REQ;
      Subscribe.CNF TO STEST_END.REQ;
      W2W_2.CNF TO GUIDIdentifier.REQ;
      GUIDIdentifier.CNF TO W2W.REQ;
    END_CONNECTIONS
    DATA_CONNECTIONS
      W2W_1_1_4.OUT TO WrongIdentifier.ID;
      W2W_1_1_3.OUT TO UnknownIdentifier.ID;
      W2W_1_1_2.OUT TO wrongNodeId.ID;
      W2W_1_1_1.OUT TO wrongPair.ID;
      W2W_1_1.OUT TO NoExistingAction.ID;
      W2W_1.OUT TO emptyAction.ID;
      W2W.OUT TO NoSemicolon.ID;
      W2W_1_1_4_1.OUT TO LocalWithoutBrowseName.ID;
      W2W_1_1_4_2.OUT TO RemoteWithoutBrowseNameNorNodeId.ID;
      W2W_1_1_4_1.OUT TO LocalWithoutBrowseName.ID;
      W2W_1_1_4_2.OUT TO RemoteWithoutBrowseNameNorNodeId.ID;
      W2W_1_1_4_2_1.OUT TO LocalRead.ID;
      W2W_1_1_4_2_1_1.OUT TO RemoteRead.ID;
      W2W_1_1_4_2_1_1.OUT TO RemoteRead.ID;
      W2W_1_1_4_2_1.OUT TO LocalRead.ID;
      W2W_1_1_4_2_1_1_1_1.OUT TO RemoteWrite.ID;
      W2W_1_1_4_2_1_1_1.OUT TO LocalWrite.ID;
      W2W_1_1_4_2_1_1_1_1.OUT TO RemoteWrite.ID;
      W2W_1_1_4_2_1_1_1.OUT TO LocalWrite.ID;
      W2W_1_1_4_2_1_1_1_1_1.OUT TO CreateMethod.ID;
      W2W_1_1_4_2_1_1_1_1_1_1.OUT TO CallMethod.ID;
      W2W_1_1_4_2_1_1_1_1_1_1.OUT TO CallMethod.ID;
      W2W_1_1_4_2_1_1_1_1_1_1_1.OUT TO Subscribe.ID;
      W2W_1_1_4_2_1_1_1_1_1_1_1.OUT TO Subscribe.ID;
      W2W_2.OUT TO GUIDIdentifier.ID;
      W2W_2.OUT TO GUIDIdentifier.ID;
    END_CONNECTIONS
  END_APPLICATION
  APPLICATION OpcUaLocalWorking
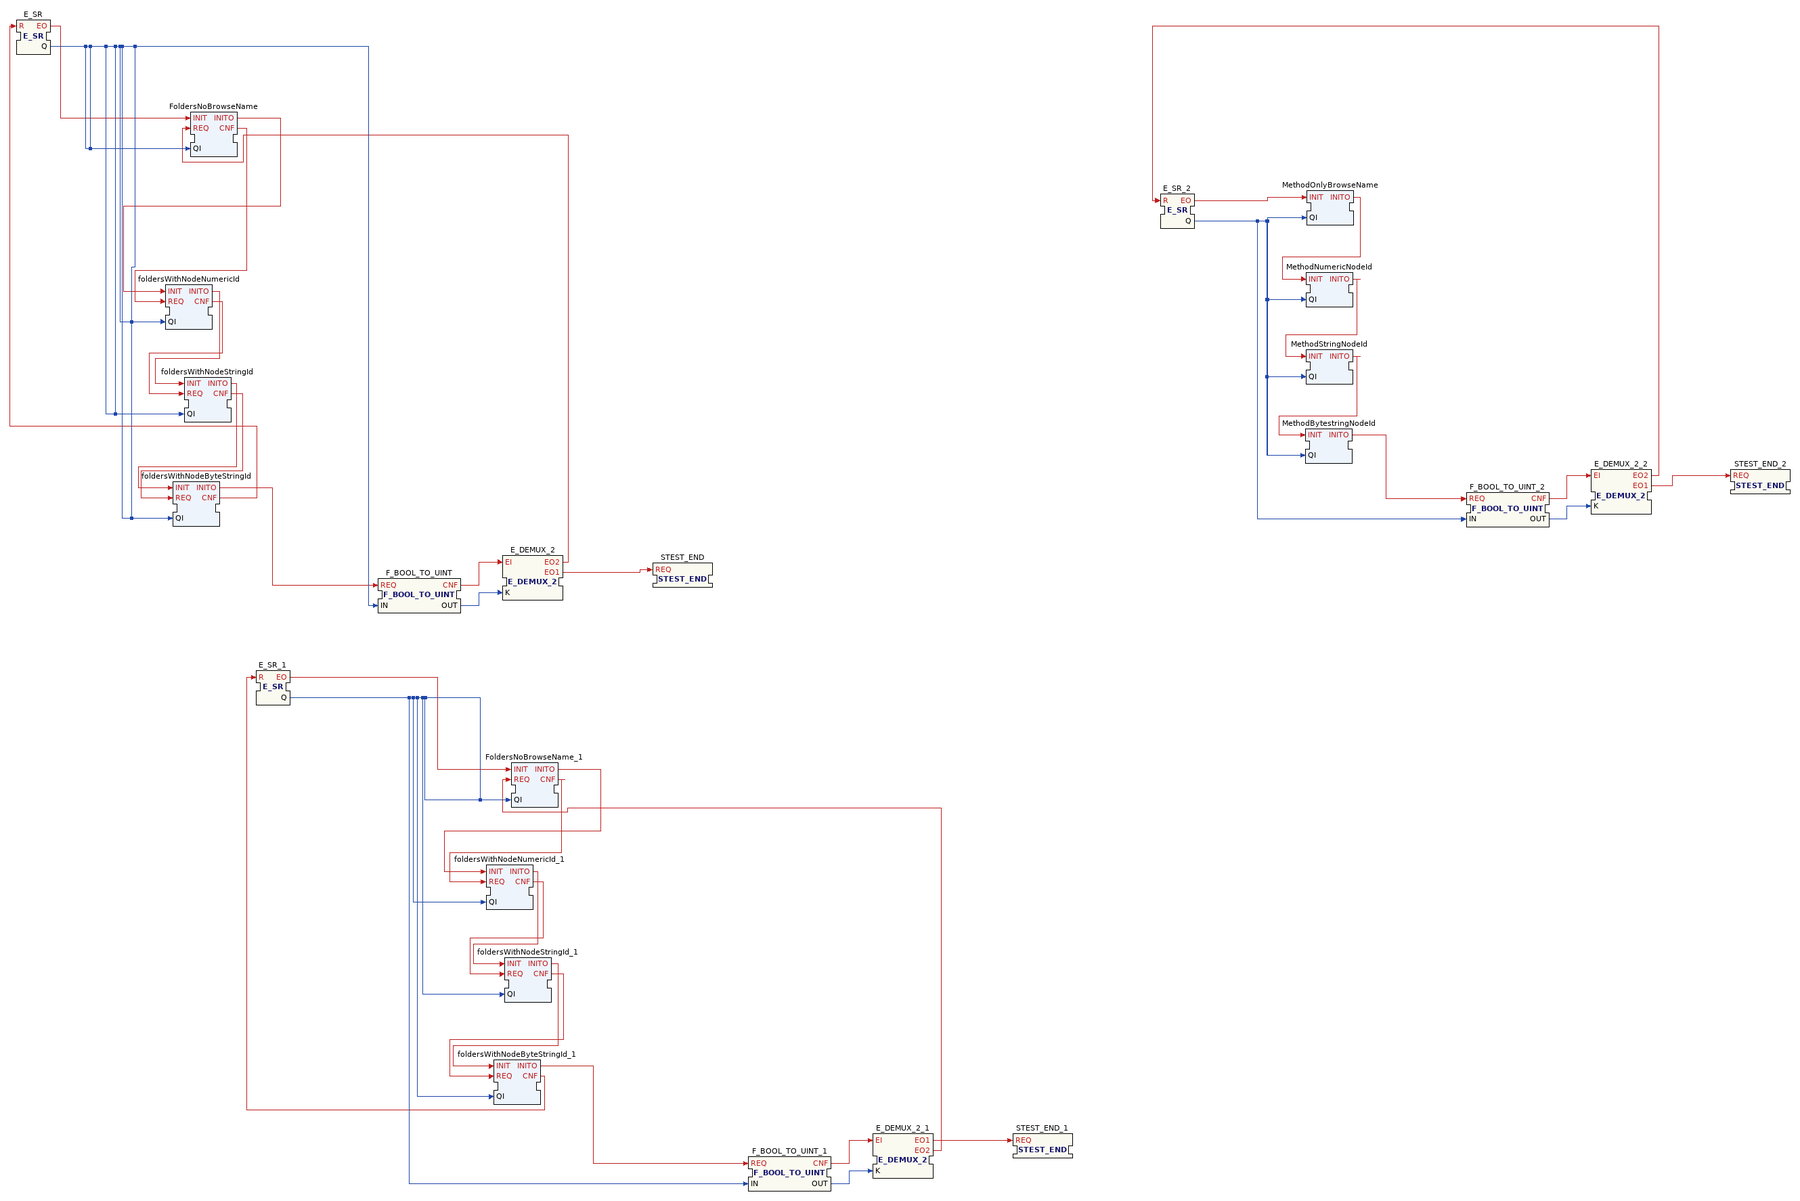
    FBS
      E_SR : E_SR;
      E_DEMUX_2 : E_DEMUX_2;
      STEST_END : STEST_END;
      F_BOOL_TO_UINT : F_BOOL_TO_UINT;
      E_SR_1 : E_SR;
      F_BOOL_TO_UINT_1 : F_BOOL_TO_UINT;
      STEST_END_1 : STEST_END;
      E_DEMUX_2_1 : E_DEMUX_2;
      E_SR_2 : E_SR;
      STEST_END_2 : STEST_END;
      F_BOOL_TO_UINT_2 : F_BOOL_TO_UINT;
      E_DEMUX_2_2 : E_DEMUX_2;
    END_FBS
    SUBAPPLICATION FoldersNoBrowseName
      EVENT_INPUT
        INIT;
        REQ;
      END_EVENT
      EVENT_OUTPUT
        INITO;
        CNF;
      END_EVENT
      VAR_INPUT
        QI : BOOL;
      END_VAR
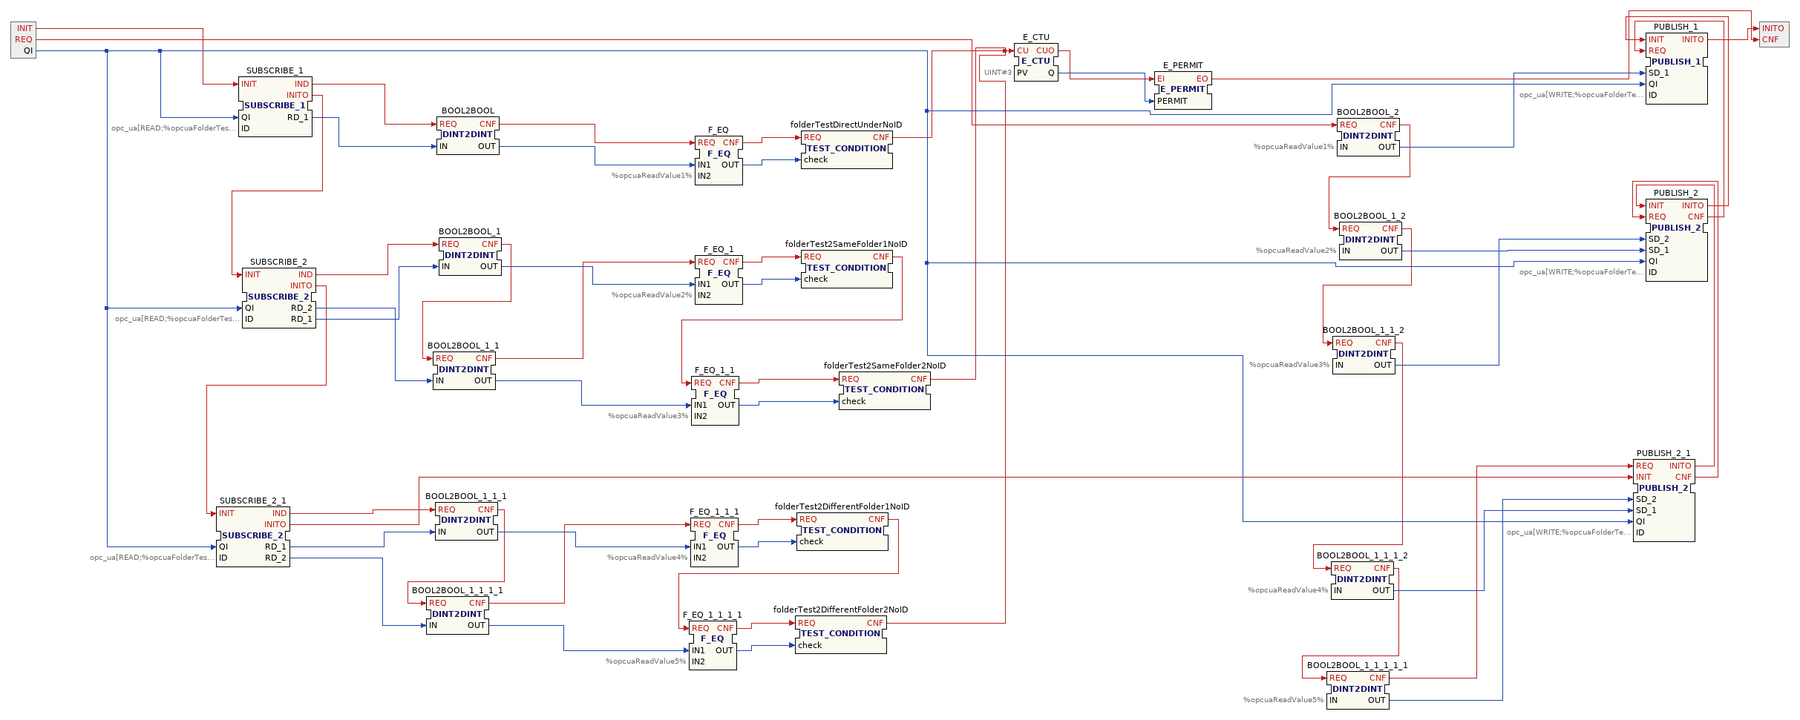
      FBS
        F_EQ_1_1_1 : F_EQ(IN2 := %opcuaReadValue4%);
        BOOL2BOOL_1_1 : DINT2DINT;
        SUBSCRIBE_2 : SUBSCRIBE_2(ID := opc_ua[READ;%opcuaFolderTestOnlyBroseName2%]);
        folderTestDirectUnderNoID : TEST_CONDITION;
        BOOL2BOOL_1 : DINT2DINT;
        BOOL2BOOL_1_1_1 : DINT2DINT;
        BOOL2BOOL_1_1_1_1_1 : DINT2DINT(IN := %opcuaReadValue5%);
        SUBSCRIBE_2_1 : SUBSCRIBE_2(ID := opc_ua[READ;%opcuaFolderTestOnlyBroseName3%]);
        SUBSCRIBE_1 : SUBSCRIBE_1(ID := opc_ua[READ;%opcuaFolderTestOnlyBroseName1%]);
        BOOL2BOOL_1_1_1_2 : DINT2DINT(IN := %opcuaReadValue4%);
        PUBLISH_2_1 : PUBLISH_2(ID := opc_ua[WRITE;%opcuaFolderTestOnlyBroseName3%]);
        BOOL2BOOL : DINT2DINT;
        F_EQ_1_1_1_1 : F_EQ(IN2 := %opcuaReadValue5%);
        BOOL2BOOL_1_1_2 : DINT2DINT(IN := %opcuaReadValue3%);
        E_PERMIT : E_PERMIT;
        folderTest2SameFolder1NoID : TEST_CONDITION;
        BOOL2BOOL_1_2 : DINT2DINT(IN := %opcuaReadValue2%);
        folderTest2DifferentFolder2NoID : TEST_CONDITION;
        BOOL2BOOL_1_1_1_1 : DINT2DINT;
        PUBLISH_1 : PUBLISH_1(ID := opc_ua[WRITE;%opcuaFolderTestOnlyBroseName1%]);
        BOOL2BOOL_2 : DINT2DINT(IN := %opcuaReadValue1%);
        F_EQ_1 : F_EQ(IN2 := %opcuaReadValue2%);
        E_CTU : E_CTU(PV := UINT#3);
        F_EQ : F_EQ(IN2 := %opcuaReadValue1%);
        PUBLISH_2 : PUBLISH_2(ID := opc_ua[WRITE;%opcuaFolderTestOnlyBroseName2%]);
        folderTest2SameFolder2NoID : TEST_CONDITION;
        folderTest2DifferentFolder1NoID : TEST_CONDITION;
        F_EQ_1_1 : F_EQ(IN2 := %opcuaReadValue3%);
      END_FBS
      EVENT_CONNECTIONS
        BOOL2BOOL_1_1_1_1.CNF TO F_EQ_1_1_1.REQ;
        F_EQ_1_1_1.CNF TO folderTest2DifferentFolder1NoID.REQ;
        BOOL2BOOL_1.CNF TO BOOL2BOOL_1_1.REQ;
        BOOL2BOOL_1_1.CNF TO F_EQ_1.REQ;
        SUBSCRIBE_2.IND TO BOOL2BOOL_1.REQ;
        F_EQ.CNF TO folderTestDirectUnderNoID.REQ;
        folderTestDirectUnderNoID.CNF TO E_CTU.CU;
        SUBSCRIBE_2_1.IND TO BOOL2BOOL_1_1_1.REQ;
        BOOL2BOOL_1_1_1.CNF TO BOOL2BOOL_1_1_1_1.REQ;
        BOOL2BOOL_1_1_1_2.CNF TO BOOL2BOOL_1_1_1_1_1.REQ;
        SUBSCRIBE_1.IND TO BOOL2BOOL.REQ;
        BOOL2BOOL_1_1_2.CNF TO BOOL2BOOL_1_1_1_2.REQ;
        PUBLISH_2_1.INITO TO PUBLISH_2.INIT;
        PUBLISH_2_1.CNF TO PUBLISH_2.REQ;
        BOOL2BOOL.CNF TO F_EQ.REQ;
        folderTest2DifferentFolder1NoID.CNF TO F_EQ_1_1_1_1.REQ;
        F_EQ_1_1_1_1.CNF TO folderTest2DifferentFolder2NoID.REQ;
        BOOL2BOOL_1_2.CNF TO BOOL2BOOL_1_1_2.REQ;
        E_CTU.CUO TO E_PERMIT.EI;
        F_EQ_1.CNF TO folderTest2SameFolder1NoID.REQ;
        folderTest2SameFolder1NoID.CNF TO F_EQ_1_1.REQ;
        BOOL2BOOL_2.CNF TO BOOL2BOOL_1_2.REQ;
        folderTest2DifferentFolder2NoID.CNF TO E_CTU.CU;
        PUBLISH_2.INITO TO PUBLISH_1.INIT;
        PUBLISH_2.CNF TO PUBLISH_1.REQ;
        folderTest2SameFolder2NoID.CNF TO E_CTU.CU;
        F_EQ_1_1.CNF TO folderTest2SameFolder2NoID.REQ;
        PUBLISH_1.INITO TO INITO;
        E_PERMIT.EO TO CNF;
        REQ TO BOOL2BOOL_2.REQ;
        INIT TO SUBSCRIBE_1.INIT;
        BOOL2BOOL_1_1_1_1_1.CNF TO PUBLISH_2_1.REQ;
        SUBSCRIBE_1.INITO TO SUBSCRIBE_2.INIT;
        SUBSCRIBE_2.INITO TO SUBSCRIBE_2_1.INIT;
        SUBSCRIBE_2_1.INITO TO PUBLISH_2_1.INIT;
      END_CONNECTIONS
      DATA_CONNECTIONS
        BOOL2BOOL_1_1_1.OUT TO F_EQ_1_1_1.IN1;
        F_EQ_1_1_1.OUT TO folderTest2DifferentFolder1NoID.check;
        SUBSCRIBE_2.RD_2 TO BOOL2BOOL_1_1.IN;
        BOOL2BOOL_1_1.OUT TO F_EQ_1_1.IN1;
        SUBSCRIBE_2.RD_1 TO BOOL2BOOL_1.IN;
        F_EQ.OUT TO folderTestDirectUnderNoID.check;
        BOOL2BOOL_1.OUT TO F_EQ_1.IN1;
        SUBSCRIBE_2_1.RD_1 TO BOOL2BOOL_1_1_1.IN;
        BOOL2BOOL_1_1_1_1_1.OUT TO PUBLISH_2_1.SD_2;
        SUBSCRIBE_2_1.RD_2 TO BOOL2BOOL_1_1_1_1.IN;
        SUBSCRIBE_1.RD_1 TO BOOL2BOOL.IN;
        BOOL2BOOL_1_1_1_2.OUT TO PUBLISH_2_1.SD_1;
        BOOL2BOOL.OUT TO F_EQ.IN1;
        BOOL2BOOL_1_1_1_1.OUT TO F_EQ_1_1_1_1.IN1;
        F_EQ_1_1_1_1.OUT TO folderTest2DifferentFolder2NoID.check;
        BOOL2BOOL_1_1_2.OUT TO PUBLISH_2.SD_2;
        E_CTU.Q TO E_PERMIT.PERMIT;
        F_EQ_1.OUT TO folderTest2SameFolder1NoID.check;
        BOOL2BOOL_1_2.OUT TO PUBLISH_2.SD_1;
        BOOL2BOOL_2.OUT TO PUBLISH_1.SD_1;
        F_EQ_1_1.OUT TO folderTest2SameFolder2NoID.check;
        QI TO SUBSCRIBE_2.QI;
        QI TO SUBSCRIBE_2_1.QI;
        QI TO SUBSCRIBE_1.QI;
        QI TO PUBLISH_2_1.QI;
        QI TO PUBLISH_1.QI;
        QI TO PUBLISH_2.QI;
      END_CONNECTIONS
    END_SUBAPPLICATION
    SUBAPPLICATION foldersWithNodeNumericId
      EVENT_INPUT
        INIT;
        REQ;
      END_EVENT
      EVENT_OUTPUT
        INITO;
        CNF;
      END_EVENT
      VAR_INPUT
        QI : BOOL;
      END_VAR
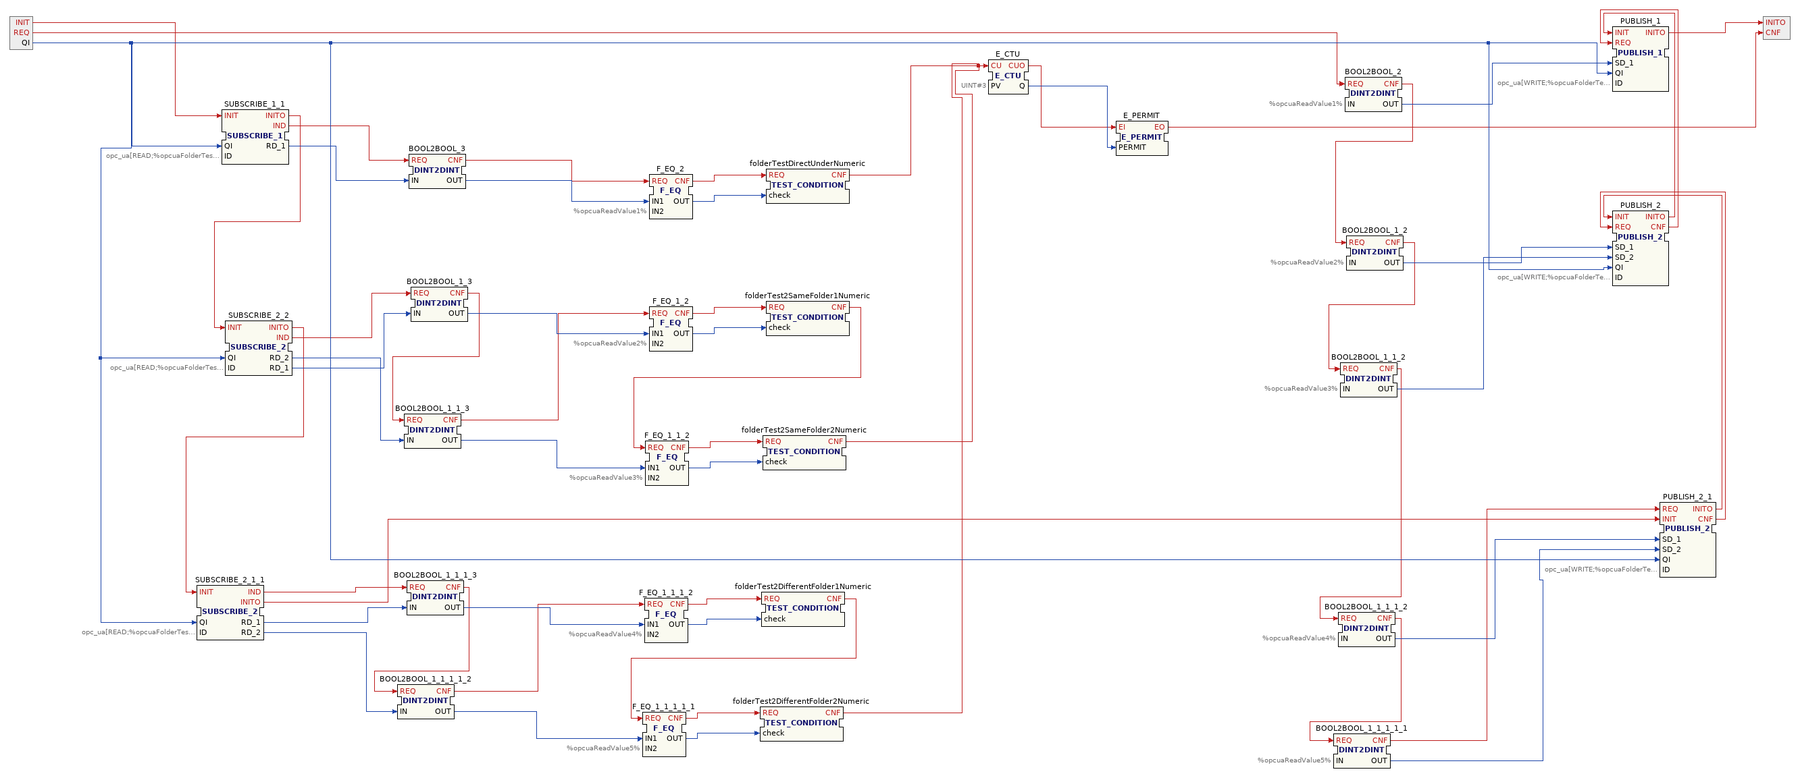
      FBS
        BOOL2BOOL_1_2 : DINT2DINT(IN := %opcuaReadValue2%);
        F_EQ_1_2 : F_EQ(IN2 := %opcuaReadValue2%);
        F_EQ_2 : F_EQ(IN2 := %opcuaReadValue1%);
        PUBLISH_2 : PUBLISH_2(ID := opc_ua[WRITE;%opcuaFolderTestWithNodeIdNumeric2%]);
        folderTest2SameFolder2Numeric : TEST_CONDITION;
        folderTest2DifferentFolder2Numeric : TEST_CONDITION;
        E_PERMIT : E_PERMIT;
        F_EQ_1_1_1_2 : F_EQ(IN2 := %opcuaReadValue4%);
        F_EQ_1_1_1_1_1 : F_EQ(IN2 := %opcuaReadValue5%);
        PUBLISH_2_1 : PUBLISH_2(ID := opc_ua[WRITE;%opcuaFolderTestWithNodeIdNumeric3%]);
        BOOL2BOOL_1_1_2 : DINT2DINT(IN := %opcuaReadValue3%);
        BOOL2BOOL_1_1_1_1_1 : DINT2DINT(IN := %opcuaReadValue5%);
        BOOL2BOOL_2 : DINT2DINT(IN := %opcuaReadValue1%);
        BOOL2BOOL_1_1_1_3 : DINT2DINT;
        BOOL2BOOL_1_1_3 : DINT2DINT;
        BOOL2BOOL_1_1_1_2 : DINT2DINT(IN := %opcuaReadValue4%);
        F_EQ_1_1_2 : F_EQ(IN2 := %opcuaReadValue3%);
        PUBLISH_1 : PUBLISH_1(ID := opc_ua[WRITE;%opcuaFolderTestWithNodeIdNumeric1%]);
        E_CTU : E_CTU(PV := UINT#3);
        folderTest2SameFolder1Numeric : TEST_CONDITION;
        SUBSCRIBE_1_1 : SUBSCRIBE_1(ID := opc_ua[READ;%opcuaFolderTestWithNodeIdNumeric1%]);
        BOOL2BOOL_1_1_1_1_2 : DINT2DINT;
        folderTest2DifferentFolder1Numeric : TEST_CONDITION;
        SUBSCRIBE_2_2 : SUBSCRIBE_2(ID := opc_ua[READ;%opcuaFolderTestWithNodeIdNumeric2%]);
        SUBSCRIBE_2_1_1 : SUBSCRIBE_2(ID := opc_ua[READ;%opcuaFolderTestWithNodeIdNumeric3%]);
        BOOL2BOOL_1_3 : DINT2DINT;
        BOOL2BOOL_3 : DINT2DINT;
        folderTestDirectUnderNumeric : TEST_CONDITION;
      END_FBS
      EVENT_CONNECTIONS
        BOOL2BOOL_2.CNF TO BOOL2BOOL_1_2.REQ;
        BOOL2BOOL_1_2.CNF TO BOOL2BOOL_1_1_2.REQ;
        BOOL2BOOL_1_1_3.CNF TO F_EQ_1_2.REQ;
        F_EQ_1_2.CNF TO folderTest2SameFolder1Numeric.REQ;
        BOOL2BOOL_3.CNF TO F_EQ_2.REQ;
        F_EQ_2.CNF TO folderTestDirectUnderNumeric.REQ;
        PUBLISH_2_1.INITO TO PUBLISH_2.INIT;
        PUBLISH_2_1.CNF TO PUBLISH_2.REQ;
        PUBLISH_2.INITO TO PUBLISH_1.INIT;
        PUBLISH_2.CNF TO PUBLISH_1.REQ;
        F_EQ_1_1_2.CNF TO folderTest2SameFolder2Numeric.REQ;
        F_EQ_1_1_1_1_1.CNF TO folderTest2DifferentFolder2Numeric.REQ;
        E_CTU.CUO TO E_PERMIT.EI;
        BOOL2BOOL_1_1_1_1_2.CNF TO F_EQ_1_1_1_2.REQ;
        F_EQ_1_1_1_2.CNF TO folderTest2DifferentFolder1Numeric.REQ;
        folderTest2DifferentFolder1Numeric.CNF TO F_EQ_1_1_1_1_1.REQ;
        BOOL2BOOL_1_1_1_1_1.CNF TO PUBLISH_2_1.REQ;
        BOOL2BOOL_1_1_2.CNF TO BOOL2BOOL_1_1_1_2.REQ;
        BOOL2BOOL_1_1_1_2.CNF TO BOOL2BOOL_1_1_1_1_1.REQ;
        SUBSCRIBE_2_1_1.IND TO BOOL2BOOL_1_1_1_3.REQ;
        BOOL2BOOL_1_1_1_3.CNF TO BOOL2BOOL_1_1_1_1_2.REQ;
        BOOL2BOOL_1_3.CNF TO BOOL2BOOL_1_1_3.REQ;
        folderTest2SameFolder1Numeric.CNF TO F_EQ_1_1_2.REQ;
        SUBSCRIBE_1_1.INITO TO SUBSCRIBE_2_2.INIT;
        SUBSCRIBE_1_1.IND TO BOOL2BOOL_3.REQ;
        SUBSCRIBE_2_2.INITO TO SUBSCRIBE_2_1_1.INIT;
        SUBSCRIBE_2_2.IND TO BOOL2BOOL_1_3.REQ;
        PUBLISH_1.INITO TO INITO;
        INIT TO SUBSCRIBE_1_1.INIT;
        folderTestDirectUnderNumeric.CNF TO E_CTU.CU;
        folderTest2SameFolder2Numeric.CNF TO E_CTU.CU;
        folderTest2DifferentFolder2Numeric.CNF TO E_CTU.CU;
        E_PERMIT.EO TO CNF;
        REQ TO BOOL2BOOL_2.REQ;
        SUBSCRIBE_2_1_1.INITO TO PUBLISH_2_1.INIT;
      END_CONNECTIONS
      DATA_CONNECTIONS
        BOOL2BOOL_1_2.OUT TO PUBLISH_2.SD_1;
        BOOL2BOOL_1_3.OUT TO F_EQ_1_2.IN1;
        F_EQ_1_2.OUT TO folderTest2SameFolder1Numeric.check;
        BOOL2BOOL_3.OUT TO F_EQ_2.IN1;
        F_EQ_2.OUT TO folderTestDirectUnderNumeric.check;
        BOOL2BOOL_1_1_2.OUT TO PUBLISH_2.SD_2;
        F_EQ_1_1_2.OUT TO folderTest2SameFolder2Numeric.check;
        F_EQ_1_1_1_1_1.OUT TO folderTest2DifferentFolder2Numeric.check;
        E_CTU.Q TO E_PERMIT.PERMIT;
        BOOL2BOOL_1_1_1_3.OUT TO F_EQ_1_1_1_2.IN1;
        F_EQ_1_1_1_2.OUT TO folderTest2DifferentFolder1Numeric.check;
        BOOL2BOOL_1_1_1_1_2.OUT TO F_EQ_1_1_1_1_1.IN1;
        BOOL2BOOL_1_1_1_2.OUT TO PUBLISH_2_1.SD_1;
        BOOL2BOOL_1_1_1_1_1.OUT TO PUBLISH_2_1.SD_2;
        BOOL2BOOL_2.OUT TO PUBLISH_1.SD_1;
        SUBSCRIBE_2_1_1.RD_1 TO BOOL2BOOL_1_1_1_3.IN;
        SUBSCRIBE_2_2.RD_2 TO BOOL2BOOL_1_1_3.IN;
        BOOL2BOOL_1_1_3.OUT TO F_EQ_1_1_2.IN1;
        SUBSCRIBE_1_1.RD_1 TO BOOL2BOOL_3.IN;
        SUBSCRIBE_2_1_1.RD_2 TO BOOL2BOOL_1_1_1_1_2.IN;
        SUBSCRIBE_2_2.RD_1 TO BOOL2BOOL_1_3.IN;
        QI TO SUBSCRIBE_1_1.QI;
        QI TO SUBSCRIBE_2_2.QI;
        QI TO SUBSCRIBE_2_1_1.QI;
        QI TO PUBLISH_1.QI;
        QI TO PUBLISH_2.QI;
        QI TO PUBLISH_2_1.QI;
      END_CONNECTIONS
    END_SUBAPPLICATION
    SUBAPPLICATION foldersWithNodeByteStringId
      EVENT_INPUT
        INIT;
        REQ;
      END_EVENT
      EVENT_OUTPUT
        INITO;
        CNF;
      END_EVENT
      VAR_INPUT
        QI : BOOL;
      END_VAR
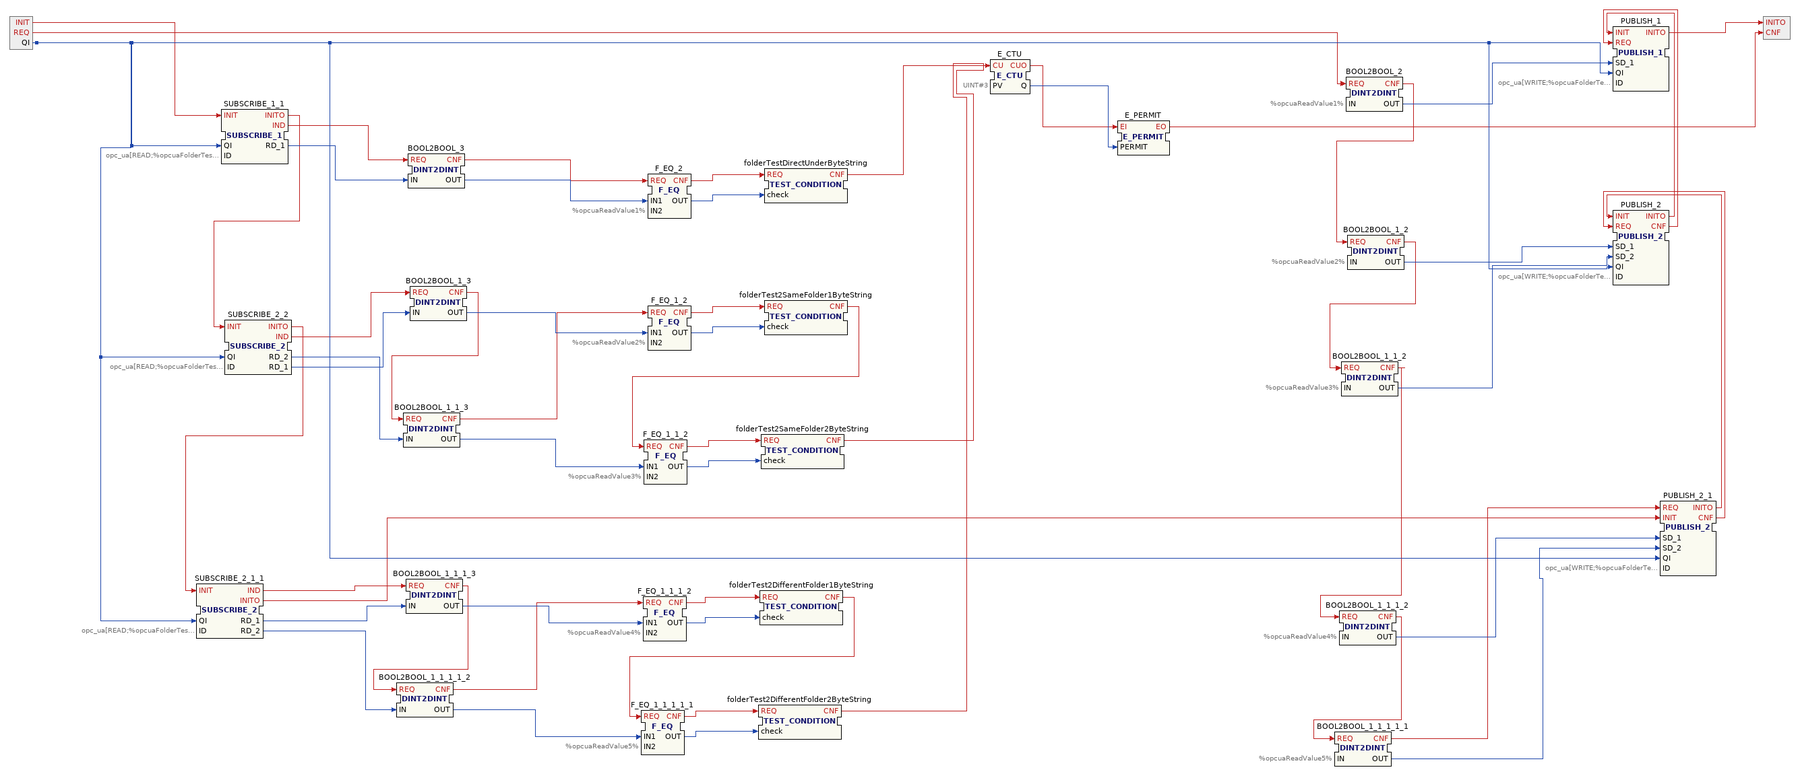
      FBS
        BOOL2BOOL_1_2 : DINT2DINT(IN := %opcuaReadValue2%);
        F_EQ_1_2 : F_EQ(IN2 := %opcuaReadValue2%);
        F_EQ_2 : F_EQ(IN2 := %opcuaReadValue1%);
        PUBLISH_2 : PUBLISH_2(ID := opc_ua[WRITE;%opcuaFolderTestWithNodeIdByteString2%]);
        folderTest2SameFolder2ByteString : TEST_CONDITION;
        folderTest2DifferentFolder2ByteString : TEST_CONDITION;
        E_PERMIT : E_PERMIT;
        F_EQ_1_1_1_2 : F_EQ(IN2 := %opcuaReadValue4%);
        F_EQ_1_1_1_1_1 : F_EQ(IN2 := %opcuaReadValue5%);
        PUBLISH_2_1 : PUBLISH_2(ID := opc_ua[WRITE;%opcuaFolderTestWithNodeIdByteString3%]);
        BOOL2BOOL_1_1_2 : DINT2DINT(IN := %opcuaReadValue3%);
        BOOL2BOOL_1_1_1_1_1 : DINT2DINT(IN := %opcuaReadValue5%);
        BOOL2BOOL_2 : DINT2DINT(IN := %opcuaReadValue1%);
        BOOL2BOOL_1_1_1_3 : DINT2DINT;
        BOOL2BOOL_1_1_3 : DINT2DINT;
        BOOL2BOOL_1_1_1_2 : DINT2DINT(IN := %opcuaReadValue4%);
        F_EQ_1_1_2 : F_EQ(IN2 := %opcuaReadValue3%);
        PUBLISH_1 : PUBLISH_1(ID := opc_ua[WRITE;%opcuaFolderTestWithNodeIdByteString1%]);
        E_CTU : E_CTU(PV := UINT#3);
        folderTest2SameFolder1ByteString : TEST_CONDITION;
        SUBSCRIBE_1_1 : SUBSCRIBE_1(ID := opc_ua[READ;%opcuaFolderTestWithNodeIdByteString1%]);
        BOOL2BOOL_1_1_1_1_2 : DINT2DINT;
        folderTest2DifferentFolder1ByteString : TEST_CONDITION;
        SUBSCRIBE_2_2 : SUBSCRIBE_2(ID := opc_ua[READ;%opcuaFolderTestWithNodeIdByteString2%]);
        SUBSCRIBE_2_1_1 : SUBSCRIBE_2(ID := opc_ua[READ;%opcuaFolderTestWithNodeIdByteString3%]);
        BOOL2BOOL_1_3 : DINT2DINT;
        BOOL2BOOL_3 : DINT2DINT;
        folderTestDirectUnderByteString : TEST_CONDITION;
      END_FBS
      EVENT_CONNECTIONS
        BOOL2BOOL_2.CNF TO BOOL2BOOL_1_2.REQ;
        BOOL2BOOL_1_2.CNF TO BOOL2BOOL_1_1_2.REQ;
        BOOL2BOOL_1_1_3.CNF TO F_EQ_1_2.REQ;
        F_EQ_1_2.CNF TO folderTest2SameFolder1ByteString.REQ;
        BOOL2BOOL_3.CNF TO F_EQ_2.REQ;
        F_EQ_2.CNF TO folderTestDirectUnderByteString.REQ;
        PUBLISH_2_1.INITO TO PUBLISH_2.INIT;
        PUBLISH_2_1.CNF TO PUBLISH_2.REQ;
        PUBLISH_2.INITO TO PUBLISH_1.INIT;
        PUBLISH_2.CNF TO PUBLISH_1.REQ;
        F_EQ_1_1_2.CNF TO folderTest2SameFolder2ByteString.REQ;
        F_EQ_1_1_1_1_1.CNF TO folderTest2DifferentFolder2ByteString.REQ;
        E_CTU.CUO TO E_PERMIT.EI;
        BOOL2BOOL_1_1_1_1_2.CNF TO F_EQ_1_1_1_2.REQ;
        F_EQ_1_1_1_2.CNF TO folderTest2DifferentFolder1ByteString.REQ;
        folderTest2DifferentFolder1ByteString.CNF TO F_EQ_1_1_1_1_1.REQ;
        BOOL2BOOL_1_1_1_1_1.CNF TO PUBLISH_2_1.REQ;
        BOOL2BOOL_1_1_2.CNF TO BOOL2BOOL_1_1_1_2.REQ;
        BOOL2BOOL_1_1_1_2.CNF TO BOOL2BOOL_1_1_1_1_1.REQ;
        SUBSCRIBE_2_1_1.IND TO BOOL2BOOL_1_1_1_3.REQ;
        BOOL2BOOL_1_1_1_3.CNF TO BOOL2BOOL_1_1_1_1_2.REQ;
        BOOL2BOOL_1_3.CNF TO BOOL2BOOL_1_1_3.REQ;
        folderTest2SameFolder1ByteString.CNF TO F_EQ_1_1_2.REQ;
        SUBSCRIBE_1_1.INITO TO SUBSCRIBE_2_2.INIT;
        SUBSCRIBE_1_1.IND TO BOOL2BOOL_3.REQ;
        SUBSCRIBE_2_2.INITO TO SUBSCRIBE_2_1_1.INIT;
        SUBSCRIBE_2_2.IND TO BOOL2BOOL_1_3.REQ;
        PUBLISH_1.INITO TO INITO;
        INIT TO SUBSCRIBE_1_1.INIT;
        folderTestDirectUnderByteString.CNF TO E_CTU.CU;
        folderTest2SameFolder2ByteString.CNF TO E_CTU.CU;
        folderTest2DifferentFolder2ByteString.CNF TO E_CTU.CU;
        E_PERMIT.EO TO CNF;
        REQ TO BOOL2BOOL_2.REQ;
        SUBSCRIBE_2_1_1.INITO TO PUBLISH_2_1.INIT;
      END_CONNECTIONS
      DATA_CONNECTIONS
        BOOL2BOOL_1_2.OUT TO PUBLISH_2.SD_1;
        BOOL2BOOL_1_3.OUT TO F_EQ_1_2.IN1;
        F_EQ_1_2.OUT TO folderTest2SameFolder1ByteString.check;
        BOOL2BOOL_3.OUT TO F_EQ_2.IN1;
        F_EQ_2.OUT TO folderTestDirectUnderByteString.check;
        BOOL2BOOL_1_1_2.OUT TO PUBLISH_2.SD_2;
        F_EQ_1_1_2.OUT TO folderTest2SameFolder2ByteString.check;
        F_EQ_1_1_1_1_1.OUT TO folderTest2DifferentFolder2ByteString.check;
        E_CTU.Q TO E_PERMIT.PERMIT;
        BOOL2BOOL_1_1_1_3.OUT TO F_EQ_1_1_1_2.IN1;
        F_EQ_1_1_1_2.OUT TO folderTest2DifferentFolder1ByteString.check;
        BOOL2BOOL_1_1_1_1_2.OUT TO F_EQ_1_1_1_1_1.IN1;
        BOOL2BOOL_1_1_1_2.OUT TO PUBLISH_2_1.SD_1;
        BOOL2BOOL_1_1_1_1_1.OUT TO PUBLISH_2_1.SD_2;
        BOOL2BOOL_2.OUT TO PUBLISH_1.SD_1;
        SUBSCRIBE_2_1_1.RD_1 TO BOOL2BOOL_1_1_1_3.IN;
        SUBSCRIBE_2_2.RD_2 TO BOOL2BOOL_1_1_3.IN;
        BOOL2BOOL_1_1_3.OUT TO F_EQ_1_1_2.IN1;
        SUBSCRIBE_1_1.RD_1 TO BOOL2BOOL_3.IN;
        SUBSCRIBE_2_1_1.RD_2 TO BOOL2BOOL_1_1_1_1_2.IN;
        SUBSCRIBE_2_2.RD_1 TO BOOL2BOOL_1_3.IN;
        QI TO SUBSCRIBE_1_1.QI;
        QI TO SUBSCRIBE_2_2.QI;
        QI TO SUBSCRIBE_2_1_1.QI;
        QI TO PUBLISH_1.QI;
        QI TO PUBLISH_2.QI;
        QI TO PUBLISH_2_1.QI;
      END_CONNECTIONS
    END_SUBAPPLICATION
    SUBAPPLICATION foldersWithNodeStringId
      EVENT_INPUT
        INIT;
        REQ;
      END_EVENT
      EVENT_OUTPUT
        INITO;
        CNF;
      END_EVENT
      VAR_INPUT
        QI : BOOL;
      END_VAR
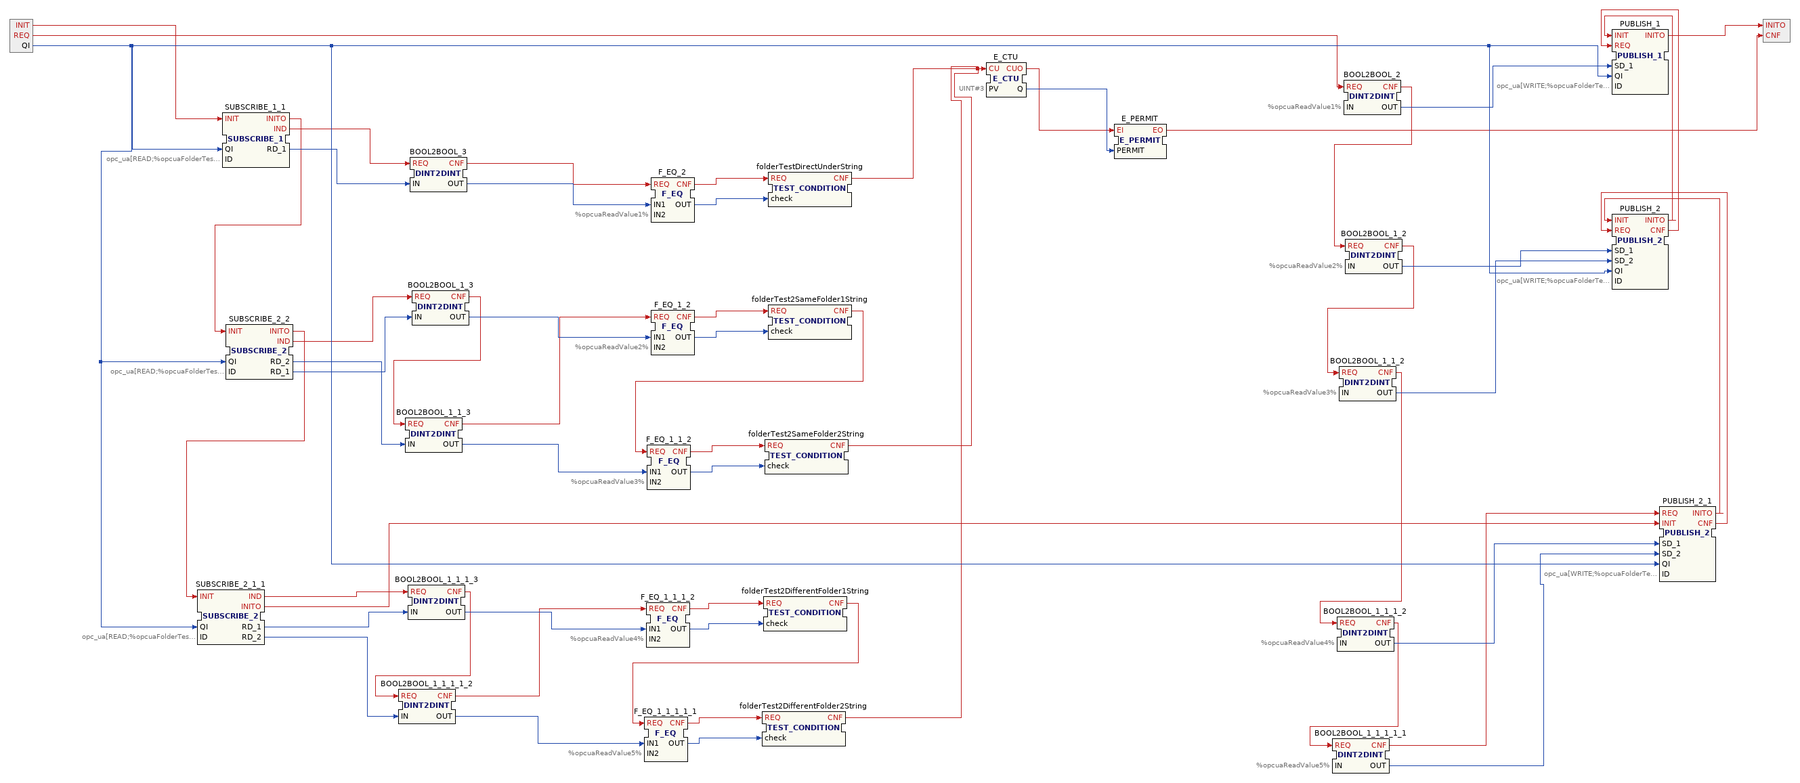
      FBS
        BOOL2BOOL_1_2 : DINT2DINT(IN := %opcuaReadValue2%);
        F_EQ_1_2 : F_EQ(IN2 := %opcuaReadValue2%);
        F_EQ_2 : F_EQ(IN2 := %opcuaReadValue1%);
        PUBLISH_2 : PUBLISH_2(ID := opc_ua[WRITE;%opcuaFolderTestWithNodeIdString2%]);
        folderTest2SameFolder2String : TEST_CONDITION;
        folderTest2DifferentFolder2String : TEST_CONDITION;
        E_PERMIT : E_PERMIT;
        F_EQ_1_1_1_2 : F_EQ(IN2 := %opcuaReadValue4%);
        F_EQ_1_1_1_1_1 : F_EQ(IN2 := %opcuaReadValue5%);
        PUBLISH_2_1 : PUBLISH_2(ID := opc_ua[WRITE;%opcuaFolderTestWithNodeIdString3%]);
        BOOL2BOOL_1_1_2 : DINT2DINT(IN := %opcuaReadValue3%);
        BOOL2BOOL_1_1_1_1_1 : DINT2DINT(IN := %opcuaReadValue5%);
        BOOL2BOOL_2 : DINT2DINT(IN := %opcuaReadValue1%);
        BOOL2BOOL_1_1_1_3 : DINT2DINT;
        BOOL2BOOL_1_1_3 : DINT2DINT;
        BOOL2BOOL_1_1_1_2 : DINT2DINT(IN := %opcuaReadValue4%);
        F_EQ_1_1_2 : F_EQ(IN2 := %opcuaReadValue3%);
